   // sequencer 1: S01-S99 初始化 / S01-S99 Initial
   INITIAL_STEP F12_Initial:   // S1, max time T#10S, warning time T#7S
              S    #ioPM_Inface.InitialRun
              R    #ioPM_Inface.InitialOK
              R    #ioPM_Inface.WaitRunning
              R    #ioPM_Inface.Running
              R    #ioPM_Inface.ProcessComplete
              R    #ioPM_Inface.UnPause
              R    "Station_Sys".Cmd.Calibration
              R    "Station_Sys".Cmd.ChangeOver
                   //"ST350_Sys".Cmd.DryRun
              R    "Station_Sys".Cmd.Reserve
              R    "Station_Sys".Cmd.OneCycle
          S1  N    "AutoProcessControl".A_Table_2Loading.ServoRunCount:=0
              R    #ioPM_Inface.ProcessStart
   END_STEP
   TRANSITION Trans1 FROM F12_Initial TO S2   // T1
      := #iSysInface.Ready;
   END_TRANSITION
   STEP S2:   // S2, max time T#10S, warning time T#7S
   END_STEP
   TRANSITION Trans2 FROM S2 TO S3   // T2
      := TRUE;
   END_TRANSITION
   STEP S4:   // S4, max time T#10S, warning time T#7S
   END_STEP
   TRANSITION Trans3 FROM S4 TO S5_MESInitial   // T3
      := TRUE;
   END_TRANSITION
   STEP S5_MESInitial:   // S5, max time T#10S, warning time T#7S
   END_STEP
   TRANSITION Trans325 FROM S5_MESInitial TO WaitRobotInitialFinish   // T4
      := TRUE;
   END_TRANSITION
   STEP S10_InitialFinish:   // S10, max time T#10S, warning time T#7S
              S    #ioPM_Inface.InitialOK
   END_STEP
   TRANSITION Trans102 FROM S10_InitialFinish TO ProcessStart   // T10, jump
      := #ioPM_Inface.Running;
   END_TRANSITION
   STEP S3:   // S3, max time T#10S, warning time T#7S
   END_STEP
   TRANSITION Trans613 FROM S3 TO "ServoReady?"   // T607
      := TRUE;
   END_TRANSITION
   STEP WaitRobotInitialFinish:   // S8, max time T#10S, warning time T#7S
   END_STEP
   TRANSITION Trans10 FROM WaitRobotInitialFinish TO "CheckA-Loading-02HorizontalCylinderPos"   // T8
      := "KukaRobot3_CtrlDB".sROBtoPLC.User.Home.DO163_HomeSeqOK OR "KukaRobot3_CtrlDB".sROBtoPLC.Sys.SO.IN_HOME;
   END_TRANSITION
   STEP "A-Loading-02UpDownTakeCylinderToHP_2":   // S120, max time T#10S, warning time T#7S
              S    "ST10Cylinder".Cy[4].Inout.AutoGoHome
              R    "ST10Cylinder".Cy[4].Inout.AutoGoWork
   END_STEP
   TRANSITION Trans768 FROM "A-Loading-02UpDownTakeCylinderToHP_2" TO "A-Loading-02HorizontalCylinderToHP"   // T121
      := NOT "ST10Cylinder".Cy[4].In.WorkPositionSensor AND "ST10Cylinder".Cy[4].In.HomePositionSensor;
   END_TRANSITION
   STEP "CheckA-Loading-02HorizontalCylinderPos":   // S117, max time T#10S, warning time T#7S
   END_STEP
   TRANSITION Trans117 FROM "CheckA-Loading-02HorizontalCylinderPos" TO "A-Loading-02HorizontalCylinderToHP"   // T117
      := NOT "ST10Cylinder".Cy[3].In.WorkPositionSensor AND "ST10Cylinder".Cy[3].In.HomePositionSensor;
   END_TRANSITION
   TRANSITION Trans119 FROM "CheckA-Loading-02HorizontalCylinderPos" TO "A-Loading-02UpDownTakeCylinderToHP_2"   // T119
      := ("ST10Cylinder".Cy[3].In.WorkPositionSensor AND NOT "ST10Cylinder".Cy[3].In.HomePositionSensor) OR (NOT "ST10Cylinder".Cy[3].In.WorkPositionSensor AND NOT "ST10Cylinder".Cy[3].In.HomePositionSensor);
   END_TRANSITION
   STEP "A-Loading-02HorizontalCylinderToHP":   // S119, max time T#10S, warning time T#7S
              S    "ST10Cylinder".Cy[3].Inout.AutoGoHome
              R    "ST10Cylinder".Cy[3].Inout.AutoGoWork
   END_STEP
   TRANSITION Trans767 FROM "A-Loading-02HorizontalCylinderToHP" TO "A-Loading-02UpDownTakeCylinderToWP"   // T120
      := NOT "ST10Cylinder".Cy[3].In.WorkPositionSensor AND "ST10Cylinder".Cy[3].In.HomePositionSensor;
   END_TRANSITION
   STEP "A-Loading-02UpDownTakeCylinderToWP":   // S116, max time T#10S, warning time T#7S
              R    "ST10Cylinder".Cy[4].Inout.AutoGoHome
              S    "ST10Cylinder".Cy[4].Inout.AutoGoWork
   END_STEP
   TRANSITION Trans765 FROM "A-Loading-02UpDownTakeCylinderToWP" TO S10_InitialFinish   // T116
      := "ST10Cylinder".Cy[4].In.WorkPositionSensor AND NOT "ST10Cylinder".Cy[4].In.HomePositionSensor;
   END_TRANSITION
   STEP "ServoReady?":   // S6, max time T#10S, warning time T#7S
   END_STEP
   TRANSITION Trans4 FROM "ServoReady?" TO S4   // T5
      := "ServoV90_A4".Out.oReady;
   END_TRANSITION

   // sequencer 2: S100-S199 等待到位 / S100-S199 CheckSysStatus
   STEP "A-Loading-02HorizontalCylinderToWP_1":   // S121, max time T#10S, warning time T#7S
              R    "ST10Cylinder".Cy[3].Inout.AutoGoHome
              S    "ST10Cylinder".Cy[3].Inout.AutoGoWork
   END_STEP
   TRANSITION Trans769 FROM "A-Loading-02HorizontalCylinderToWP_1" TO TimDelay   // T122
      := "ST10Cylinder".Cy[3].In.WorkPositionSensor AND NOT "ST10Cylinder".Cy[3].In.HomePositionSensor;
   END_TRANSITION
   STEP "A-Loading-02UpDownTakeCylinderToHP3":   // S122, max time T#10S, warning time T#7S
              S    "ST10Cylinder".Cy[4].Inout.AutoGoHome
              R    "ST10Cylinder".Cy[4].Inout.AutoGoWork
   END_STEP
   TRANSITION Trans770 FROM "A-Loading-02UpDownTakeCylinderToHP3" TO "A-Loading-02HorizontalCylinderToWP_1"   // T123
      := NOT "ST10Cylinder".Cy[4].In.WorkPositionSensor AND "ST10Cylinder".Cy[4].In.HomePositionSensor;
   END_TRANSITION
   STEP TimDelay:   // S123, max time T#10S, warning time T#7S
   END_STEP
   TRANSITION Trans124 FROM TimDelay TO "A-Loading-02UpDownTakeCylinderToWP_1"   // T124
      := #TimDelay.T > t#100MS;
   END_TRANSITION
   STEP SensorNoPart:   // S113, max time T#10S, warning time T#7S
   END_STEP
   TRANSITION Trans113 FROM SensorNoPart TO WaitEmptyFinish   // T113
      := #TOF[5].Q;
   END_TRANSITION
   STEP ProcessStart:   // S100, max time T#10S, warning time T#7S
      // 自动等待开始运行
              R    #ioPM_Inface.InitialRun
              R    #ioPM_Inface.ProcessComplete
              R    #ioPM_Inface.ProcessStart
              S    #ioPM_Inface.InitialOK
              S    #ioPM_Inface.WaitRunning
          S1  N    #ioPM_Inface.ProcessResult:=0
              R    "ST10_GeneralData".FlowControl_Handshake[12].Start
              R    "ST10_GeneralData".FlowControl_Handshake[12].Done
   END_STEP
   TRANSITION Trans200 FROM ProcessStart TO WaitChangeOverFinish   // T100
      := NOT #ioPM_Inface.AlarmCycleStop AND #ioPM_Inface.Running AND NOT #iSysInface.Auto.RunningOver AND (NOT #iSysInface.Auto.OneCycleMode OR (#iSysInface.Auto.OneCycleMode AND #ioPM_Inface.TriggerOneCycle));
   END_TRANSITION
   STEP TimDelay_1:   // S124, max time T#10S, warning time T#7S
   END_STEP
   TRANSITION Trans125 FROM TimDelay_1 TO "A-Loading-02HorizontalCylinderToHP_1"   // T125
      := #TimDelay_1.T > t#1S;
   END_TRANSITION
   STEP "Process Finish":   // S237, max time T#10S, warning time T#7S
   END_STEP
   TRANSITION Trans250 FROM "Process Finish" TO ProcessStart   // T249, jump
      := TRUE;
   END_TRANSITION
   STEP "A-Loading-02HorizontalCylinderToHP_1":   // S125, max time T#10S, warning time T#7S
              S    "ST10Cylinder".Cy[3].Inout.AutoGoHome
              R    "ST10Cylinder".Cy[3].Inout.AutoGoWork
   END_STEP
   TRANSITION Trans771 FROM "A-Loading-02HorizontalCylinderToHP_1" TO "Detect UnloadingRing exist_1"   // T126
      := NOT "ST10Cylinder".Cy[3].In.WorkPositionSensor AND "ST10Cylinder".Cy[3].In.HomePositionSensor;
   END_TRANSITION
   STEP "No cartridge":   // S127, max time T#10S, warning time T#7S
   END_STEP
   TRANSITION Trans129 FROM "No cartridge" TO ServoNeedMove   // T129, jump
      := TRUE;
   END_TRANSITION
   STEP "A-Loading-02UpDownTakeCylinderToWP_1":   // S118, max time T#10S, warning time T#7S
              R    "ST10Cylinder".Cy[4].Inout.AutoGoHome
              S    "ST10Cylinder".Cy[4].Inout.AutoGoWork
   END_STEP
   TRANSITION Trans766 FROM "A-Loading-02UpDownTakeCylinderToWP_1" TO TimDelay_1   // T118
      := "ST10Cylinder".Cy[4].In.WorkPositionSensor AND NOT "ST10Cylinder".Cy[4].In.HomePositionSensor;
   END_TRANSITION
   STEP ServoNeedMove:   // S126, max time T#10S, warning time T#7S
   END_STEP
   TRANSITION Trans128 FROM ServoNeedMove TO WaitChangeOverOK   // T128
      := TRUE;
   END_TRANSITION
   STEP WaitChangeOverFinish:   // S101, max time T#10S, warning time T#7S
   END_STEP
   TRANSITION Trans101 FROM WaitChangeOverFinish TO "Clearing mode?"   // T101
      := TRUE;
   END_TRANSITION
   STEP WaitServoInPosition:   // S105, max time T#10S, warning time T#7S
              R    #ioPM_Inface.ProcessComplete
              S    #ioPM_Inface.ProcessStart
   END_STEP
   TRANSITION Trans103 FROM WaitServoInPosition TO WaitFixtureScanFinish   // T105
      := TRUE;
   END_TRANSITION
   TRANSITION Trans127 FROM WaitServoInPosition TO ServoNeedMove   // T127
      := "AlwaysTRUE" AND NOT "AlwaysTRUE";
   END_TRANSITION
   STEP "Detect cartridge exist":   // S106, max time T#10S, warning time T#7S
   END_STEP
   TRANSITION Trans106 FROM "Detect cartridge exist" TO CountClear   // T106
      := "ServoV90_A4".Out.oServoPosOK AND #TON[0].Q;
   END_TRANSITION
   TRANSITION Trans107 FROM "Detect cartridge exist" TO "No cartridge"   // T107
      := (NOT "iA-Loading-02PipeDetection" OR NOT "ServoV90_A4".Out.oServoPosOK) AND (#"Detect cartridge exist".T > t#1500MS);
   END_TRANSITION
   STEP "Detect UnloadingRing exist":   // S108, max time T#10S, warning time T#7S
   END_STEP
   TRANSITION Trans110 FROM "Detect UnloadingRing exist" TO "Request robot pick"   // T110
      := #TON[4].Q;
   END_TRANSITION
   TRANSITION Trans111 FROM "Detect UnloadingRing exist" TO "A-Loading-02UpDownTakeCylinderToHP3"   // T111
      := #TOF[5].Q AND NOT "ChangeOver_DB".Global.ScanFixtureFlag AND "ChangeOver_DB".Global.AllFixtureScanCompareOk AND "AutoProcessData".GlobalData.Table2CodeOKFlag;
   END_TRANSITION
   STEP "Detect Ring exist":   // S107, max time T#10S, warning time T#7S
   END_STEP
   TRANSITION Trans108 FROM "Detect Ring exist" TO Step111   // T108
      := #TON[2].Q;
   END_TRANSITION
   TRANSITION Trans109 FROM "Detect Ring exist" TO "No Ring"   // T109
      := NOT "iA-Loading-02Detection" AND (#"Detect Ring exist".T > t#1500MS);
   END_TRANSITION
   STEP "Wait  robot finish task":   // S130, max time T#10S, warning time T#7S
   END_STEP
   TRANSITION Trans146 FROM "Wait  robot finish task" TO SensorNoPart   // T146
      := "KukaRobot3_CtrlDB".sROBtoPLC.User.Cycle.DO258_PickTableFinish;
   END_TRANSITION
   STEP "Request robot pick":   // S112, max time T#10S, warning time T#7S
              N    "AutoProcessControl".A_Table_2Loading.Robot3PickPrimit
              S    #ioPM_Inface.ProcessComplete
              R    #ioPM_Inface.ProcessStart
   END_STEP
   TRANSITION Trans283 FROM "Request robot pick" TO "Wait  robot finish task"   // T112
      := "KukaRobot3_CtrlDB".sROBtoPLC.User.Cycle.DO257_PickTableInside AND NOT "KukaRobot3_CtrlDB".sROBtoPLC.User.Cycle.DO258_PickTableFinish;
   END_TRANSITION
   STEP "No Ring":   // S128, max time T#10S, warning time T#7S
   END_STEP
   TRANSITION Trans130 FROM "No Ring" TO ServoNeedMove   // T130, jump
      := TRUE;
   END_TRANSITION
   STEP "Detect UnloadingRing exist_1":   // S109, max time T#10S, warning time T#7S
   END_STEP
   TRANSITION Trans112 FROM "Detect UnloadingRing exist_1" TO ResetPartMissingAlarm   // T114
      := #TON[4].Q;
   END_TRANSITION
   TRANSITION Trans115 FROM "Detect UnloadingRing exist_1" TO PartMissingAlarm   // T115
      := NOT "iA-Loading-02GripperTakeDetection" AND (#"Detect UnloadingRing exist_1".T > t#3000MS);
   END_TRANSITION
   STEP PartMissingAlarm:   // S110, max time T#10S, warning time T#7S
          S1  S    "ST10_DeviceError".A.A2TableUnloading.RingCheckExist
   END_STEP
   TRANSITION Trans131 FROM PartMissingAlarm TO ProcessStart   // T131, jump
      := #iSysInface.Reset OR NOT "ST10_DeviceError"."A".A2TableUnloading.RingCheckExist;
   END_TRANSITION
   STEP Step111:   // S111, max time T#10S, warning time T#7S
          S1  N    "AutoProcessControl".A_Table_2Loading.ServoRunCount:=0
   END_STEP
   TRANSITION Trans132 FROM Step111 TO "Detect UnloadingRing exist"   // T132
      := TRUE;
   END_TRANSITION
   STEP CountClear:   // S114, max time T#10S, warning time T#7S
   END_STEP
   TRANSITION Trans133 FROM CountClear TO "Detect Ring exist"   // T133
      := TRUE;
   END_TRANSITION
   STEP "Servo returns to1st Pos":   // S16, max time T#10S, warning time T#7S
      interlock C := "ServoV90_A4".Out.oReady;
      (C)     N    "ServoV90_DeviceCtl".V90Servo[4].Point["ServoV90_DeviceCtl".V90Servo[4].nPositionListNo].Start
   END_STEP
   TRANSITION Trans17 FROM "Servo returns to1st Pos" TO CountCompare   // T16
      := "ServoV90_DeviceCtl".V90Servo[4].Point["ServoV90_DeviceCtl".V90Servo[4].nPositionListNo].Achieve;
   END_TRANSITION
   STEP ServoPosCount:   // S17, max time T#10S, warning time T#7S
          S1  N    "ServoV90_DeviceCtl".V90Servo[4].nPositionListNo:= "ServoV90_DeviceCtl".V90Servo[4].nPositionListNo+1
          S1  N    "AutoProcessControl".A_Table_2Loading.ServoRunCount:="AutoProcessControl".A_Table_2Loading.ServoRunCount+1
   END_STEP
   TRANSITION Trans18 FROM ServoPosCount TO ServoPosCountJudge   // T17
      := TRUE;
   END_TRANSITION
   STEP ServoPosCountJudge:   // S18, max time T#10S, warning time T#7S
   END_STEP
   TRANSITION Trans19 FROM ServoPosCountJudge TO "Servo returns to1st Pos"   // T18
      := ("ServoV90_DeviceCtl".V90Servo[4].nPositionListNo >= 1) AND ("ServoV90_DeviceCtl".V90Servo[4].nPositionListNo <= 8);
   END_TRANSITION
   TRANSITION Trans20 FROM ServoPosCountJudge TO ServoPosCountClear   // T19
      := ("ServoV90_A4".Auto.Index <= 0) OR ("ServoV90_A4".Auto.Index > 8);
   END_TRANSITION
   STEP ServoPosCountClear:   // S19, max time T#10S, warning time T#7S
              N    "ServoV90_DeviceCtl".V90Servo[4].nPositionListNo:=1
   END_STEP
   TRANSITION Trans21 FROM ServoPosCountClear TO "Servo returns to1st Pos"   // T20
      := "ServoV90_DeviceCtl".V90Servo[4].nPositionListNo = 1;
   END_TRANSITION
   STEP CountCompare:   // S20, max time T#10S, warning time T#7S
   END_STEP
   TRANSITION Trans22 FROM CountCompare TO ProcessStart   // T21, jump
      := "AutoProcessControl".A_Table_2Loading.ServoRunCount <= 8;
   END_TRANSITION
   TRANSITION Trans23 FROM CountCompare TO TableLackMaterial   // T22
      := "AutoProcessControl".A_Table_2Loading.ServoRunCount > 8;
   END_TRANSITION
   STEP TableLackMaterial:   // S21, max time T#10S, warning time T#7S
          S1  S    "ST10_DeviceError".A.A2TableUnloading.LackMaterial
   END_STEP
   TRANSITION Trans24 FROM TableLackMaterial TO CountClear_1   // T23
      := #iSysInface.Reset;
   END_TRANSITION
   STEP CountClear_1:   // S115, max time T#10S, warning time T#7S
          S1  N    "AutoProcessControl".A_Table_2Loading.ServoRunCount:=1
   END_STEP
   TRANSITION Trans134 FROM CountClear_1 TO CountCompare   // T134, jump
      := TRUE;
   END_TRANSITION
   STEP "Clearing mode?":   // S129, max time T#10S, warning time T#7S
   END_STEP
   TRANSITION Trans135 FROM "Clearing mode?" TO WaitServoInPosition   // T135
      := NOT "Station_Sys".Cmd.ClearFlags OR ("Station_Sys".Cmd.ClearFlags AND "AutoProcessControl".B_Press_2.Robot3PutRingPrimit AND ("AutoProcessData".F_Robot3Grip2.PartStatus = 0));
   END_TRANSITION
   STEP WaitChangeOverOK:   // S133, max time T#10S, warning time T#7S
   END_STEP
   TRANSITION Trans139 FROM WaitChangeOverOK TO ServoPosCount   // T139
      := "ChangeOver_DB".Global.AllFixtureScanCompareOk AND NOT "ChangeOver_DB".Global.ScanFixtureFlag;
   END_TRANSITION
   TRANSITION Trans31 FROM WaitChangeOverOK TO "Detect UnloadingRing exist"   // T31, jump
      := NOT "ChangeOver_DB".Global.AllFixtureScanCompareOk AND #TON[4].Q AND NOT "ST10_GeneralData".FunctionDeSelect.Global.DeSelectPB_ScanFixture;
   END_TRANSITION
   STEP WaitEmptyFinish:   // S134, max time T#10S, warning time T#7S
   END_STEP
   TRANSITION Trans140 FROM WaitEmptyFinish TO "Process Finish"   // T140
      := NOT "ChangeOver_DB".Global.ManualModeFlag;
   END_TRANSITION
   STEP WaitFixtureScanFinish:   // S30, max time T#10S, warning time T#7S
   END_STEP
   TRANSITION Trans30 FROM WaitFixtureScanFinish TO "Detect cartridge exist"   // T30
      := (NOT "ChangeOver_DB".Global.ScanFixtureFlag AND NOT "ChangeOver_DB".Global.ChangeOverRequest) OR #TON[4].Q;
   END_TRANSITION
   STEP ResetPartMissingAlarm:   // S31, max time T#10S, warning time T#7S
   END_STEP
   TRANSITION Trans32 FROM ResetPartMissingAlarm TO "Detect UnloadingRing exist"   // T32, jump
      := TRUE;
   END_TRANSITION

   // permanent post-instructions
   NETWORK 1
      #ioPM_Inface.StepNum := #RT_DATA.S_DISPLAY;
   NETWORK 2
      IF #iSysInface.Reset THEN #AlarmID := 0; END_IF;
   NETWORK 3
      #TON[10].TON(IN := #工件放行中, PT := T#0.5S);
      IF #TON[10].Q THEN #工件放行中 := FALSE; END_IF;
END_FUNCTION_BLOCK

FUNCTION_BLOCK "ST10_Flow14_B2Press"   // FB1084, GRAPH
// stored: AcknowledgeErrorsRequired false, AutoNumber false, GraphVersion 6.0, InitialValuesAcquisition false, SetENOAutomatically false
   // inherited from GRAPH_BASE
   VAR_INPUT
      iSysInface : "RCS_SysComInterface_V1";
   END_VAR
   VAR_IN_OUT
      ioPM_Inface : "RCS_PMInterface_V1";
      ioStatus : Int;
   END_VAR
   VAR
      sCtrlMode { S7_SetPoint := 'True'} : "SysFlowCtrlGraph";
      sUpdMES_Data : Bool;   // 更新MES数据
      工件放行中 : Bool;
      前站站号 { ExternalAccessible := 'False'; ExternalVisible := 'False'; ExternalWritable := 'False'} : UInt;
      本站站号 { ExternalAccessible := 'False'; ExternalVisible := 'False'; ExternalWritable := 'False'} : UInt;
      弹窗Temp : Array[1..10] of Int;
      AlarmID : Int;
      TON { S7_SetPoint := 'True'} : Array[0..10] of TON_TIME;
      TOF { S7_SetPoint := 'True'} : Array[0..10] of TOF_TIME;
      sUP { S7_SetPoint := 'True'} : Array[0..10] of Bool;
      更新RFID完成 : Bool;
   END_VAR
   VAR_TEMP
      Tempresult : USInt;
      本站站号乘10 : UInt;
   END_VAR
   // // TON[0] : 托盘流入1托盘到位传感器 / iA-Rotating product Check
   // // TON[1] : 托盘流入1托盘到位传感器
   // // TON[2] : 托盘流入1产品有无传感器
   // // TON[3] : 托盘流入1产品有无传感器
   // // TON[4] : 托盘流入1姿态检测光电2
   // // TON[5] : 托盘流入1姿态检测光电3
   // // TON[0].Q : 托盘流入1托盘到位 / iA-Rotating product Check
   // // TON[1].Q : 托盘流入1托盘无
   // // TON[2].Q : 托盘流入1有产品
   // // TON[3].Q : 托盘流入1无产品
   // // TON[4].Q : 托盘流入1姿态检测光电2
   // // TON[5].Q : 托盘流入1姿态检测光电3
   // // TOF[1] : iA-Rotating product Check
BEGIN
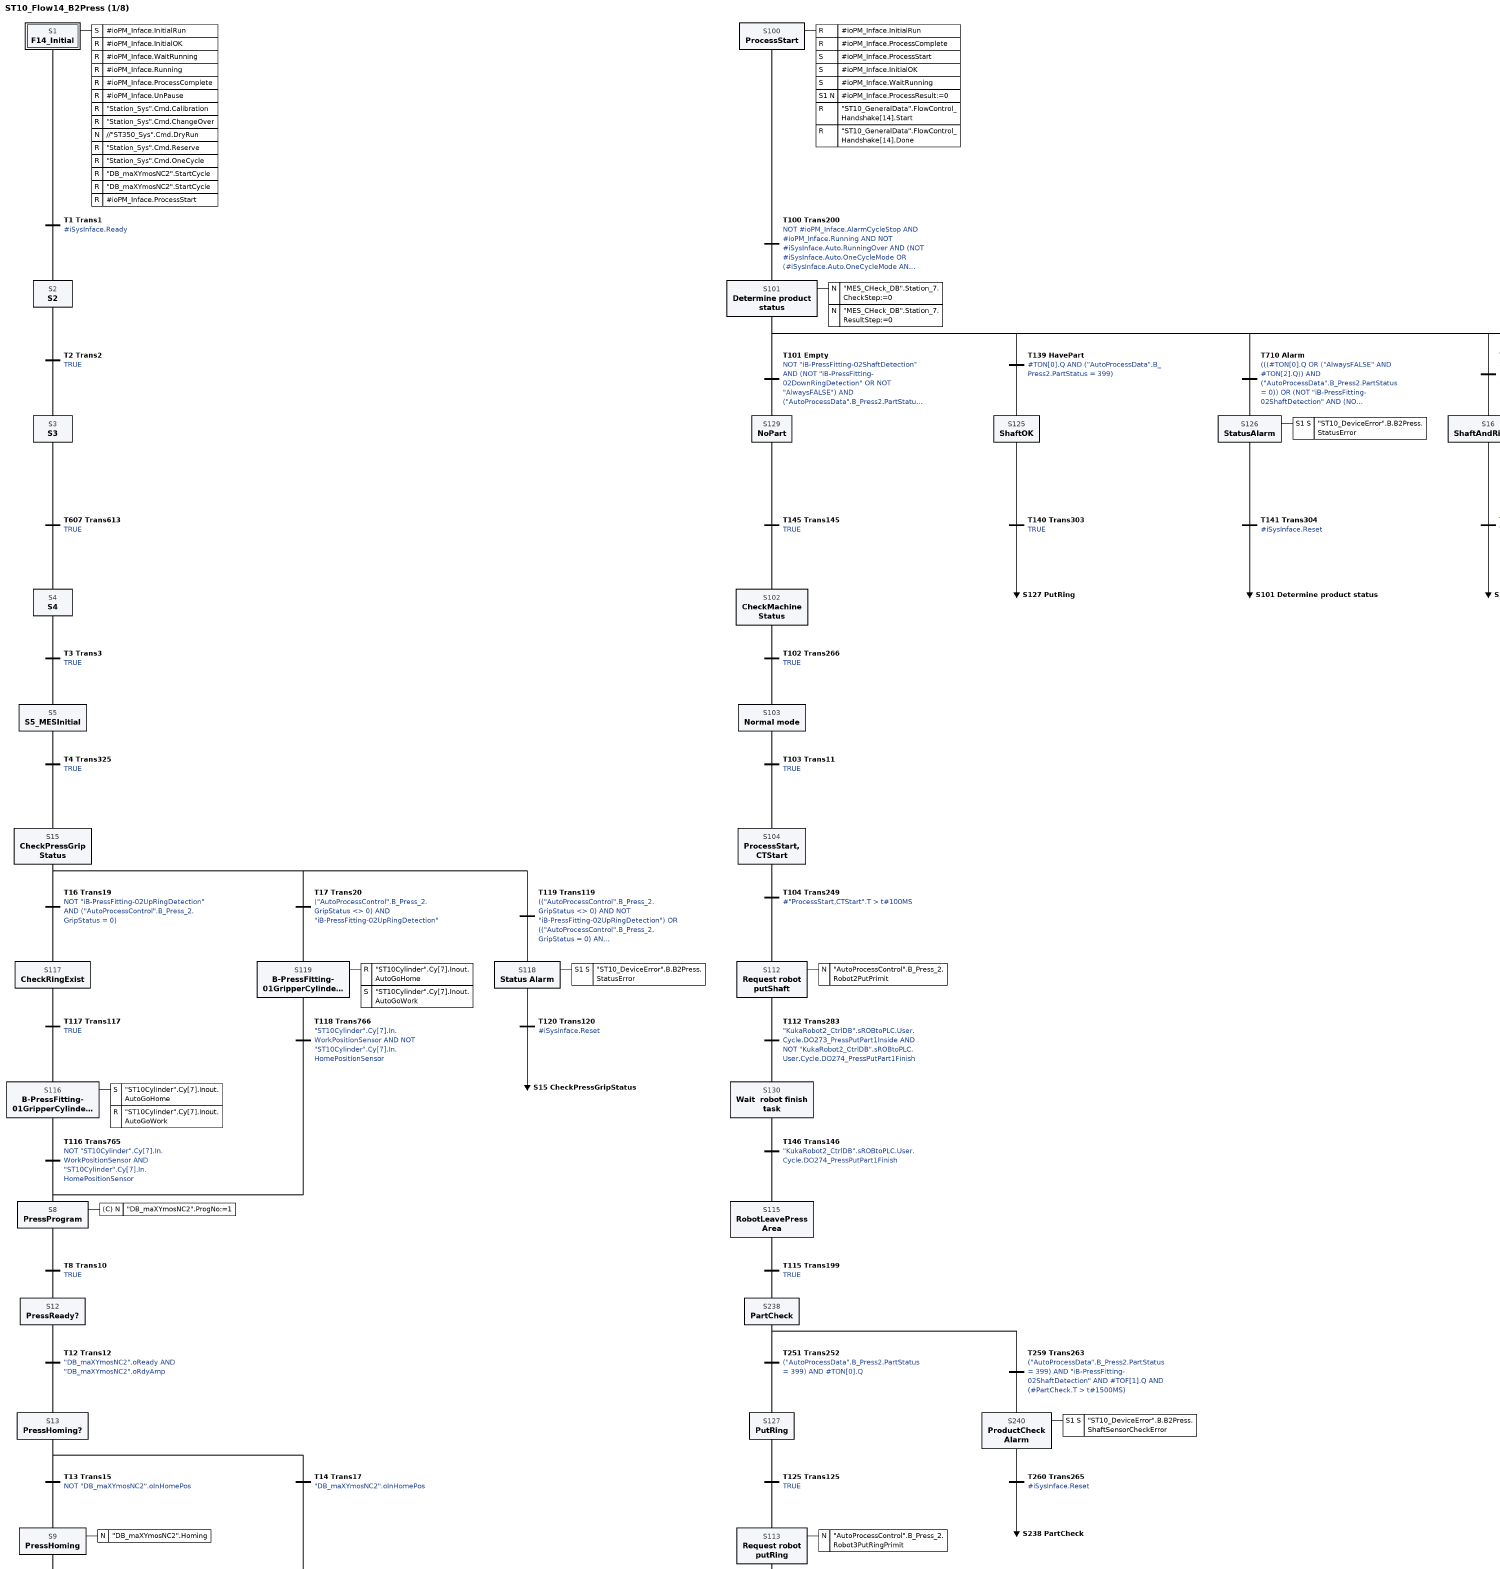
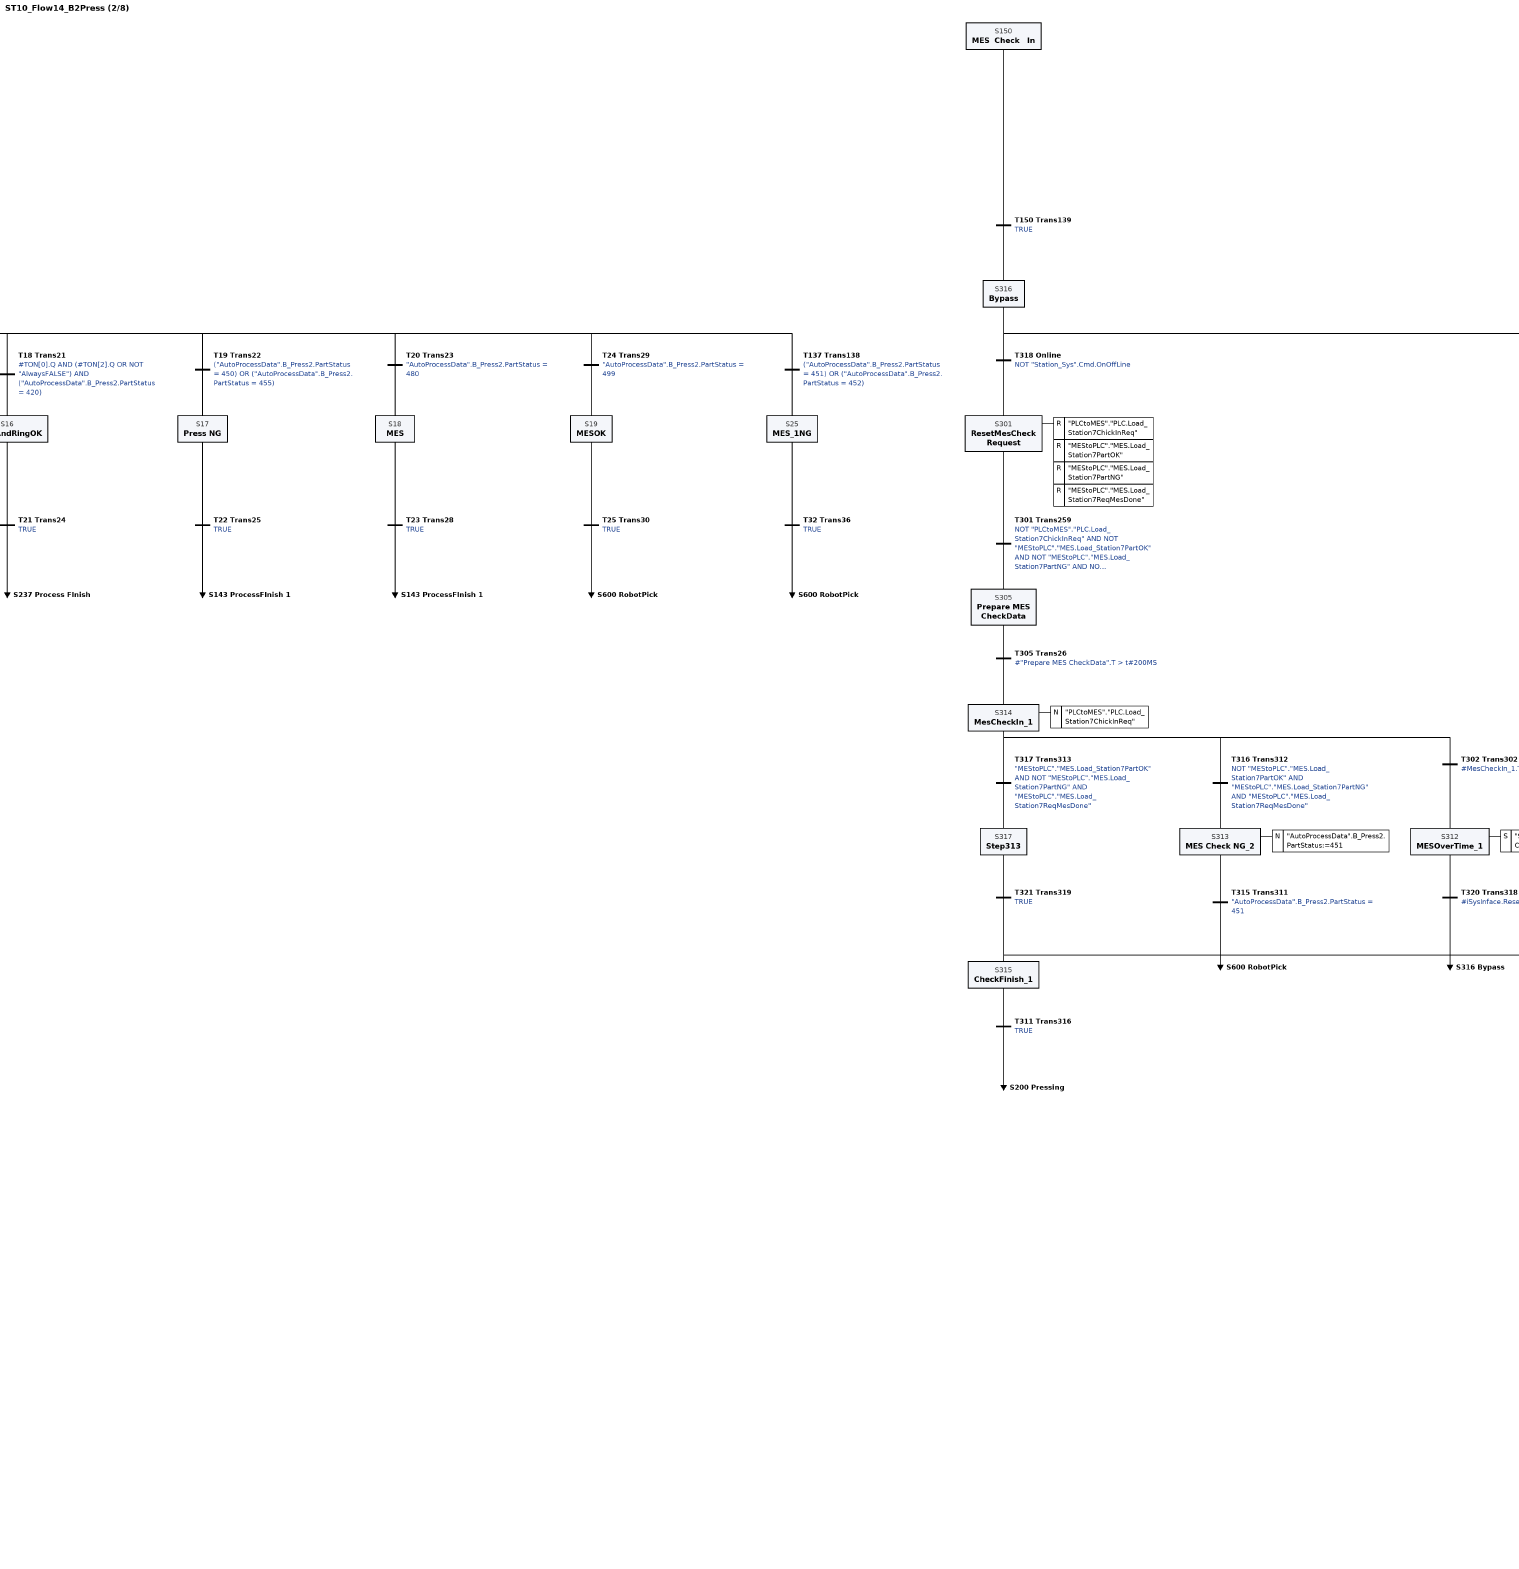
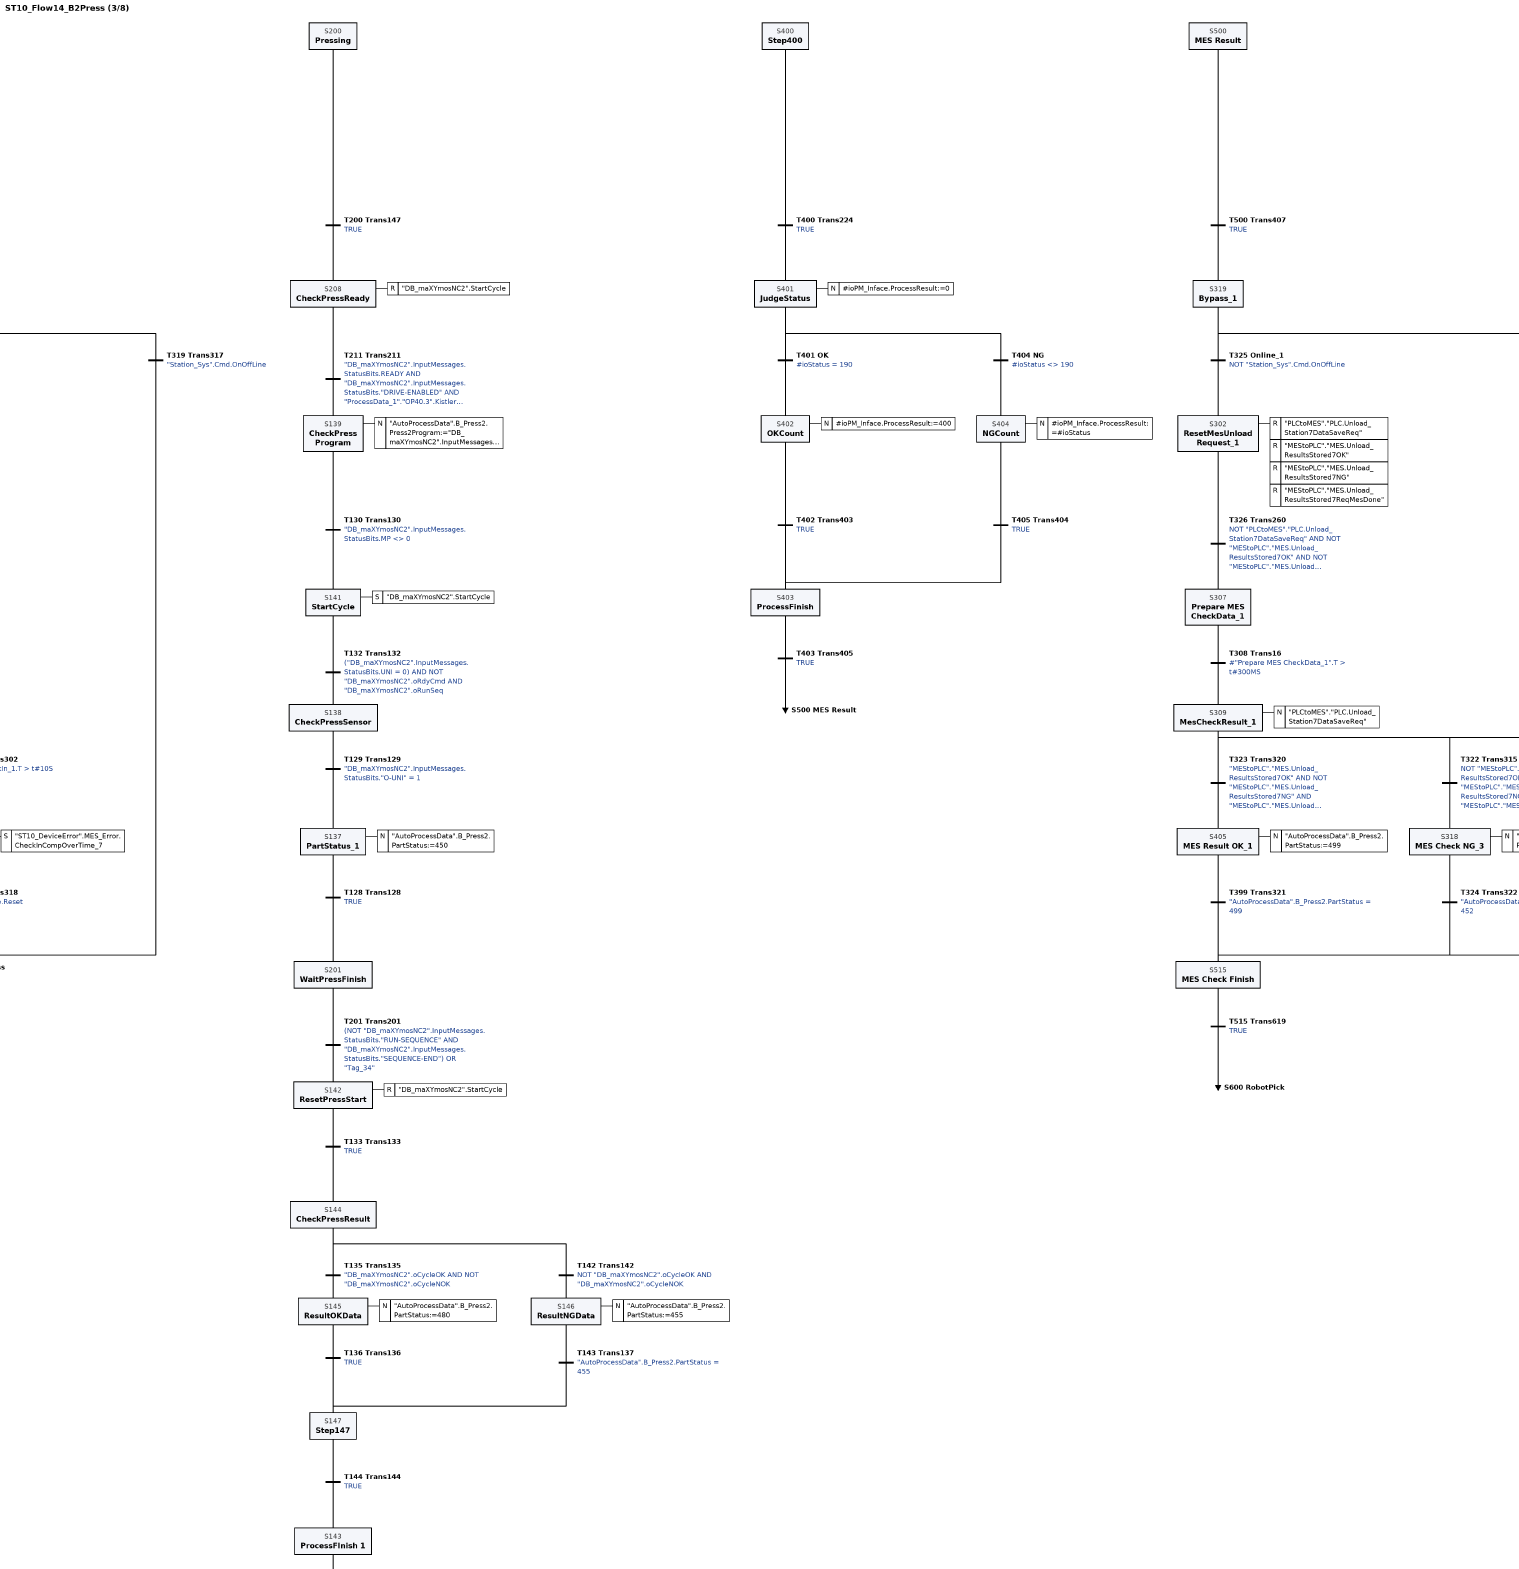
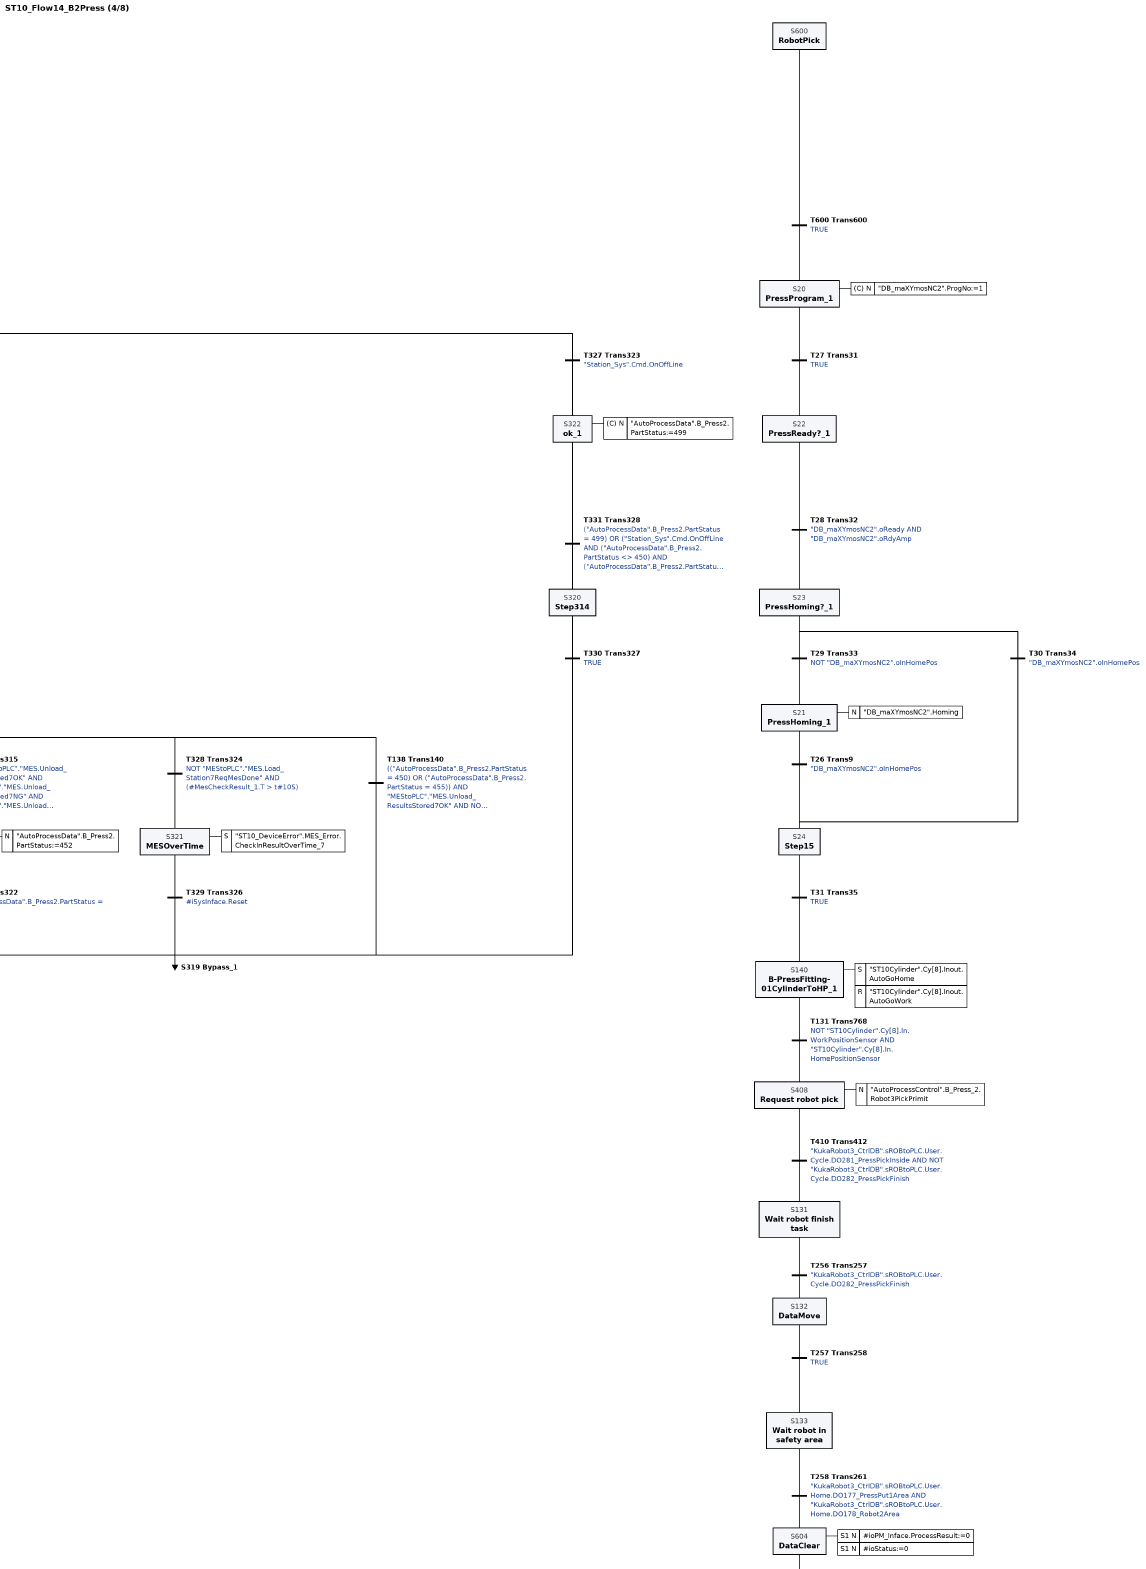
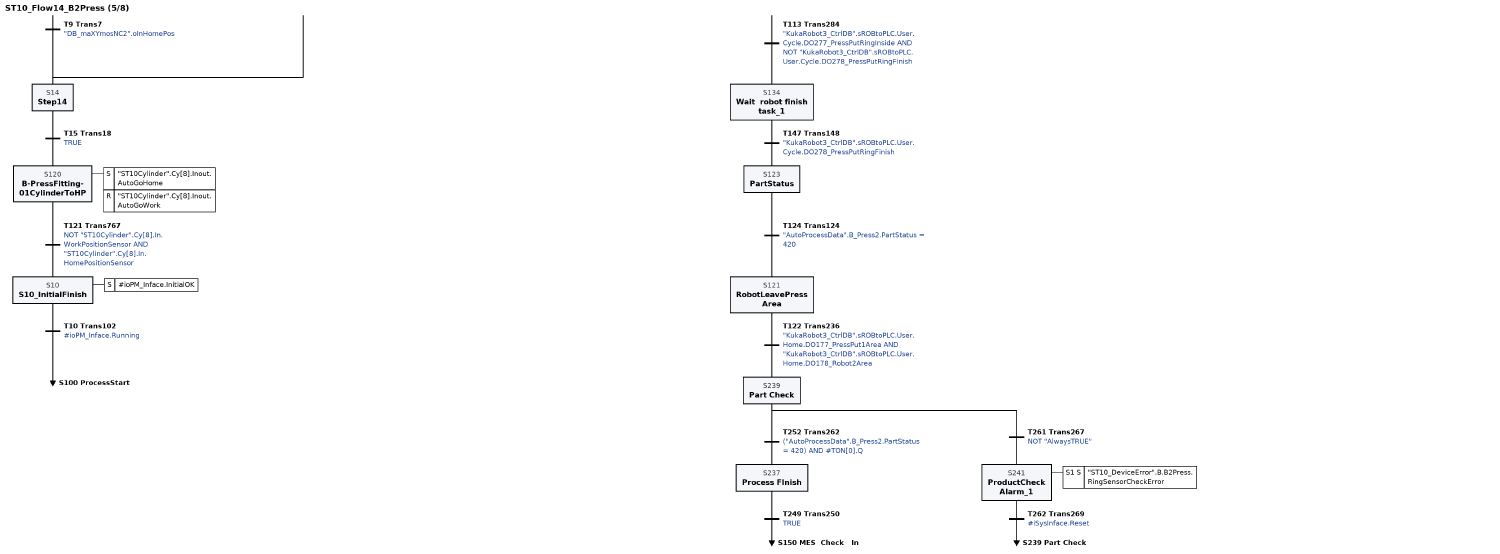
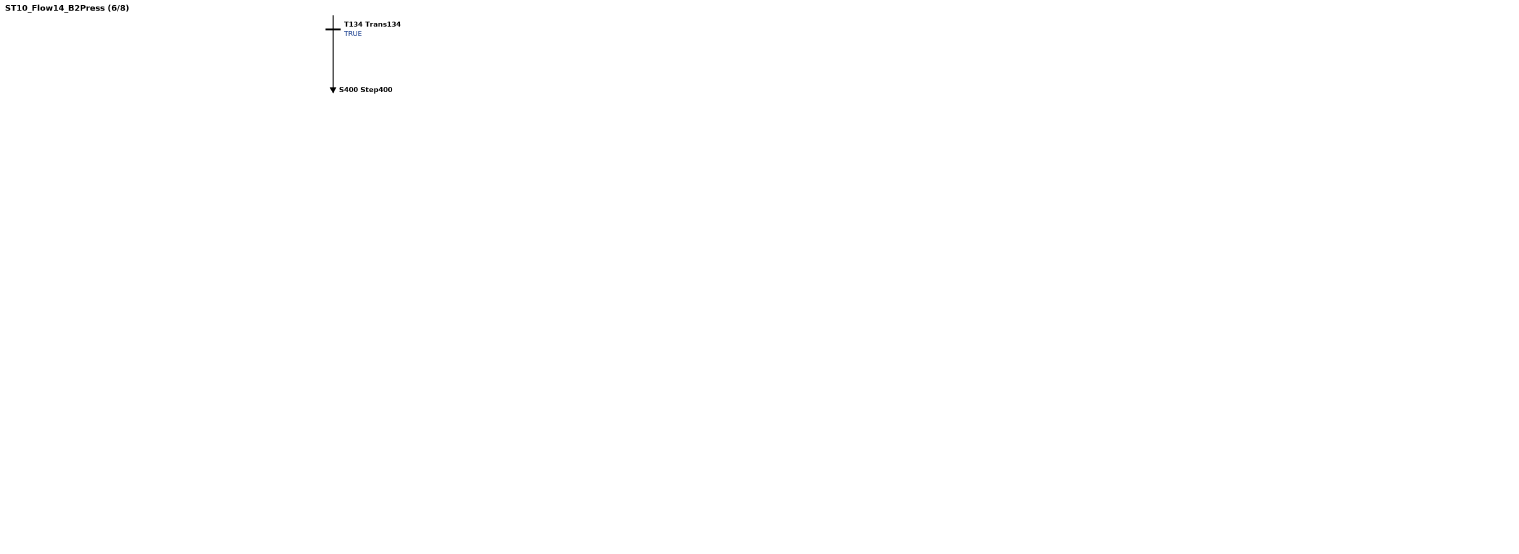
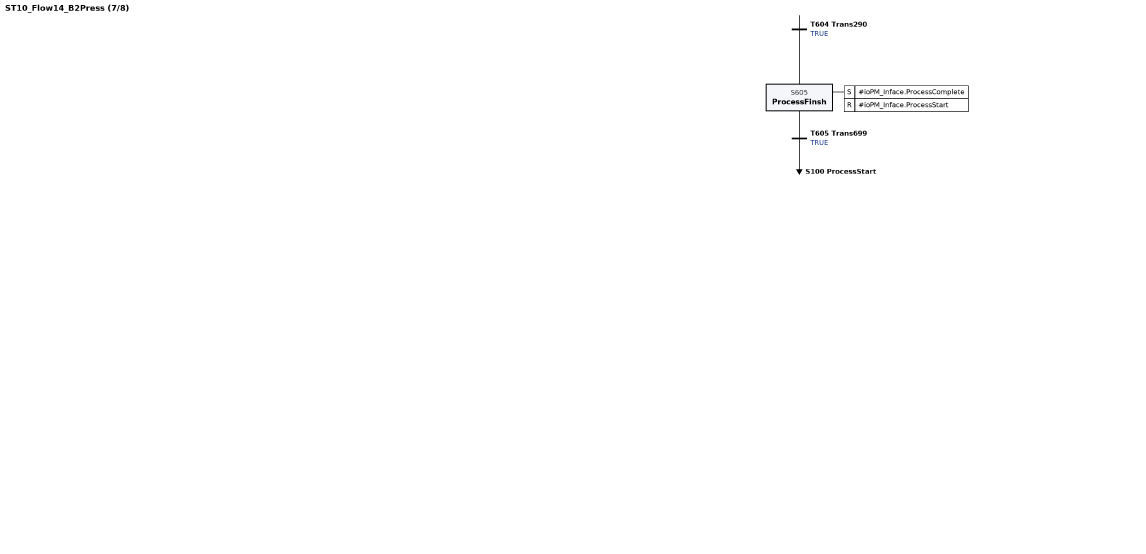
   // permanent pre-instructions
   NETWORK 1
      #TON[10].TON(IN := "AlwaysTRUE" AND "Station_Sys".Alarm.ImmediatelyStop, PT := T#300ms);
      #ioPM_Inface.AlarmImdilyStop := #TON[10].Q;
      #ioPM_Inface.AlarmCycleStop := "AlwaysTRUE" AND "Station_Sys".Alarm.CycleStop;
   NETWORK 2
      IF NOT False THEN
          #sCtrlMode(iSysInface := #iSysInface, ioPM_Inface := #ioPM_Inface, ioGraphCtrl := #RT_DATA.MOP);   // "SysFlowCtrlGraph"
      END_IF;
   NETWORK 3
      #TON[0].TON(IN := "AlwaysTRUE" AND "iB-PressFitting-02ShaftDetection", PT := t#500ms);   // 工位11有托盘
      #TOF[1].TOF(IN := "AlwaysTRUE" AND NOT "iB-PressFitting-02ShaftDetection", PT := T#300ms);   // 工位无托盘
      #TON[2].TON(IN := "AlwaysTRUE" AND "iB-PressFitting-02DownRingDetection", PT := T#300ms);
      #TOF[3].TOF(IN := "AlwaysTRUE" AND NOT "iB-PressFitting-02DownRingDetection", PT := T#300ms);
      #TON[4].TON(IN := "AlwaysTRUE" AND "iB-PressFitting-02UpRingDetection", PT := T#300ms);
      #TON[5].TON(IN := "AlwaysTRUE" AND NOT "iB-PressFitting-02UpRingDetection", PT := T#300ms);
   NETWORK 4
      #前站站号 := 345;
      #本站站号 := 350;

   // sequencer 1: S01-S99 初始化 / S01-S99 Initial
   INITIAL_STEP F14_Initial:   // S1, max time T#10S, warning time T#7S
              S    #ioPM_Inface.InitialRun
              R    #ioPM_Inface.InitialOK
              R    #ioPM_Inface.WaitRunning
              R    #ioPM_Inface.Running
              R    #ioPM_Inface.ProcessComplete
              R    #ioPM_Inface.UnPause
              R    "Station_Sys".Cmd.Calibration
              R    "Station_Sys".Cmd.ChangeOver
                   //"ST350_Sys".Cmd.DryRun
              R    "Station_Sys".Cmd.Reserve
              R    "Station_Sys".Cmd.OneCycle
              R    "DB_maXYmosNC2".StartCycle
              R    "DB_maXYmosNC2".StartCycle
              R    #ioPM_Inface.ProcessStart
              R    "AutoProcessControl".B_Press_2.Robot3PickPrimit
              R    "AutoProcessControl".B_Press_2.Robot3PutRingPrimit
              R    "AutoProcessControl".B_Press_2.Robot2PutPrimit
   END_STEP
   TRANSITION Trans1 FROM F14_Initial TO S2   // T1
      := #iSysInface.Ready;
   END_TRANSITION
   STEP S2:   // S2, max time T#10S, warning time T#7S
   END_STEP
   TRANSITION Trans2 FROM S2 TO S3   // T2
      := TRUE;
   END_TRANSITION
   STEP S4:   // S4, max time T#10S, warning time T#7S
   END_STEP
   TRANSITION Trans3 FROM S4 TO S5_MESInitial   // T3
      := TRUE;
   END_TRANSITION
   STEP S5_MESInitial:   // S5, max time T#10S, warning time T#7S
   END_STEP
   TRANSITION Trans325 FROM S5_MESInitial TO CheckPressGripStatus   // T4
      := TRUE;
   END_TRANSITION
   STEP S10_InitialFinish:   // S10, max time T#10S, warning time T#7S
              S    #ioPM_Inface.InitialOK
   END_STEP
   TRANSITION Trans102 FROM S10_InitialFinish TO ProcessStart   // T10, jump
      := #ioPM_Inface.Running;
   END_TRANSITION
   STEP S3:   // S3, max time T#10S, warning time T#7S
   END_STEP
   TRANSITION Trans613 FROM S3 TO S4   // T607
      := TRUE;
   END_TRANSITION
   STEP PressProgram:   // S8, max time T#10S, warning time T#7S
      interlock C := NOT "ST10_GeneralData".FunctionDeSelect."B".FunctionDeSelected_TestPress375A1;
      (C)     N    "DB_maXYmosNC2".ProgNo:=1
   END_STEP
   TRANSITION Trans10 FROM PressProgram TO "PressReady?"   // T8
      := TRUE;
   END_TRANSITION
   STEP PressHoming:   // S9, max time T#10S, warning time T#7S
              N    "DB_maXYmosNC2".Homing
   END_STEP
   TRANSITION Trans7 FROM PressHoming TO Step14   // T9
      := "DB_maXYmosNC2".oInHomePos;
   END_TRANSITION
   STEP "PressReady?":   // S12, max time T#10S, warning time T#7S
   END_STEP
   TRANSITION Trans12 FROM "PressReady?" TO "PressHoming?"   // T12
      := "DB_maXYmosNC2".oReady AND "DB_maXYmosNC2".oRdyAmp;
   END_TRANSITION
   STEP "PressHoming?":   // S13, max time T#10S, warning time T#7S
   END_STEP
   TRANSITION Trans15 FROM "PressHoming?" TO PressHoming   // T13
      := NOT "DB_maXYmosNC2".oInHomePos;
   END_TRANSITION
   TRANSITION Trans17 FROM "PressHoming?" TO Step14   // T14
      := "DB_maXYmosNC2".oInHomePos;
   END_TRANSITION
   STEP Step14:   // S14, max time T#10S, warning time T#7S
   END_STEP
   TRANSITION Trans18 FROM Step14 TO "B-PressFitting-01CylinderToHP"   // T15
      := TRUE;
   END_TRANSITION
   STEP CheckPressGripStatus:   // S15, max time T#10S, warning time T#7S
   END_STEP
   TRANSITION Trans19 FROM CheckPressGripStatus TO CheckRingExist   // T16
      := NOT "iB-PressFitting-02UpRingDetection" AND ("AutoProcessControl".B_Press_2.GripStatus = 0);
   END_TRANSITION
   TRANSITION Trans20 FROM CheckPressGripStatus TO "B-PressFitting-01GripperCylinderToWP"   // T17
      := ("AutoProcessControl".B_Press_2.GripStatus <> 0) AND "iB-PressFitting-02UpRingDetection";
   END_TRANSITION
   TRANSITION Trans119 FROM CheckPressGripStatus TO "Status Alarm"   // T119
      := (("AutoProcessControl".B_Press_2.GripStatus <> 0) AND NOT "iB-PressFitting-02UpRingDetection") OR (("AutoProcessControl".B_Press_2.GripStatus = 0) AND "iB-PressFitting-02UpRingDetection");
   END_TRANSITION
   STEP "B-PressFitting-01GripperCylinderToHP":   // S116, max time T#10S, warning time T#7S
              S    "ST10Cylinder".Cy[7].Inout.AutoGoHome
              R    "ST10Cylinder".Cy[7].Inout.AutoGoWork
   END_STEP
   TRANSITION Trans765 FROM "B-PressFitting-01GripperCylinderToHP" TO PressProgram   // T116
      := NOT "ST10Cylinder".Cy[7].In.WorkPositionSensor AND "ST10Cylinder".Cy[7].In.HomePositionSensor;
   END_TRANSITION
   STEP CheckRingExist:   // S117, max time T#10S, warning time T#7S
   END_STEP
   TRANSITION Trans117 FROM CheckRingExist TO "B-PressFitting-01GripperCylinderToHP"   // T117
      := TRUE;
   END_TRANSITION
   STEP "Status Alarm":   // S118, max time T#10S, warning time T#7S
          S1  S    "ST10_DeviceError".B.B2Press.StatusError
   END_STEP
   TRANSITION Trans120 FROM "Status Alarm" TO CheckPressGripStatus   // T120, jump
      := #iSysInface.Reset;
   END_TRANSITION
   STEP "B-PressFitting-01GripperCylinderToWP":   // S119, max time T#10S, warning time T#7S
              R    "ST10Cylinder".Cy[7].Inout.AutoGoHome
              S    "ST10Cylinder".Cy[7].Inout.AutoGoWork
   END_STEP
   TRANSITION Trans766 FROM "B-PressFitting-01GripperCylinderToWP" TO PressProgram   // T118
      := "ST10Cylinder".Cy[7].In.WorkPositionSensor AND NOT "ST10Cylinder".Cy[7].In.HomePositionSensor;
   END_TRANSITION
   STEP "B-PressFitting-01CylinderToHP":   // S120, max time T#10S, warning time T#7S
              S    "ST10Cylinder".Cy[8].Inout.AutoGoHome
              R    "ST10Cylinder".Cy[8].Inout.AutoGoWork
   END_STEP
   TRANSITION Trans767 FROM "B-PressFitting-01CylinderToHP" TO S10_InitialFinish   // T121
      := NOT "ST10Cylinder".Cy[8].In.WorkPositionSensor AND "ST10Cylinder".Cy[8].In.HomePositionSensor;
   END_TRANSITION

   // sequencer 2: S100-S199 等待到位 / S100-S149 CheckPartStatus
   STEP "Wait  robot finish task":   // S130, max time T#10S, warning time T#7S
   END_STEP
   TRANSITION Trans146 FROM "Wait  robot finish task" TO "RobotLeavePress Area"   // T146
      := "KukaRobot2_CtrlDB".sROBtoPLC.User.Cycle.DO274_PressPutPart1Finish;
   END_TRANSITION
   STEP CheckMachineStatus:   // S102, max time T#10S, warning time T#7S
   END_STEP
   TRANSITION Trans266 FROM CheckMachineStatus TO "Normal mode"   // T102
      := TRUE;
   END_TRANSITION
   STEP "Normal mode":   // S103, max time T#10S, warning time T#7S
   END_STEP
   TRANSITION Trans11 FROM "Normal mode" TO "ProcessStart,CTStart"   // T103
      := TRUE;
   END_TRANSITION
   STEP ProcessStart:   // S100, max time T#10S, warning time T#7S
      // 自动等待开始运行
              R    #ioPM_Inface.InitialRun
              R    #ioPM_Inface.ProcessComplete
              S    #ioPM_Inface.ProcessStart
              S    #ioPM_Inface.InitialOK
              S    #ioPM_Inface.WaitRunning
          S1  N    #ioPM_Inface.ProcessResult:=0
              R    "ST10_GeneralData".FlowControl_Handshake[14].Start
              R    "ST10_GeneralData".FlowControl_Handshake[14].Done
   END_STEP
   TRANSITION Trans200 FROM ProcessStart TO "Determine product status"   // T100
      := NOT #ioPM_Inface.AlarmCycleStop AND #ioPM_Inface.Running AND NOT #iSysInface.Auto.RunningOver AND (NOT #iSysInface.Auto.OneCycleMode OR (#iSysInface.Auto.OneCycleMode AND #ioPM_Inface.TriggerOneCycle));
   END_TRANSITION
   STEP "ProcessStart,CTStart":   // S104, max time T#10S, warning time T#7S
   END_STEP
   TRANSITION Trans249 FROM "ProcessStart,CTStart" TO "Request robot putShaft"   // T104
      := #"ProcessStart,CTStart".T > t#100MS;
   END_TRANSITION
   STEP "Process FInish":   // S237, max time T#10S, warning time T#7S
   END_STEP
   TRANSITION Trans250 FROM "Process FInish" TO "MES  Check   In"   // T249, jump
      := TRUE;
   END_TRANSITION
   STEP "Request robot putShaft":   // S112, max time T#10S, warning time T#7S
              N    "AutoProcessControl".B_Press_2.Robot2PutPrimit
   END_STEP
   TRANSITION Trans283 FROM "Request robot putShaft" TO "Wait  robot finish task"   // T112
      := "KukaRobot2_CtrlDB".sROBtoPLC.User.Cycle.DO273_PressPutPart1Inside AND NOT "KukaRobot2_CtrlDB".sROBtoPLC.User.Cycle.DO274_PressPutPart1Finish;
   END_TRANSITION
   STEP PutRing:   // S127, max time T#10S, warning time T#7S
   END_STEP
   TRANSITION Trans125 FROM PutRing TO "Request robot putRing"   // T125
      := TRUE;
   END_TRANSITION
   STEP PartCheck:   // S238, max time T#10S, warning time T#7S
   END_STEP
   TRANSITION Trans252 FROM PartCheck TO PutRing   // T251
      := ("AutoProcessData".B_Press2.PartStatus = 399) AND #TON[0].Q;
   END_TRANSITION
   TRANSITION Trans263 FROM PartCheck TO ProductCheckAlarm   // T259
      := ("AutoProcessData".B_Press2.PartStatus = 399) AND "iB-PressFitting-02ShaftDetection" AND #TOF[1].Q AND (#PartCheck.T > t#1500MS);
   END_TRANSITION
   STEP "Determine product status":   // S101, max time T#10S, warning time T#7S
              N    "MES_CHeck_DB".Station_7.CheckStep:=0
              N    "MES_CHeck_DB".Station_7.ResultStep:=0
   END_STEP
   TRANSITION Empty FROM "Determine product status" TO NoPart   // T101
      := NOT "iB-PressFitting-02ShaftDetection" AND (NOT "iB-PressFitting-02DownRingDetection" OR NOT "AlwaysFALSE") AND ("AutoProcessData".B_Press2.PartStatus = 0) AND (#"Determine product status".T > t#1000MS);
   END_TRANSITION
   TRANSITION HavePart FROM "Determine product status" TO ShaftOK   // T139
      := #TON[0].Q AND ("AutoProcessData".B_Press2.PartStatus = 399);
   END_TRANSITION
   TRANSITION Alarm FROM "Determine product status" TO StatusAlarm   // T710
      := (((#TON[0].Q OR ("AlwaysFALSE" AND #TON[2].Q)) AND ("AutoProcessData".B_Press2.PartStatus = 0)) OR (NOT "iB-PressFitting-02ShaftDetection" AND (NOT "iB-PressFitting-02DownRingDetection" OR NOT "AlwaysFALSE") AND ("AutoProcessData".B_Press2.PartStatus <> 0))) AND (#"Determine product status".T > t#1500MS);
   END_TRANSITION
   TRANSITION Trans21 FROM "Determine product status" TO ShaftAndRingOK   // T18
      := #TON[0].Q AND (#TON[2].Q OR NOT "AlwaysFALSE") AND ("AutoProcessData".B_Press2.PartStatus = 420);
   END_TRANSITION
   TRANSITION Trans22 FROM "Determine product status" TO "Press NG"   // T19
      := ("AutoProcessData".B_Press2.PartStatus = 450) OR ("AutoProcessData".B_Press2.PartStatus = 455);
   END_TRANSITION
   TRANSITION Trans23 FROM "Determine product status" TO MES   // T20
      := "AutoProcessData".B_Press2.PartStatus = 480;
   END_TRANSITION
   TRANSITION Trans29 FROM "Determine product status" TO MESOK   // T24
      := "AutoProcessData".B_Press2.PartStatus = 499;
   END_TRANSITION
   TRANSITION Trans138 FROM "Determine product status" TO MES_1NG   // T137
      := ("AutoProcessData".B_Press2.PartStatus = 451) OR ("AutoProcessData".B_Press2.PartStatus = 452);
   END_TRANSITION
   STEP ShaftOK:   // S125, max time T#10S, warning time T#7S
   END_STEP
   TRANSITION Trans303 FROM ShaftOK TO PutRing   // T140, jump
      := TRUE;
   END_TRANSITION
   STEP StatusAlarm:   // S126, max time T#10S, warning time T#7S
          S1  S    "ST10_DeviceError".B.B2Press.StatusError
   END_STEP
   TRANSITION Trans304 FROM StatusAlarm TO "Determine product status"   // T141, jump
      := #iSysInface.Reset;
   END_TRANSITION
   STEP NoPart:   // S129, max time T#10S, warning time T#7S
   END_STEP
   TRANSITION Trans145 FROM NoPart TO CheckMachineStatus   // T145
      := TRUE;
   END_TRANSITION
   STEP ShaftAndRingOK:   // S16, max time T#10S, warning time T#7S
   END_STEP
   TRANSITION Trans24 FROM ShaftAndRingOK TO "Process FInish"   // T21, jump
      := TRUE;
   END_TRANSITION
   STEP "Press NG":   // S17, max time T#10S, warning time T#7S
   END_STEP
   TRANSITION Trans25 FROM "Press NG" TO "ProcessFInish 1"   // T22, jump
      := TRUE;
   END_TRANSITION
   STEP MES:   // S18, max time T#10S, warning time T#7S
   END_STEP
   TRANSITION Trans28 FROM MES TO "ProcessFInish 1"   // T23, jump
      := TRUE;
   END_TRANSITION
   STEP MESOK:   // S19, max time T#10S, warning time T#7S
   END_STEP
   TRANSITION Trans30 FROM MESOK TO RobotPick   // T25, jump
      := TRUE;
   END_TRANSITION
   STEP "Wait  robot finish task_1":   // S134, max time T#10S, warning time T#7S
   END_STEP
   TRANSITION Trans148 FROM "Wait  robot finish task_1" TO PartStatus   // T147
      := "KukaRobot3_CtrlDB".sROBtoPLC.User.Cycle.DO278_PressPutRingFinish;
   END_TRANSITION
   STEP "Request robot putRing":   // S113, max time T#10S, warning time T#7S
              N    "AutoProcessControl".B_Press_2.Robot3PutRingPrimit
   END_STEP
   TRANSITION Trans284 FROM "Request robot putRing" TO "Wait  robot finish task_1"   // T113
      := "KukaRobot3_CtrlDB".sROBtoPLC.User.Cycle.DO277_PressPutRingInside AND NOT "KukaRobot3_CtrlDB".sROBtoPLC.User.Cycle.DO278_PressPutRingFinish;
   END_TRANSITION
   STEP "Part Check":   // S239, max time T#10S, warning time T#7S
   END_STEP
   TRANSITION Trans262 FROM "Part Check" TO "Process FInish"   // T252
      := ("AutoProcessData".B_Press2.PartStatus = 420) AND #TON[0].Q;
   END_TRANSITION
   TRANSITION Trans267 FROM "Part Check" TO ProductCheckAlarm_1   // T261
      := NOT "AlwaysTRUE";
   END_TRANSITION
   STEP ProductCheckAlarm:   // S240, max time T#10S, warning time T#7S
          S1  S    "ST10_DeviceError".B.B2Press.ShaftSensorCheckError
   END_STEP
   TRANSITION Trans265 FROM ProductCheckAlarm TO PartCheck   // T260, jump
      := #iSysInface.Reset;
   END_TRANSITION
   STEP ProductCheckAlarm_1:   // S241, max time T#10S, warning time T#7S
          S1  S    "ST10_DeviceError".B.B2Press.RingSensorCheckError
   END_STEP
   TRANSITION Trans269 FROM ProductCheckAlarm_1 TO "Part Check"   // T262, jump
      := #iSysInface.Reset;
   END_TRANSITION
   STEP RobotLeavePressArea:   // S121, max time T#10S, warning time T#7S
   END_STEP
   TRANSITION Trans236 FROM RobotLeavePressArea TO "Part Check"   // T122
      := "KukaRobot3_CtrlDB".sROBtoPLC.User.Home.DO177_PressPut1Area AND "KukaRobot3_CtrlDB".sROBtoPLC.User.Home.DO178_Robot2Area;
   END_TRANSITION
   STEP "RobotLeavePress Area":   // S115, max time T#10S, warning time T#7S
   END_STEP
   TRANSITION Trans199 FROM "RobotLeavePress Area" TO PartCheck   // T115
      := TRUE;
   END_TRANSITION
   STEP PartStatus:   // S123, max time T#10S, warning time T#7S
   END_STEP
   TRANSITION Trans124 FROM PartStatus TO RobotLeavePressArea   // T124
      := "AutoProcessData".B_Press2.PartStatus = 420;
   END_TRANSITION
   STEP MES_1NG:   // S25, max time T#10S, warning time T#7S
   END_STEP
   TRANSITION Trans36 FROM MES_1NG TO RobotPick   // T32, jump
      := TRUE;
   END_TRANSITION

   // sequencer 3: S150-S199 MES Check In
   STEP "MES  Check   In":   // S150, max time T#10S, warning time T#7S
   END_STEP
   TRANSITION Trans139 FROM "MES  Check   In" TO Bypass   // T150
      := TRUE;
   END_TRANSITION
   STEP MESOverTime_1:   // S312, max time T#10S, warning time T#7S
              S    "ST10_DeviceError".MES_Error.CheckInCompOverTime_7
   END_STEP
   TRANSITION Trans318 FROM MESOverTime_1 TO Bypass   // T320, jump
      := #iSysInface.Reset;
   END_TRANSITION
   STEP "MES Check NG_2":   // S313, max time T#10S, warning time T#7S
              N    "AutoProcessData".B_Press2.PartStatus:=451
   END_STEP
   TRANSITION Trans311 FROM "MES Check NG_2" TO RobotPick   // T315, jump
      := "AutoProcessData".B_Press2.PartStatus = 451;
   END_TRANSITION
   STEP ResetMesCheckRequest:   // S301, max time T#10S, warning time T#7S
              R    "PLCtoMES"."PLC.Load_Station7ChickInReq"
              R    "MEStoPLC"."MES.Load_Station7PartOK"
              R    "MEStoPLC"."MES.Load_Station7PartNG"
              R    "MEStoPLC"."MES.Load_Station7ReqMesDone"
   END_STEP
   TRANSITION Trans259 FROM ResetMesCheckRequest TO "Prepare MES CheckData"   // T301
      := NOT "PLCtoMES"."PLC.Load_Station7ChickInReq" AND NOT "MEStoPLC"."MES.Load_Station7PartOK" AND NOT "MEStoPLC"."MES.Load_Station7PartNG" AND NOT "MEStoPLC"."MES.Load_Station7ReqMesDone";
   END_TRANSITION
   STEP "Prepare MES CheckData":   // S305, max time T#10S, warning time T#7S
   END_STEP
   TRANSITION Trans26 FROM "Prepare MES CheckData" TO MesCheckIn_1   // T305
      := #"Prepare MES CheckData".T > t#200MS;
   END_TRANSITION
   STEP MesCheckIn_1:   // S314, max time T#10S, warning time T#7S
              N    "PLCtoMES"."PLC.Load_Station7ChickInReq"
   END_STEP
   TRANSITION Trans313 FROM MesCheckIn_1 TO Step313   // T317
      := "MEStoPLC"."MES.Load_Station7PartOK" AND NOT "MEStoPLC"."MES.Load_Station7PartNG" AND "MEStoPLC"."MES.Load_Station7ReqMesDone";
   END_TRANSITION
   TRANSITION Trans312 FROM MesCheckIn_1 TO "MES Check NG_2"   // T316
      := NOT "MEStoPLC"."MES.Load_Station7PartOK" AND "MEStoPLC"."MES.Load_Station7PartNG" AND "MEStoPLC"."MES.Load_Station7ReqMesDone";
   END_TRANSITION
   TRANSITION Trans302 FROM MesCheckIn_1 TO MESOverTime_1   // T302
      := #MesCheckIn_1.T > t#10S;
   END_TRANSITION
   STEP CheckFinish_1:   // S315, max time T#10S, warning time T#7S
   END_STEP
   TRANSITION Trans316 FROM CheckFinish_1 TO Pressing   // T311, jump
      := TRUE;
   END_TRANSITION
   STEP Bypass:   // S316, max time T#10S, warning time T#7S
   END_STEP
   TRANSITION Online FROM Bypass TO ResetMesCheckRequest   // T318
      := NOT "Station_Sys".Cmd.OnOffLine;
   END_TRANSITION
   TRANSITION Trans317 FROM Bypass TO CheckFinish_1   // T319
      := "Station_Sys".Cmd.OnOffLine;
   END_TRANSITION
   STEP Step313:   // S317, max time T#10S, warning time T#7S
   END_STEP
   TRANSITION Trans319 FROM Step313 TO CheckFinish_1   // T321
      := TRUE;
   END_TRANSITION

   // sequencer 4: S200-S299Pressing
   STEP Pressing:   // S200, max time T#10S, warning time T#7S
   END_STEP
   TRANSITION Trans147 FROM Pressing TO CheckPressReady   // T200
      := TRUE;
   END_TRANSITION
   STEP WaitPressFinish:   // S201, max time T#10S, warning time T#7S
   END_STEP
   TRANSITION Trans201 FROM WaitPressFinish TO ResetPressStart   // T201
      := (NOT "DB_maXYmosNC2".InputMessages.StatusBits."RUN-SEQUENCE" AND "DB_maXYmosNC2".InputMessages.StatusBits."SEQUENCE-END") OR "Tag_34";
   END_TRANSITION
   STEP ResultNGData:   // S146, max time T#10S, warning time T#7S
              N    "AutoProcessData".B_Press2.PartStatus:=455
   END_STEP
   TRANSITION Trans137 FROM ResultNGData TO Step147   // T143
      := "AutoProcessData".B_Press2.PartStatus = 455;
   END_TRANSITION
   STEP PartStatus_1:   // S137, max time T#10S, warning time T#7S
              N    "AutoProcessData".B_Press2.PartStatus:=450
   END_STEP
   TRANSITION Trans128 FROM PartStatus_1 TO WaitPressFinish   // T128
      := TRUE;
   END_TRANSITION
   STEP CheckPressSensor:   // S138, max time T#10S, warning time T#7S
   END_STEP
   TRANSITION Trans129 FROM CheckPressSensor TO PartStatus_1   // T129
      := "DB_maXYmosNC2".InputMessages.StatusBits."O-UNI" = 1;
   END_TRANSITION
   STEP ResetPressStart:   // S142, max time T#10S, warning time T#7S
              R    "DB_maXYmosNC2".StartCycle
   END_STEP
   TRANSITION Trans133 FROM ResetPressStart TO CheckPressResult   // T133
      := TRUE;
   END_TRANSITION
   STEP CheckPressProgram:   // S139, max time T#10S, warning time T#7S
              N    "AutoProcessData".B_Press2.Press2Program:="DB_maXYmosNC2".InputMessages.StatusBits.MP
   END_STEP
   TRANSITION Trans130 FROM CheckPressProgram TO StartCycle   // T130
      := "DB_maXYmosNC2".InputMessages.StatusBits.MP <> 0;
   END_TRANSITION
   STEP StartCycle:   // S141, max time T#10S, warning time T#7S
              S    "DB_maXYmosNC2".StartCycle
   END_STEP
   TRANSITION Trans132 FROM StartCycle TO CheckPressSensor   // T132
      := ("DB_maXYmosNC2".InputMessages.StatusBits.UNI = 0) AND NOT "DB_maXYmosNC2".oRdyCmd AND "DB_maXYmosNC2".oRunSeq;
   END_TRANSITION
   STEP CheckPressReady:   // S208, max time T#10S, warning time T#7S
              R    "DB_maXYmosNC2".StartCycle
   END_STEP
   TRANSITION Trans211 FROM CheckPressReady TO CheckPressProgram   // T211
      := "DB_maXYmosNC2".InputMessages.StatusBits.READY AND "DB_maXYmosNC2".InputMessages.StatusBits."DRIVE-ENABLED" AND "ProcessData_1"."OP40.3".Kistler_Interlock;
   END_TRANSITION
   STEP "ProcessFInish 1":   // S143, max time T#10S, warning time T#7S
   END_STEP
   TRANSITION Trans134 FROM "ProcessFInish 1" TO Step400   // T134, jump
      := TRUE;
   END_TRANSITION
   STEP ResultOKData:   // S145, max time T#10S, warning time T#7S
              N    "AutoProcessData".B_Press2.PartStatus:=480
   END_STEP
   TRANSITION Trans136 FROM ResultOKData TO Step147   // T136
      := TRUE;
   END_TRANSITION
   STEP CheckPressResult:   // S144, max time T#10S, warning time T#7S
   END_STEP
   TRANSITION Trans135 FROM CheckPressResult TO ResultOKData   // T135
      := "DB_maXYmosNC2".oCycleOK AND NOT "DB_maXYmosNC2".oCycleNOK;
   END_TRANSITION
   TRANSITION Trans142 FROM CheckPressResult TO ResultNGData   // T142
      := NOT "DB_maXYmosNC2".oCycleOK AND "DB_maXYmosNC2".oCycleNOK;
   END_TRANSITION
   STEP Step147:   // S147, max time T#10S, warning time T#7S
   END_STEP
   TRANSITION Trans144 FROM Step147 TO "ProcessFInish 1"   // T144
      := TRUE;
   END_TRANSITION

   // sequencer 5: S400-S499OK&NG数据处理 / S400-S499OK&NG Status Count
   STEP Step400:   // S400, max time T#10S, warning time T#7S
   END_STEP
   TRANSITION Trans224 FROM Step400 TO JudgeStatus   // T400
      := TRUE;
   END_TRANSITION
   STEP JudgeStatus:   // S401, max time T#10S, warning time T#7S
              N    #ioPM_Inface.ProcessResult:=0
   END_STEP
   TRANSITION OK FROM JudgeStatus TO OKCount   // T401
      := #ioStatus = 190;
   END_TRANSITION
   TRANSITION NG FROM JudgeStatus TO NGCount   // T404
      := #ioStatus <> 190;
   END_TRANSITION
   STEP OKCount:   // S402, max time T#10S, warning time T#7S
              N    #ioPM_Inface.ProcessResult:=400
   END_STEP
   TRANSITION Trans403 FROM OKCount TO ProcessFinish   // T402
      := TRUE;
   END_TRANSITION
   STEP NGCount:   // S404, max time T#10S, warning time T#7S
              N    #ioPM_Inface.ProcessResult:=#ioStatus
   END_STEP
   TRANSITION Trans404 FROM NGCount TO ProcessFinish   // T405
      := TRUE;
   END_TRANSITION
   STEP ProcessFinish:   // S403, max time T#10S, warning time T#7S
   END_STEP
   TRANSITION Trans405 FROM ProcessFinish TO "MES Result"   // T403, jump
      := TRUE;
   END_TRANSITION

   // sequencer 6: S500-S599 MES上传RFID写入 / S500-S599 MES Result
   STEP "MES Result":   // S500, max time T#10S, warning time T#7S
   END_STEP
   TRANSITION Trans407 FROM "MES Result" TO Bypass_1   // T500
      := TRUE;
   END_TRANSITION
   STEP "MES Check Finish":   // S515, max time T#10S, warning time T#7S
   END_STEP
   TRANSITION Trans619 FROM "MES Check Finish" TO RobotPick   // T515, jump
      := TRUE;
   END_TRANSITION
   STEP "MES Result OK_1":   // S405, max time T#10S, warning time T#7S
              N    "AutoProcessData".B_Press2.PartStatus:=499
   END_STEP
   TRANSITION Trans321 FROM "MES Result OK_1" TO "MES Check Finish"   // T399
      := "AutoProcessData".B_Press2.PartStatus = 499;
   END_TRANSITION
   STEP "MES Check NG_3":   // S318, max time T#10S, warning time T#7S
              N    "AutoProcessData".B_Press2.PartStatus:=452
   END_STEP
   TRANSITION Trans322 FROM "MES Check NG_3" TO "MES Check Finish"   // T324
      := "AutoProcessData".B_Press2.PartStatus = 452;
   END_TRANSITION
   STEP MesCheckResult_1:   // S309, max time T#10S, warning time T#7S
              N    "PLCtoMES"."PLC.Unload_Station7DataSaveReq"
   END_STEP
   TRANSITION Trans320 FROM MesCheckResult_1 TO "MES Result OK_1"   // T323
      := "MEStoPLC"."MES.Unload_ResultsStored7OK" AND NOT "MEStoPLC"."MES.Unload_ResultsStored7NG" AND "MEStoPLC"."MES.Unload_ResultsStored7ReqMesDone" AND ("AutoProcessData".B_Press2.PartStatus <> 450) AND ("AutoProcessData".B_Press2.PartStatus <> 455);
   END_TRANSITION
   TRANSITION Trans315 FROM MesCheckResult_1 TO "MES Check NG_3"   // T322
      := NOT "MEStoPLC"."MES.Unload_ResultsStored7OK" AND "MEStoPLC"."MES.Unload_ResultsStored7NG" AND "MEStoPLC"."MES.Unload_ResultsStored7ReqMesDone";
   END_TRANSITION
   TRANSITION Trans324 FROM MesCheckResult_1 TO MESOverTime   // T328
      := NOT "MEStoPLC"."MES.Load_Station7ReqMesDone" AND (#MesCheckResult_1.T > t#10S);
   END_TRANSITION
   TRANSITION Trans140 FROM MesCheckResult_1 TO "MES Check Finish"   // T138
      := (("AutoProcessData".B_Press2.PartStatus = 450) OR ("AutoProcessData".B_Press2.PartStatus = 455)) AND "MEStoPLC"."MES.Unload_ResultsStored7OK" AND NOT "MEStoPLC"."MES.Unload_ResultsStored7NG" AND "MEStoPLC"."MES.Unload_ResultsStored7ReqMesDone";
   END_TRANSITION
   STEP Bypass_1:   // S319, max time T#10S, warning time T#7S
   END_STEP
   TRANSITION Online_1 FROM Bypass_1 TO ResetMesUnloadRequest_1   // T325
      := NOT "Station_Sys".Cmd.OnOffLine;
   END_TRANSITION
   TRANSITION Trans323 FROM Bypass_1 TO ok_1   // T327
      := "Station_Sys".Cmd.OnOffLine;
   END_TRANSITION
   STEP ResetMesUnloadRequest_1:   // S302, max time T#10S, warning time T#7S
              R    "PLCtoMES"."PLC.Unload_Station7DataSaveReq"
              R    "MEStoPLC"."MES.Unload_ResultsStored7OK"
              R    "MEStoPLC"."MES.Unload_ResultsStored7NG"
              R    "MEStoPLC"."MES.Unload_ResultsStored7ReqMesDone"
   END_STEP
   TRANSITION Trans260 FROM ResetMesUnloadRequest_1 TO "Prepare MES CheckData_1"   // T326
      := NOT "PLCtoMES"."PLC.Unload_Station7DataSaveReq" AND NOT "MEStoPLC"."MES.Unload_ResultsStored7OK" AND NOT "MEStoPLC"."MES.Unload_ResultsStored7NG" AND NOT "MEStoPLC"."MES.Unload_ResultsStored7ReqMesDone";
   END_TRANSITION
   STEP Step314:   // S320, max time T#10S, warning time T#7S
   END_STEP
   TRANSITION Trans327 FROM Step314 TO "MES Check Finish"   // T330
      := TRUE;
   END_TRANSITION
   STEP MESOverTime:   // S321, max time T#10S, warning time T#7S
              S    "ST10_DeviceError".MES_Error.CheckInResultOverTime_7
   END_STEP
   TRANSITION Trans326 FROM MESOverTime TO Bypass_1   // T329, jump
      := #iSysInface.Reset;
   END_TRANSITION
   STEP ok_1:   // S322, max time T#10S, warning time T#7S
      interlock C := "AutoProcessData".B_Press2.PartStatus = 480;
      (C)     N    "AutoProcessData".B_Press2.PartStatus:=499
   END_STEP
   TRANSITION Trans328 FROM ok_1 TO Step314   // T331
      := ("AutoProcessData".B_Press2.PartStatus = 499) OR ("Station_Sys".Cmd.OnOffLine AND ("AutoProcessData".B_Press2.PartStatus <> 450) AND ("AutoProcessData".B_Press2.PartStatus <> 455));
   END_TRANSITION
   STEP "Prepare MES CheckData_1":   // S307, max time T#10S, warning time T#7S
   END_STEP
   TRANSITION Trans16 FROM "Prepare MES CheckData_1" TO MesCheckResult_1   // T308
      := #"Prepare MES CheckData_1".T > t#300MS;
   END_TRANSITION

   // sequencer 7: S600-S699工件放行 / S600-S699 RobotPick
   STEP RobotPick:   // S600, max time T#10S, warning time T#7S
   END_STEP
   TRANSITION Trans600 FROM RobotPick TO PressProgram_1   // T600
      := TRUE;
   END_TRANSITION
   STEP ProcessFinsh:   // S605, max time T#10S, warning time T#7S: 正式使用时，需要激活复位空循环
              S    #ioPM_Inface.ProcessComplete
              R    #ioPM_Inface.ProcessStart
   END_STEP
   TRANSITION Trans699 FROM ProcessFinsh TO ProcessStart   // T605, jump
      := TRUE;
   END_TRANSITION
   STEP DataClear:   // S604, max time T#10S, warning time T#7S
          S1  N    #ioPM_Inface.ProcessResult:=0
          S1  N    #ioStatus:=0
   END_STEP
   TRANSITION Trans290 FROM DataClear TO ProcessFinsh   // T604
      := TRUE;
   END_TRANSITION
   STEP "Request robot pick":   // S408, max time T#10S, warning time T#7S
              N    "AutoProcessControl".B_Press_2.Robot3PickPrimit
   END_STEP
   TRANSITION Trans412 FROM "Request robot pick" TO "Wait robot finish task"   // T410
      := "KukaRobot3_CtrlDB".sROBtoPLC.User.Cycle.DO281_PressPickInside AND NOT "KukaRobot3_CtrlDB".sROBtoPLC.User.Cycle.DO282_PressPickFinish;
   END_TRANSITION
   STEP "Wait robot finish task":   // S131, max time T#10S, warning time T#7S
   END_STEP
   TRANSITION Trans257 FROM "Wait robot finish task" TO DataMove   // T256
      := "KukaRobot3_CtrlDB".sROBtoPLC.User.Cycle.DO282_PressPickFinish;
   END_TRANSITION
   STEP DataMove:   // S132, max time T#10S, warning time T#7S
   END_STEP
   TRANSITION Trans258 FROM DataMove TO "Wait robot in safety area"   // T257
      := TRUE;
   END_TRANSITION
   STEP "Wait robot in safety area":   // S133, max time T#10S, warning time T#7S
   END_STEP
   TRANSITION Trans261 FROM "Wait robot in safety area" TO DataClear   // T258
      := "KukaRobot3_CtrlDB".sROBtoPLC.User.Home.DO177_PressPut1Area AND "KukaRobot3_CtrlDB".sROBtoPLC.User.Home.DO178_Robot2Area;
   END_TRANSITION
   STEP PressProgram_1:   // S20, max time T#10S, warning time T#7S
      interlock C := NOT "ST10_GeneralData".FunctionDeSelect."B".FunctionDeSelected_TestPress375A1;
      (C)     N    "DB_maXYmosNC2".ProgNo:=1
   END_STEP
   TRANSITION Trans31 FROM PressProgram_1 TO "PressReady?_1"   // T27
      := TRUE;
   END_TRANSITION
   STEP PressHoming_1:   // S21, max time T#10S, warning time T#7S
              N    "DB_maXYmosNC2".Homing
   END_STEP
   TRANSITION Trans9 FROM PressHoming_1 TO Step15   // T26
      := "DB_maXYmosNC2".oInHomePos;
   END_TRANSITION
   STEP "PressReady?_1":   // S22, max time T#10S, warning time T#7S
   END_STEP
   TRANSITION Trans32 FROM "PressReady?_1" TO "PressHoming?_1"   // T28
      := "DB_maXYmosNC2".oReady AND "DB_maXYmosNC2".oRdyAmp;
   END_TRANSITION
   STEP "PressHoming?_1":   // S23, max time T#10S, warning time T#7S
   END_STEP
   TRANSITION Trans33 FROM "PressHoming?_1" TO PressHoming_1   // T29
      := NOT "DB_maXYmosNC2".oInHomePos;
   END_TRANSITION
   TRANSITION Trans34 FROM "PressHoming?_1" TO Step15   // T30
      := "DB_maXYmosNC2".oInHomePos;
   END_TRANSITION
   STEP Step15:   // S24, max time T#10S, warning time T#7S
   END_STEP
   TRANSITION Trans35 FROM Step15 TO "B-PressFitting-01CylinderToHP_1"   // T31
      := TRUE;
   END_TRANSITION
   STEP "B-PressFitting-01CylinderToHP_1":   // S140, max time T#10S, warning time T#7S
              S    "ST10Cylinder".Cy[8].Inout.AutoGoHome
              R    "ST10Cylinder".Cy[8].Inout.AutoGoWork
   END_STEP
   TRANSITION Trans768 FROM "B-PressFitting-01CylinderToHP_1" TO "Request robot pick"   // T131
      := NOT "ST10Cylinder".Cy[8].In.WorkPositionSensor AND "ST10Cylinder".Cy[8].In.HomePositionSensor;
   END_TRANSITION

   // permanent post-instructions
   NETWORK 1
      #ioPM_Inface.StepNum := #RT_DATA.S_DISPLAY;
   NETWORK 2
      IF #iSysInface.Reset THEN #AlarmID := 0; END_IF;
   NETWORK 3
      #TON[10].TON(IN := #工件放行中, PT := T#0.5S);
      IF #TON[10].Q THEN #工件放行中 := FALSE; END_IF;
END_FUNCTION_BLOCK

FUNCTION_BLOCK "ST10_Flow15_FRobot_3"   // FB1085, GRAPH
// stored: AcknowledgeErrorsRequired false, AutoNumber false, GraphVersion 6.0, InitialValuesAcquisition false, SetENOAutomatically false
   // inherited from GRAPH_BASE
   VAR_INPUT
      iSysInface : "RCS_SysComInterface_V1";
   END_VAR
   VAR_IN_OUT
      ioPM_Inface : "RCS_PMInterface_V1";
      ioStatus : Int;
   END_VAR
   VAR
      sCtrlMode { S7_SetPoint := 'True'} : "SysFlowCtrlGraph";
      sUpdMES_Data : Bool;   // 更新MES数据
      工件放行中 : Bool;
      前站站号 { ExternalAccessible := 'False'; ExternalVisible := 'False'; ExternalWritable := 'False'} : UInt;
      本站站号 { ExternalAccessible := 'False'; ExternalVisible := 'False'; ExternalWritable := 'False'} : UInt;
      弹窗Temp : Array[1..10] of Int;
      AlarmID : Int;
      TON { S7_SetPoint := 'True'} : Array[0..10] of TON_TIME;
      TOF { S7_SetPoint := 'True'} : Array[0..10] of TOF_TIME;
      sUP { S7_SetPoint := 'True'} : Array[0..10] of Bool;
      更新RFID完成 : Bool;
   END_VAR
   VAR_TEMP
      Tempresult : USInt;
      本站站号乘10 : UInt;
   END_VAR
   // // TON[0] : 托盘流入1托盘到位传感器
   // // TON[1] : 托盘流入1托盘到位传感器
   // // TON[2] : 托盘流入1产品有无传感器
   // // TON[3] : 托盘流入1产品有无传感器
   // // TON[4] : 托盘流入1姿态检测光电2
   // // TON[5] : 托盘流入1姿态检测光电3
   // // TON[0].Q : 托盘流入1托盘到位
   // // TON[1].Q : 托盘流入1托盘无
   // // TON[2].Q : 托盘流入1有产品
   // // TON[3].Q : 托盘流入1无产品
   // // TON[4].Q : 托盘流入1姿态检测光电2
   // // TON[5].Q : 托盘流入1姿态检测光电3
BEGIN
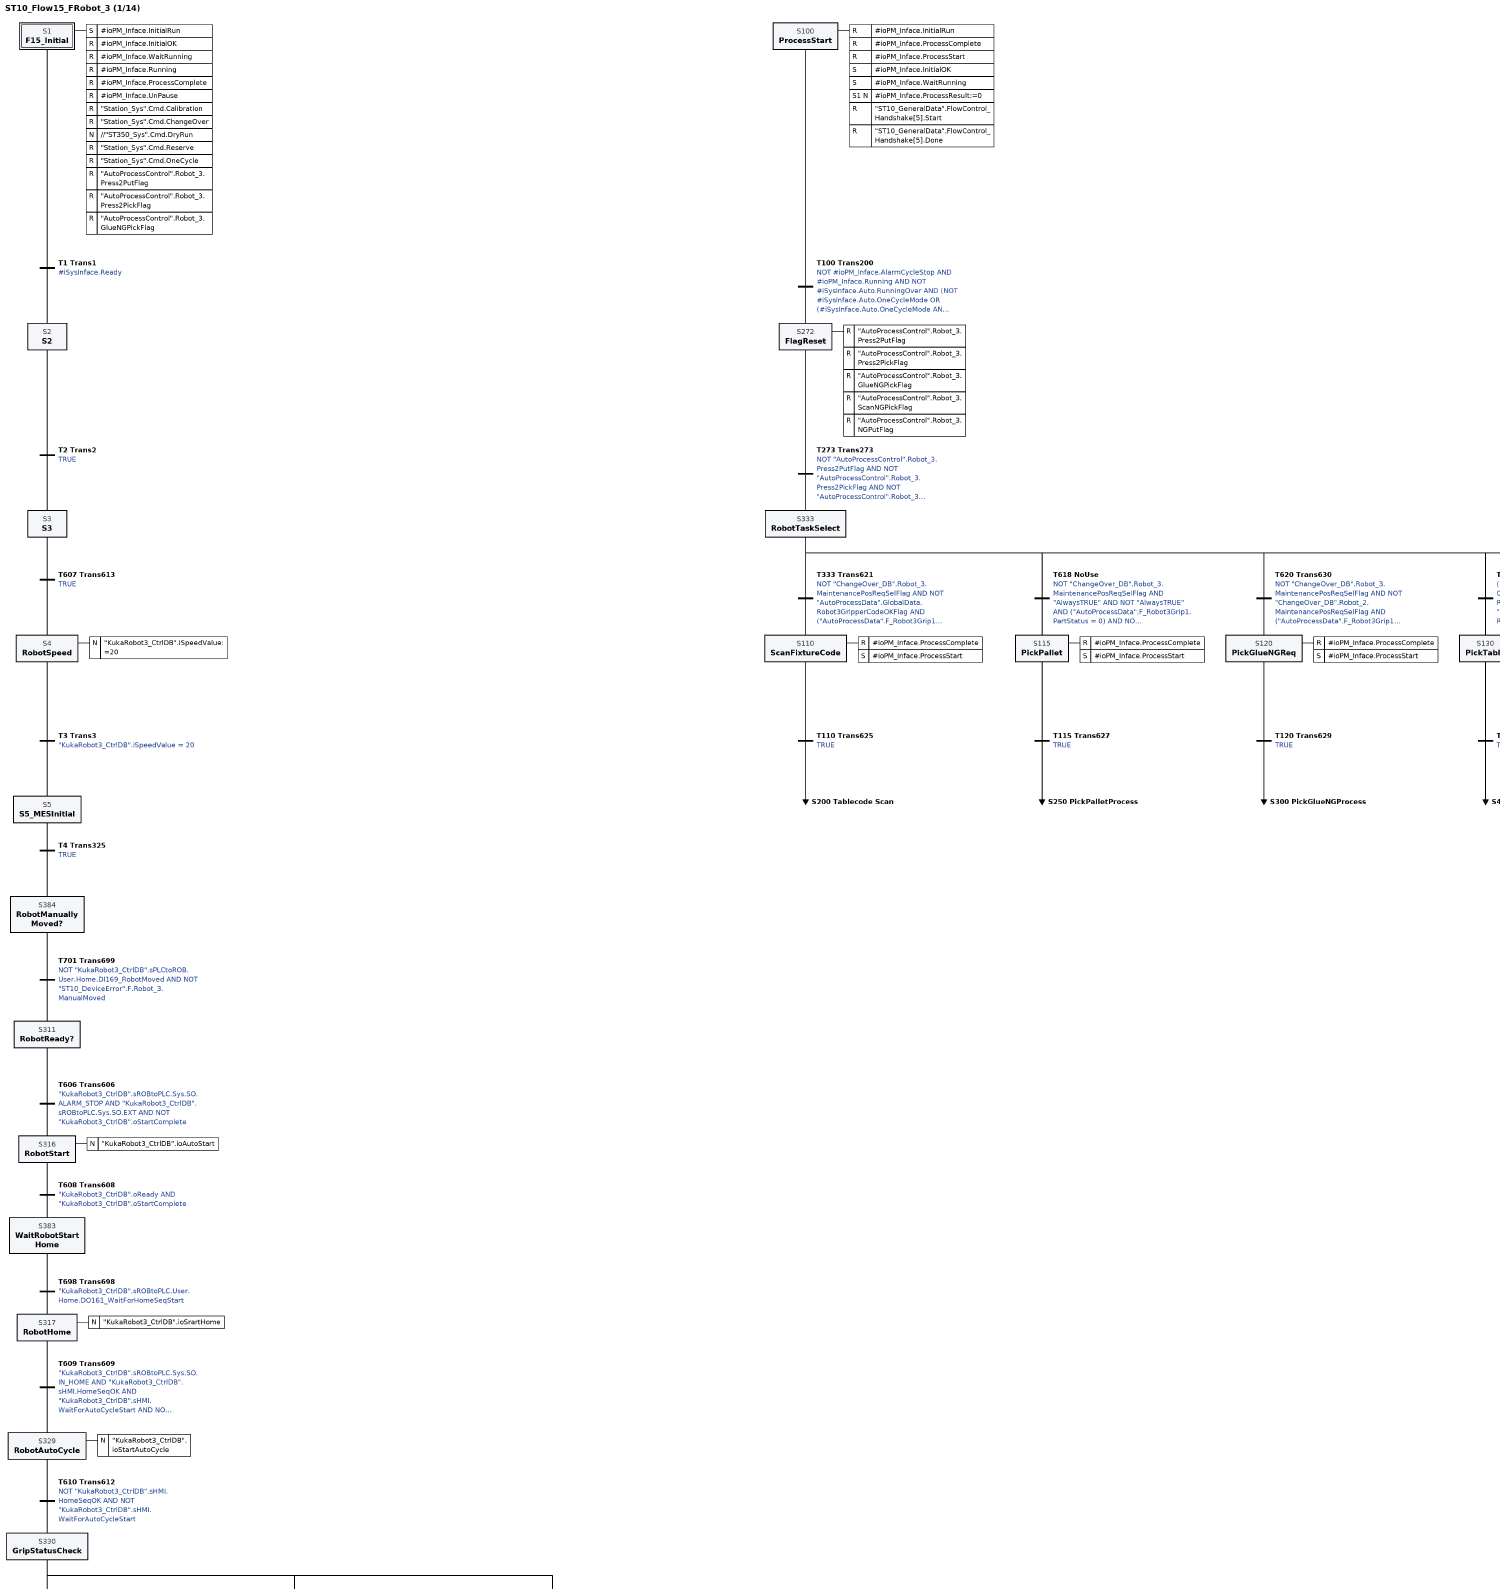
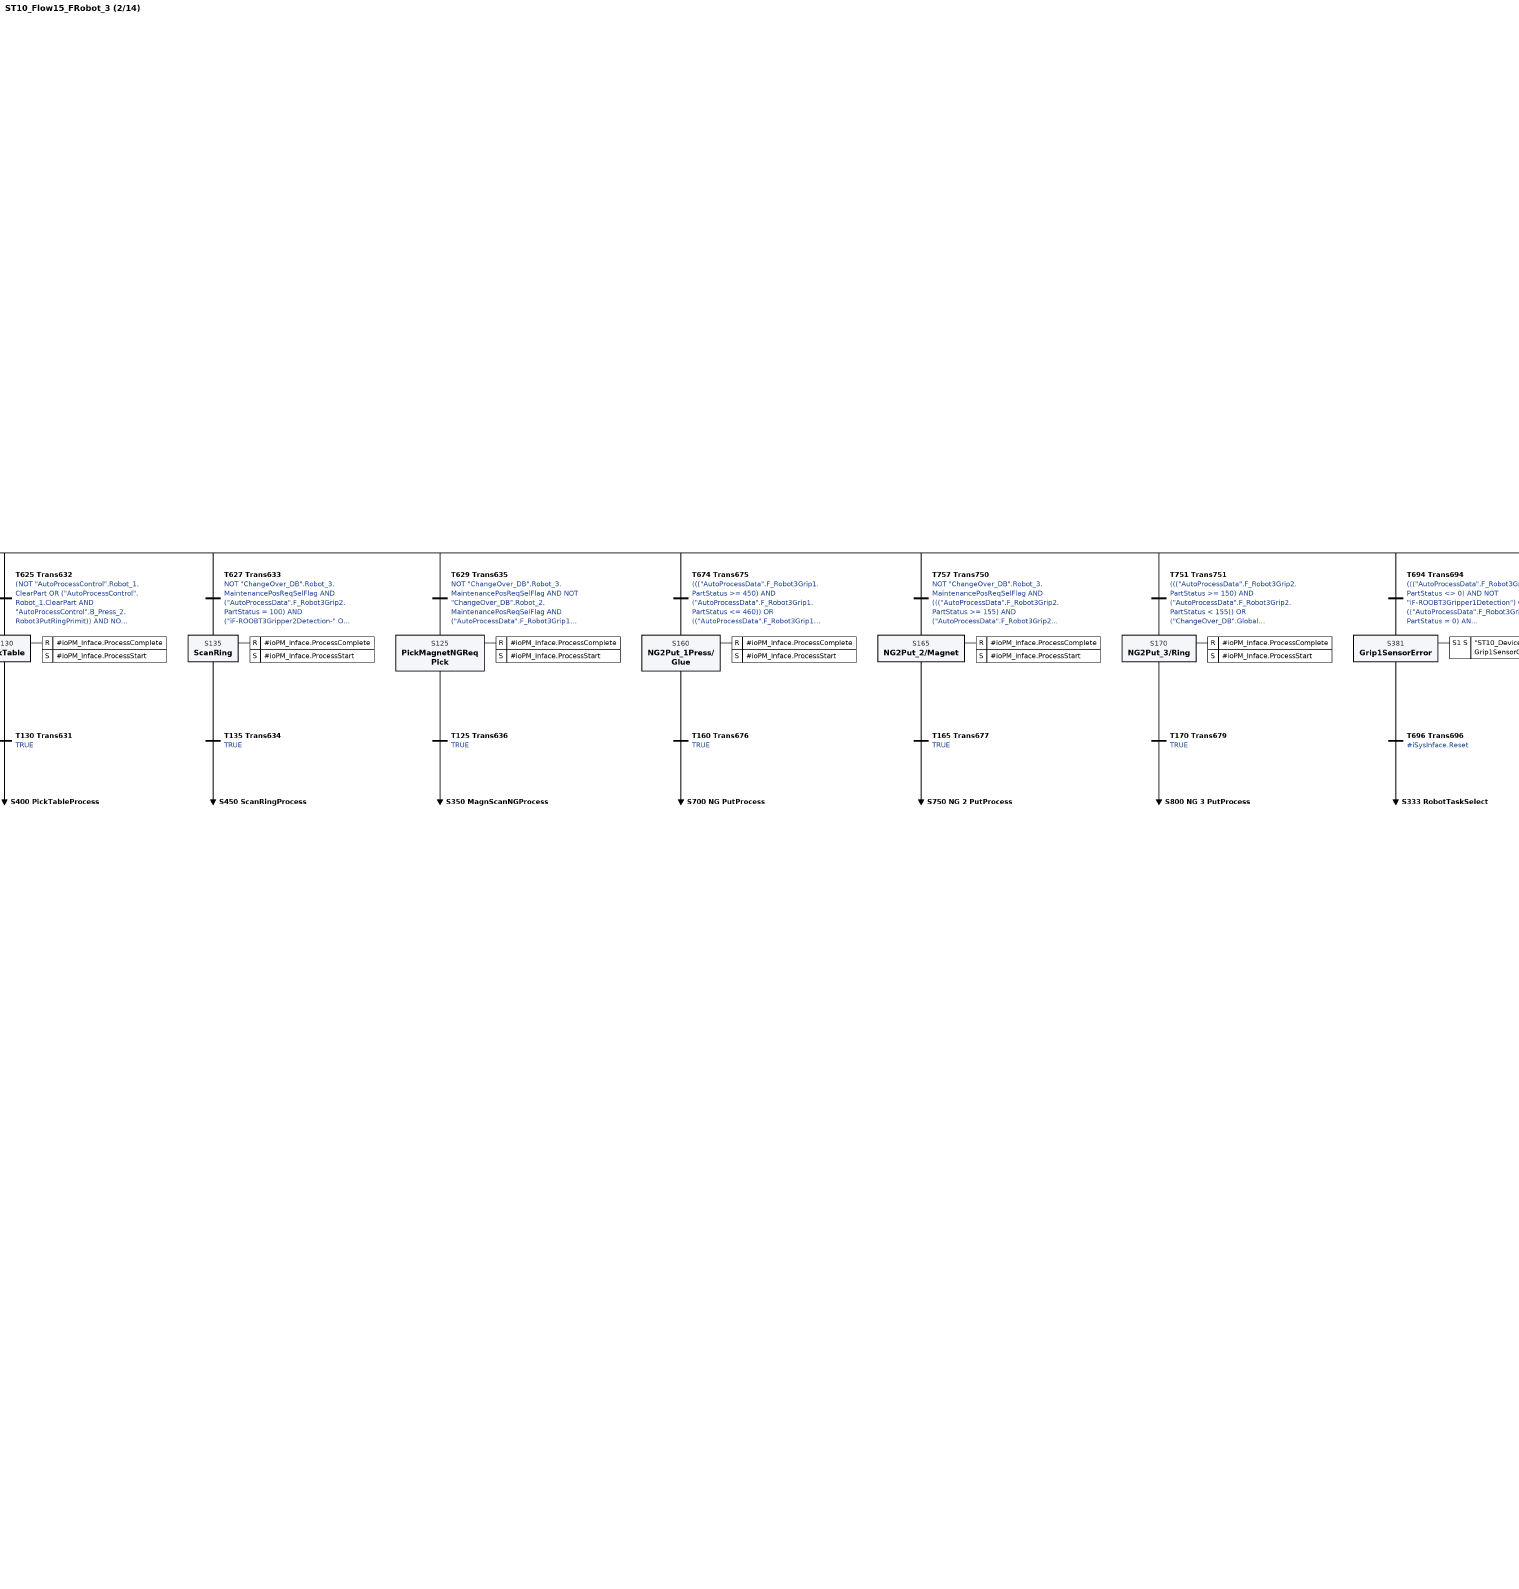
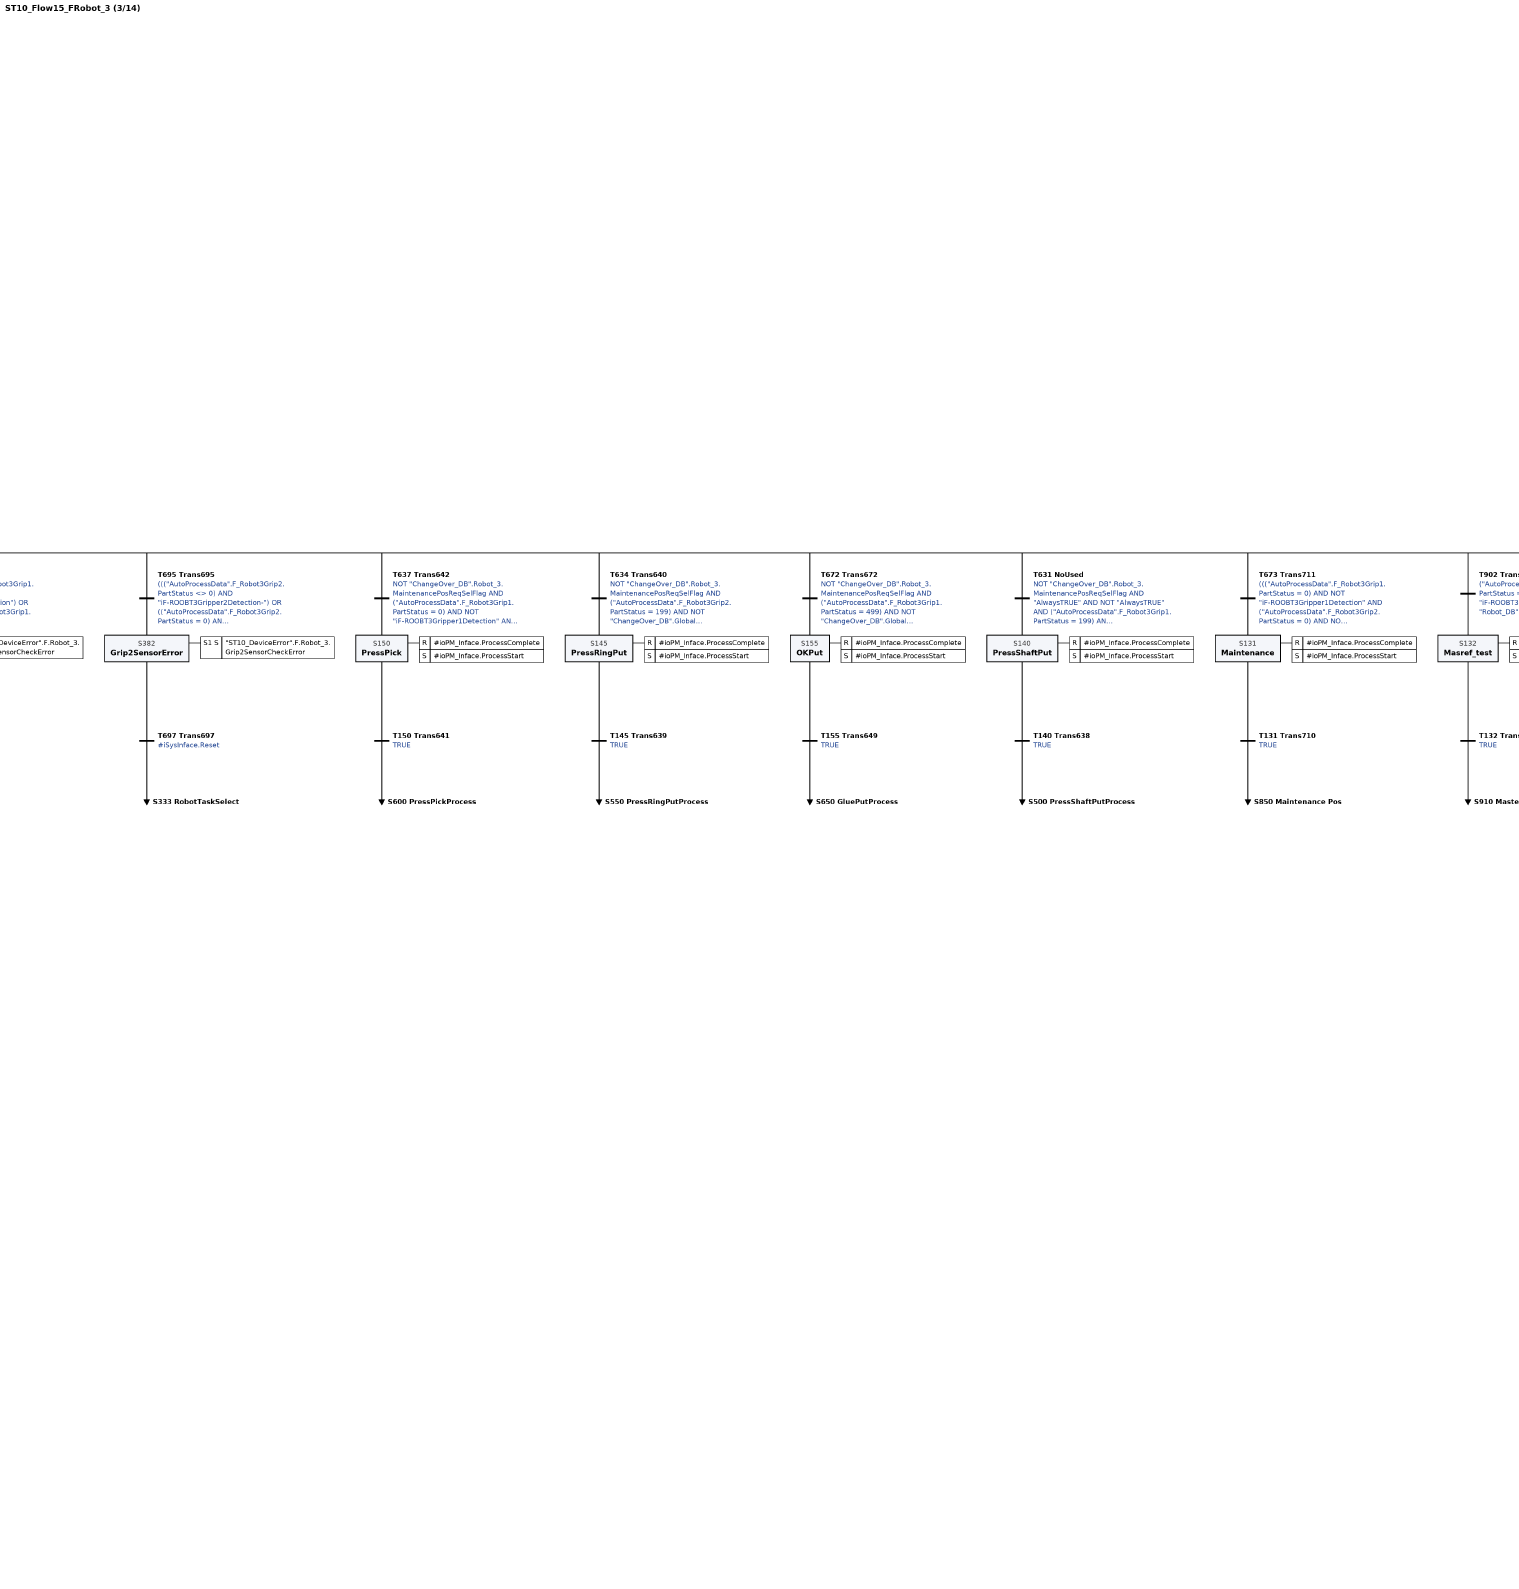
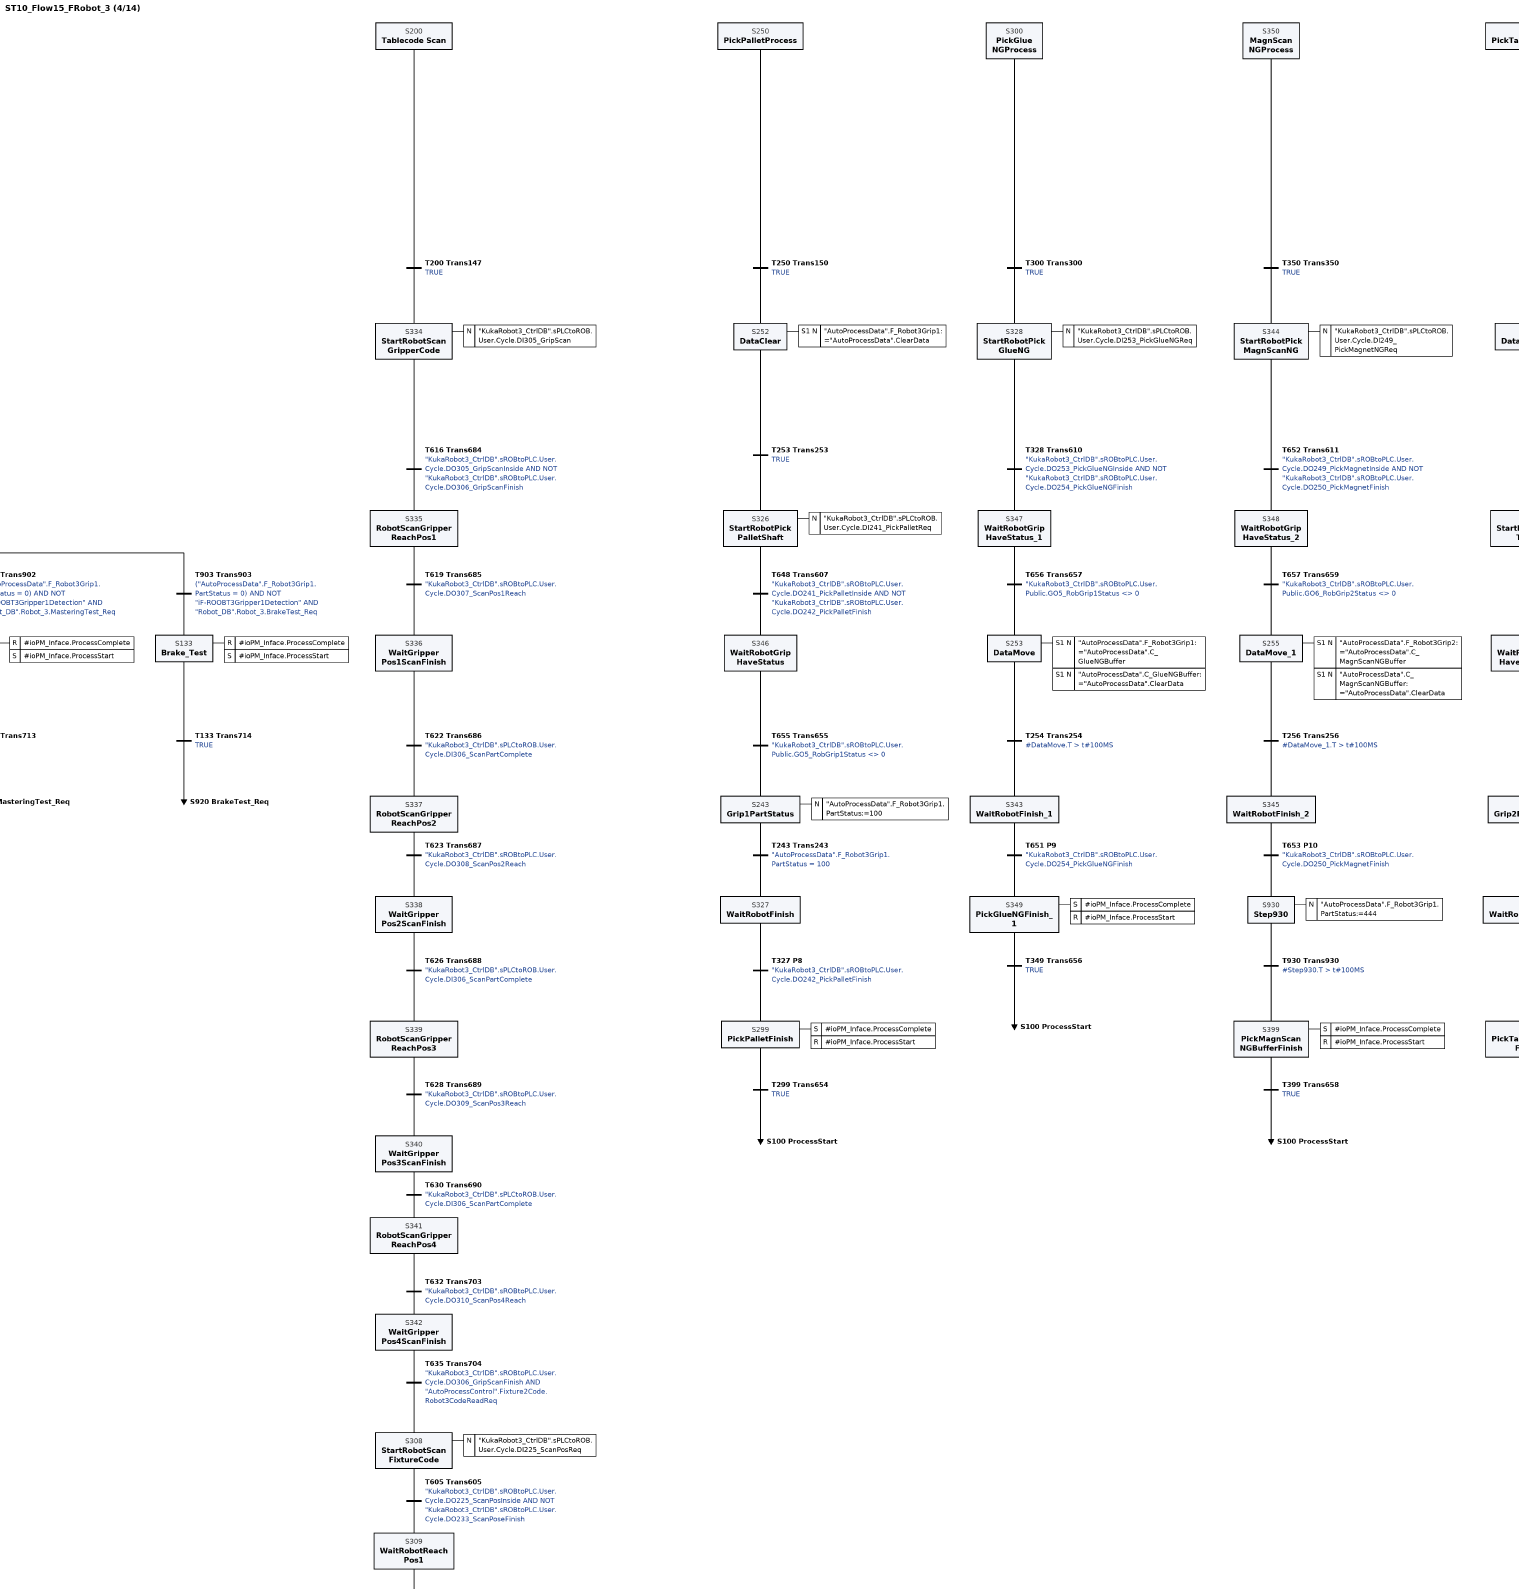
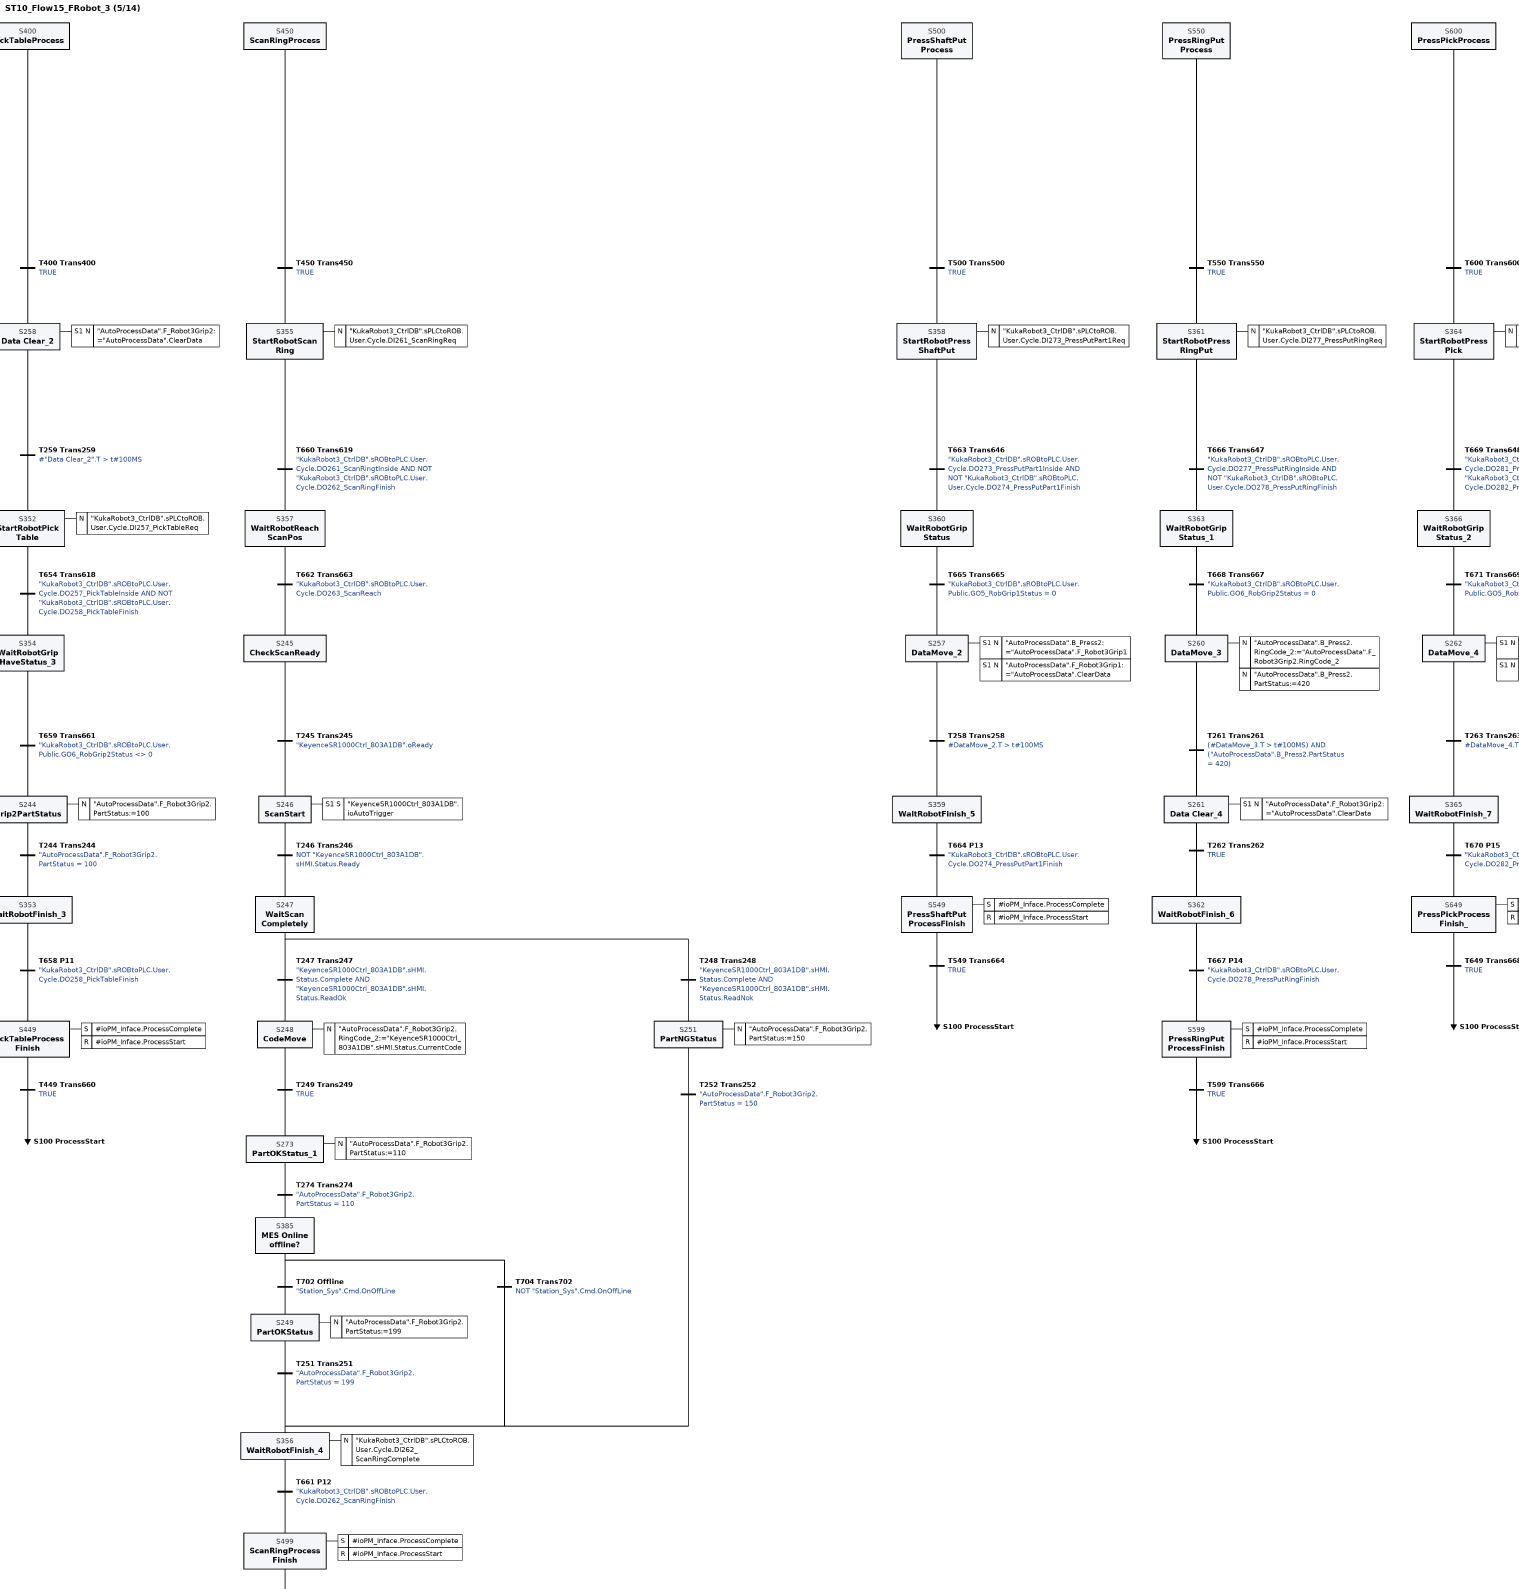
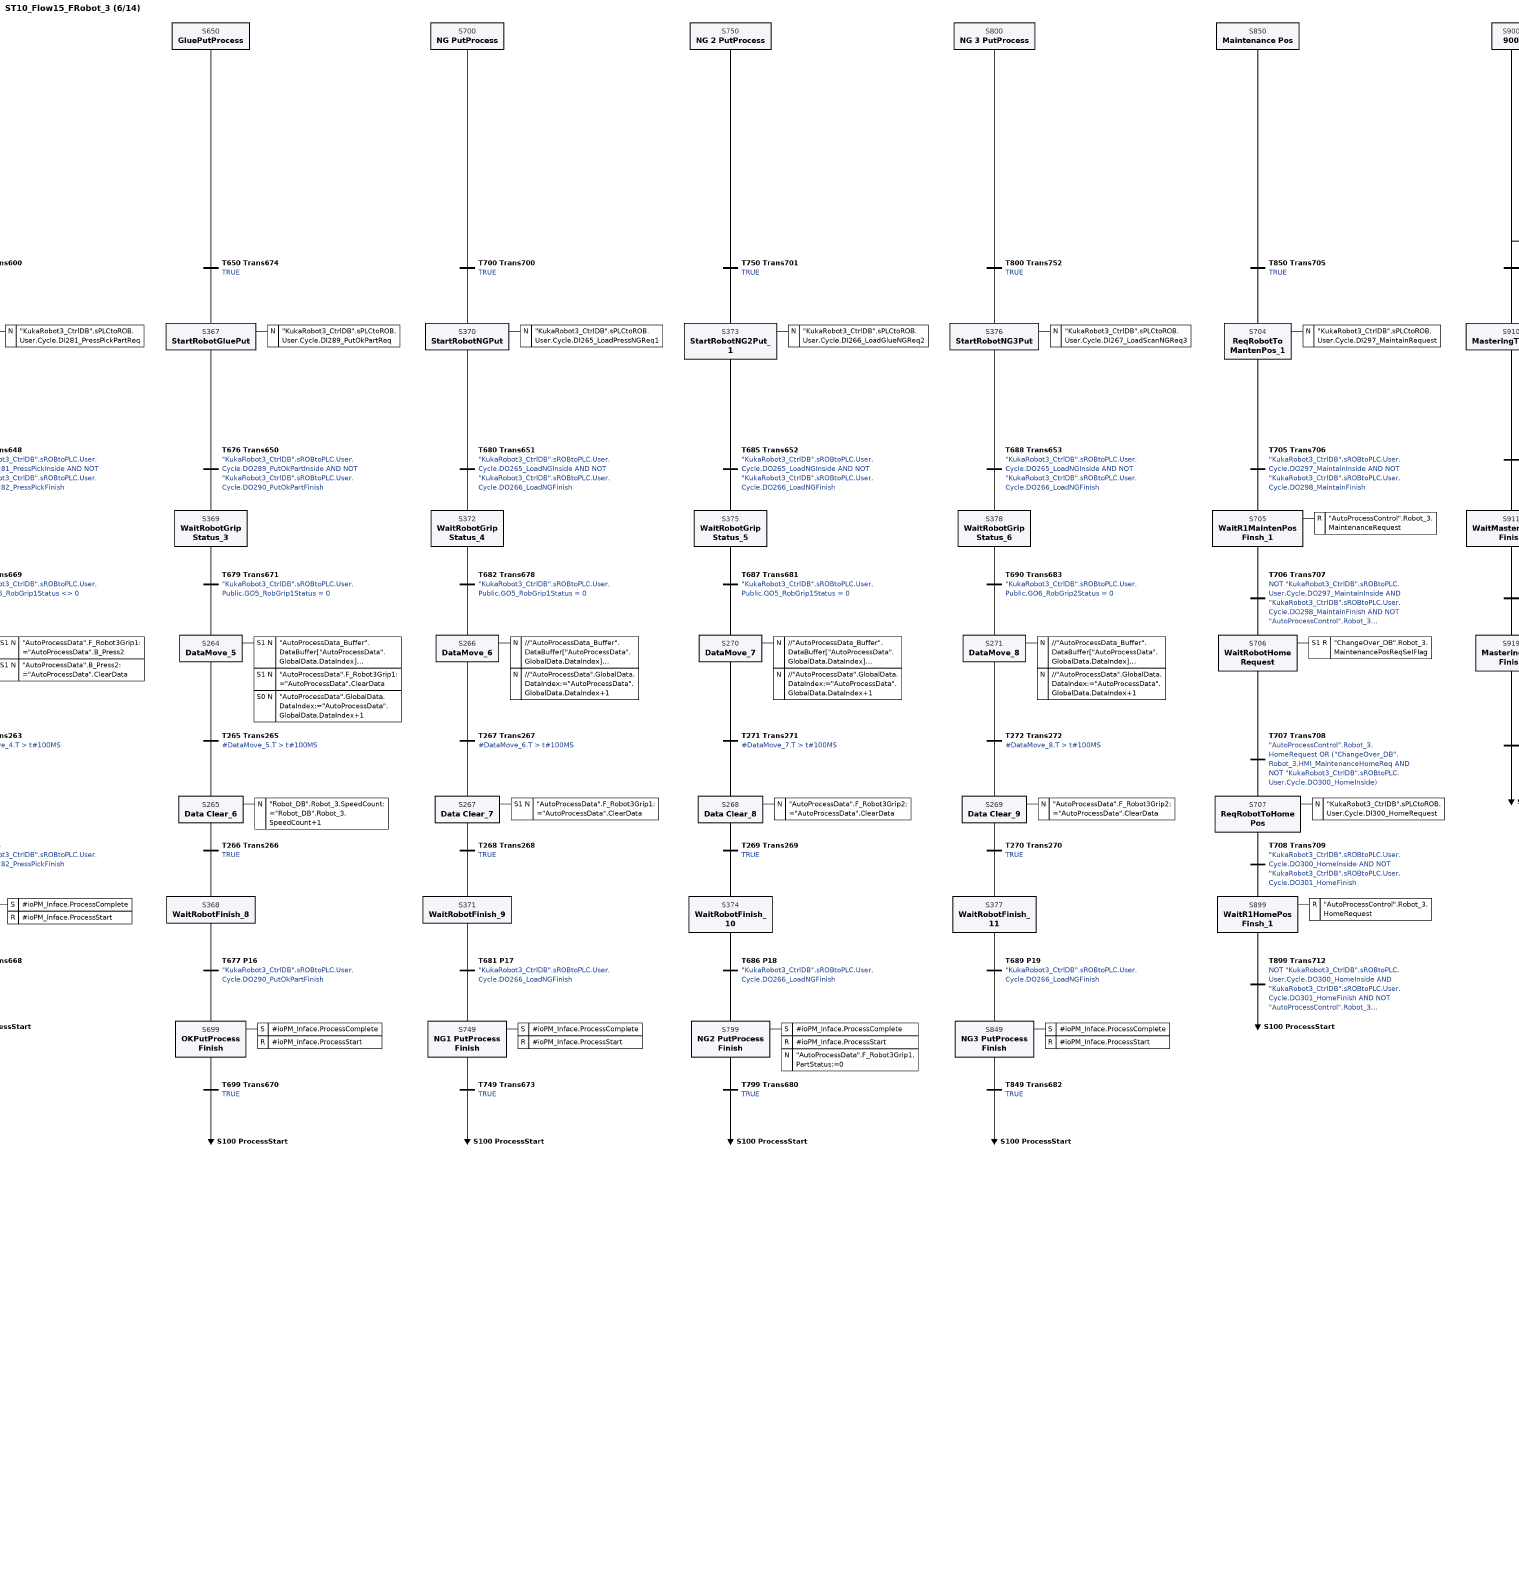
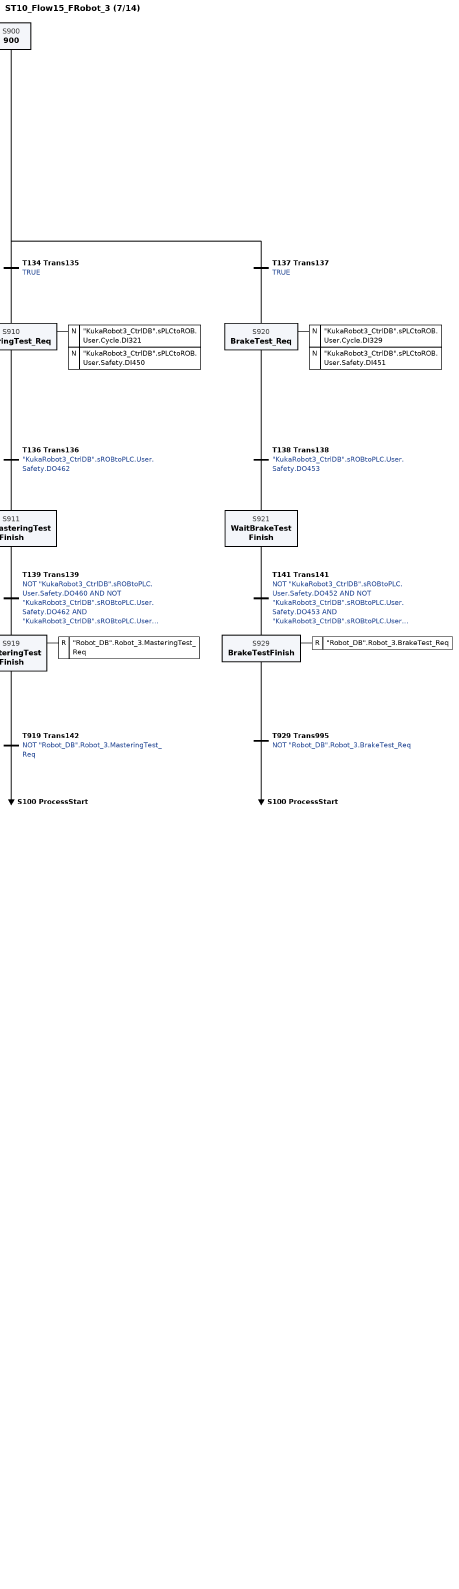
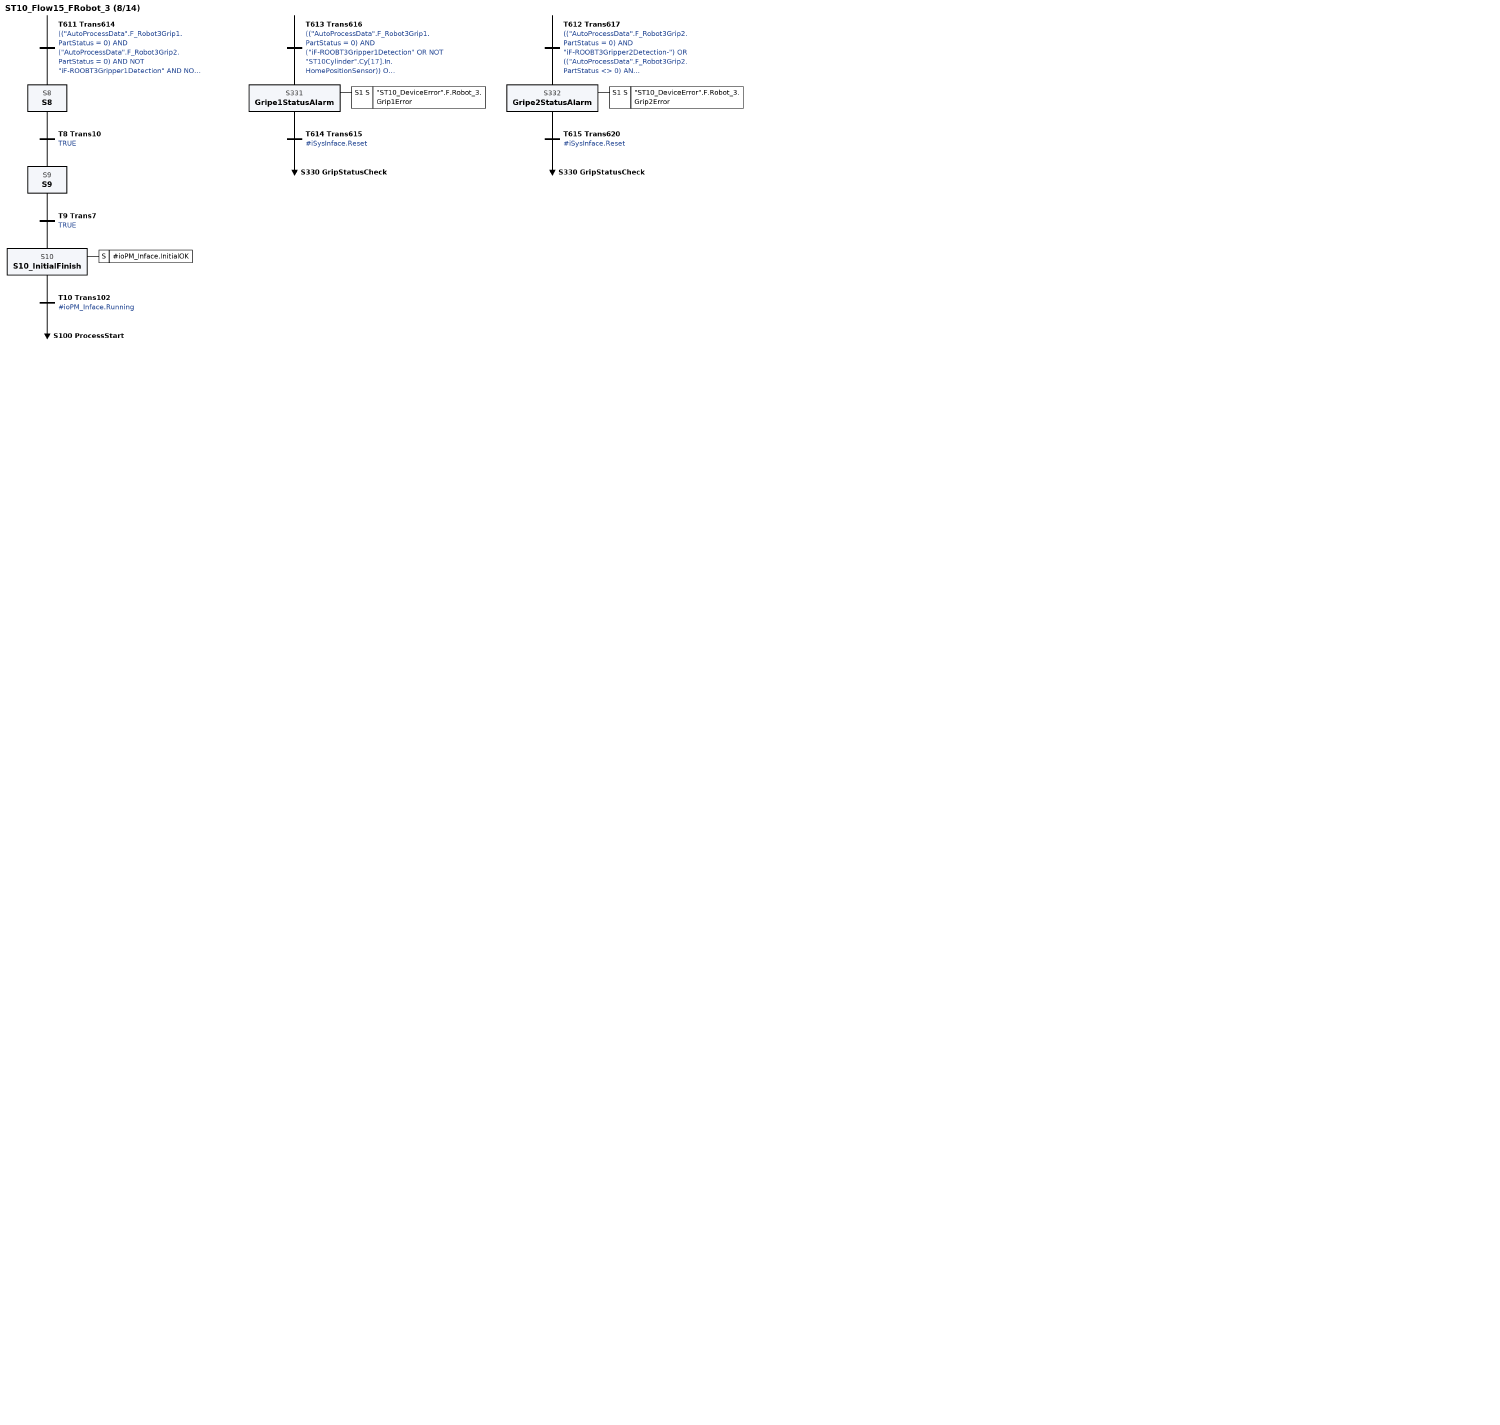
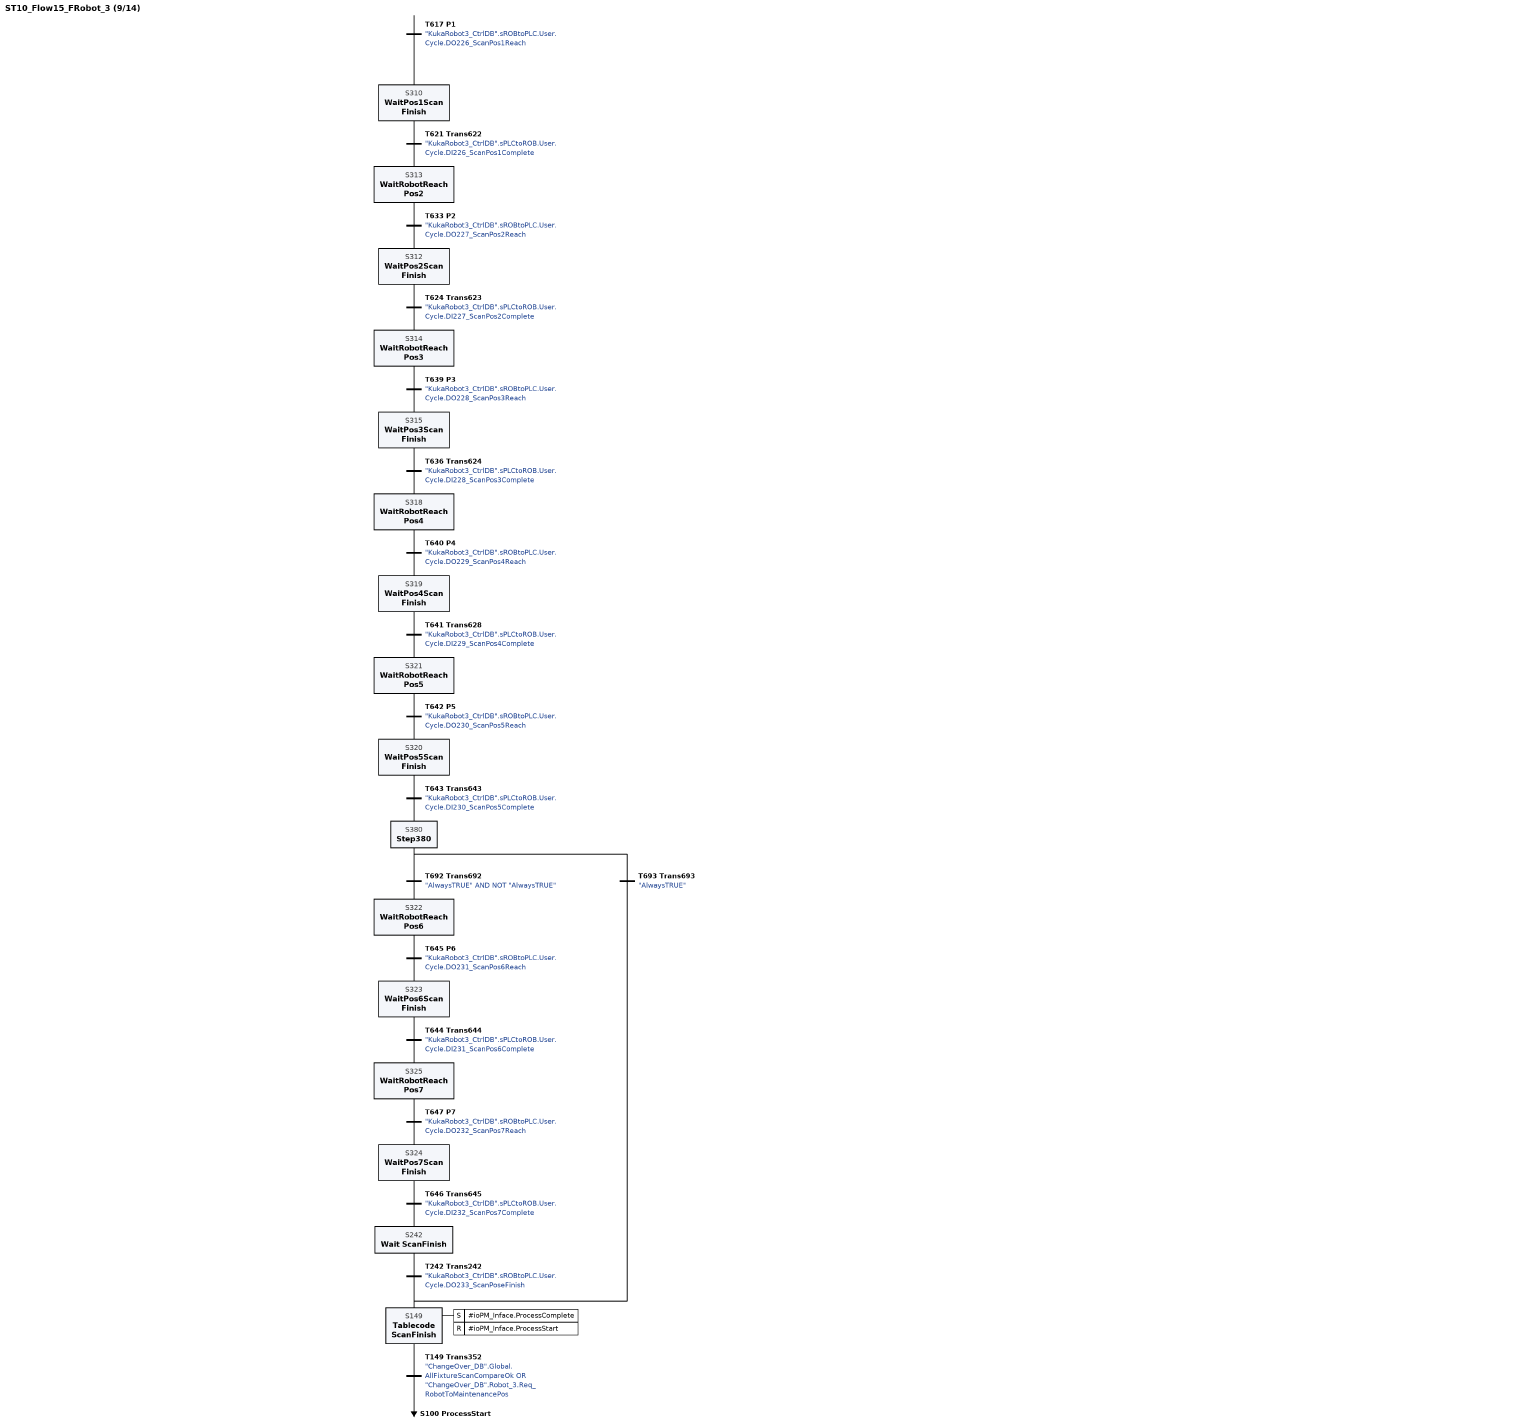
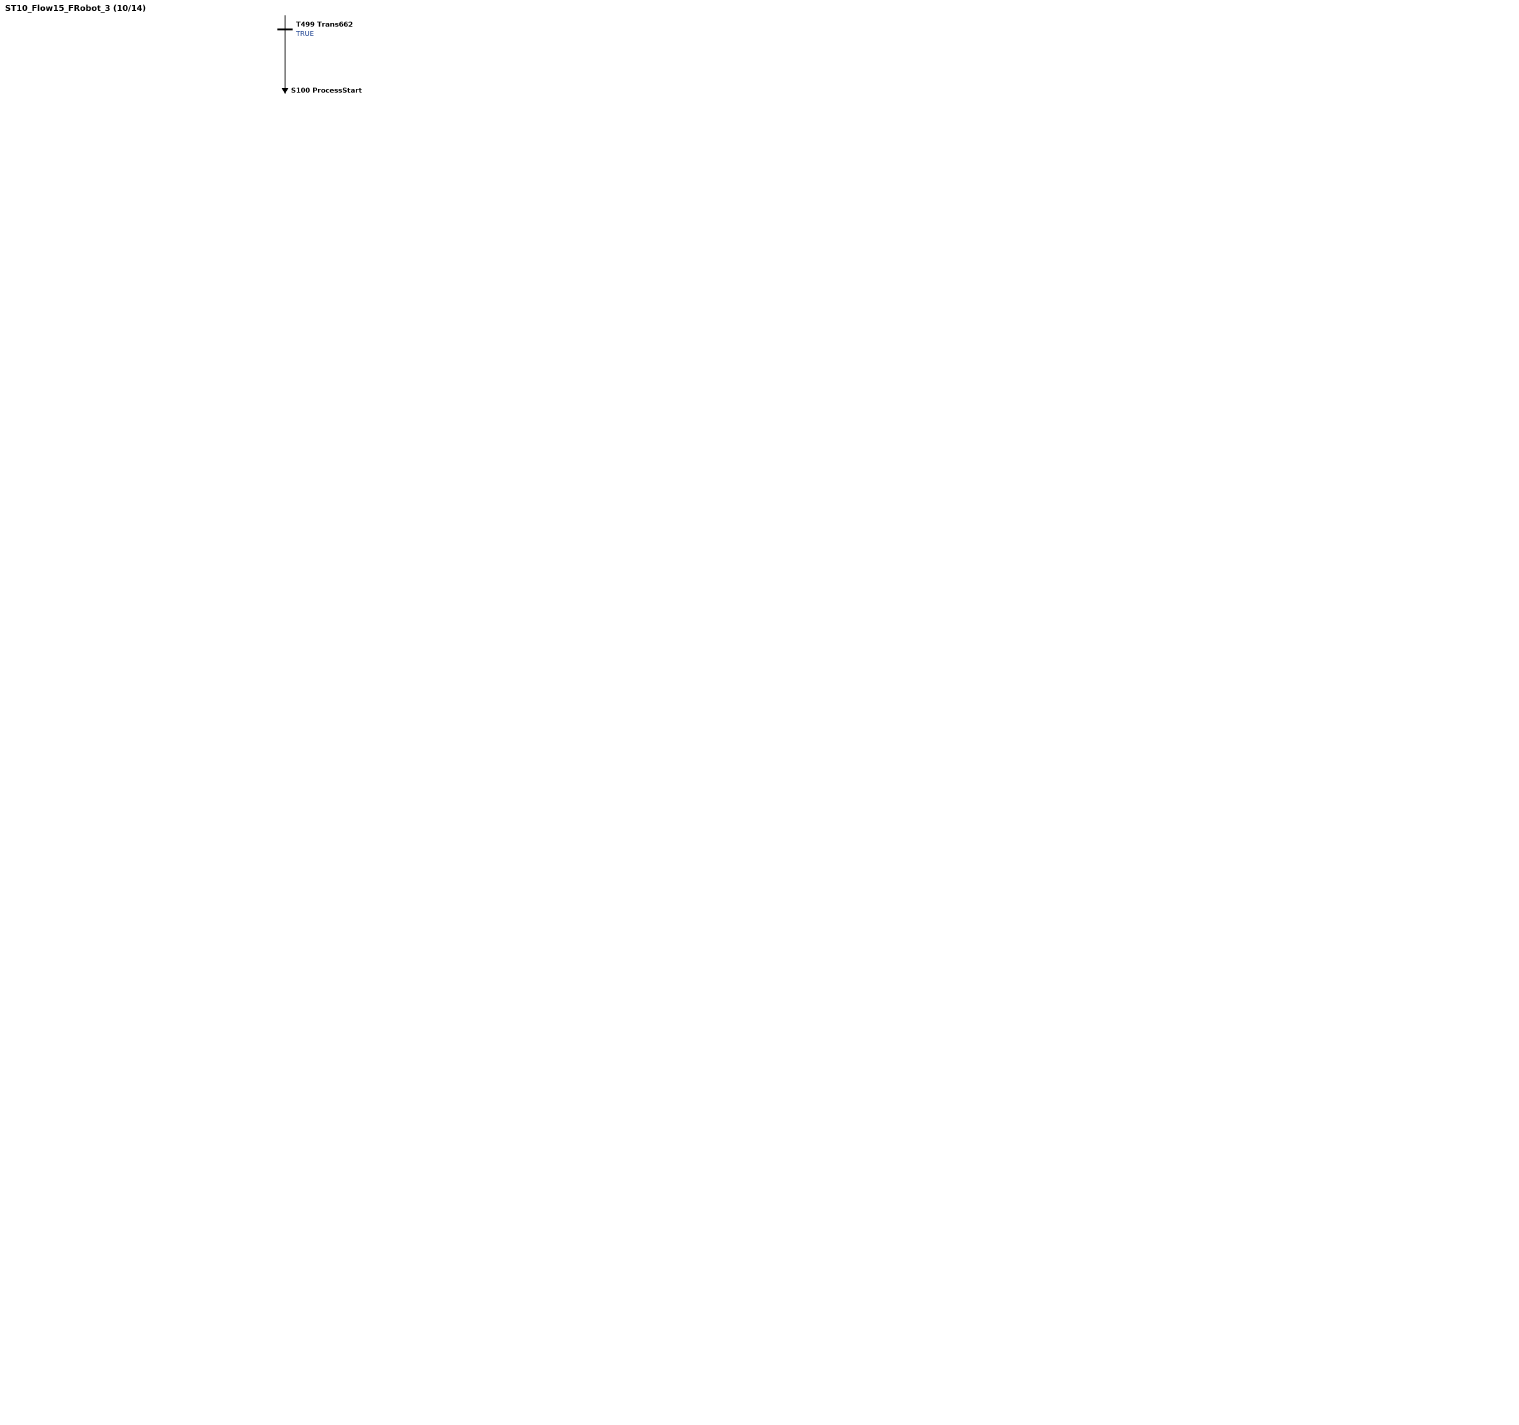
   // permanent pre-instructions
   NETWORK 1
      #TON[10].TON(IN := "AlwaysTRUE" AND "Station_Sys".Alarm.ImmediatelyStop, PT := T#300ms);
      #ioPM_Inface.AlarmImdilyStop := #TON[10].Q;
      #ioPM_Inface.AlarmCycleStop := "AlwaysTRUE" AND "Station_Sys".Alarm.CycleStop;
   NETWORK 2
      IF NOT False THEN
          #sCtrlMode(iSysInface := #iSysInface, ioPM_Inface := #ioPM_Inface, ioGraphCtrl := #RT_DATA.MOP);   // "SysFlowCtrlGraph"
      END_IF;
   NETWORK 3
      #TON[0].TON(IN := "AlwaysTRUE" AND "iA-Rotating product Check", PT := t#500ms);   // 工位11有托盘
      #TON[1].TOF(IN := "AlwaysTRUE" AND NOT "iA-Rotating product Check", PT := T#300ms);   // 工位无托盘
      #TON[2].TON(IN := "AlwaysTRUE", PT := T#300ms);
      #TON[3].TON(IN := "AlwaysTRUE", PT := T#300ms);
      #TON[4].TON(IN := "AlwaysTRUE", PT := T#300ms);
      #TON[5].TON(IN := "AlwaysTRUE", PT := T#300ms);
   NETWORK 4
      #前站站号 := 345;
      #本站站号 := 350;

   // sequencer 1: S01-S99 初始化 / S01-S99 Initial
   INITIAL_STEP F15_Initial:   // S1, max time T#10S, warning time T#7S
              S    #ioPM_Inface.InitialRun
              R    #ioPM_Inface.InitialOK
              R    #ioPM_Inface.WaitRunning
              R    #ioPM_Inface.Running
              R    #ioPM_Inface.ProcessComplete
              R    #ioPM_Inface.UnPause
              R    "Station_Sys".Cmd.Calibration
              R    "Station_Sys".Cmd.ChangeOver
                   //"ST350_Sys".Cmd.DryRun
              R    "Station_Sys".Cmd.Reserve
              R    "Station_Sys".Cmd.OneCycle
              R    "AutoProcessControl".Robot_3.Press2PutFlag
              R    "AutoProcessControl".Robot_3.Press2PickFlag
              R    "AutoProcessControl".Robot_3.GlueNGPickFlag
              R    "AutoProcessControl".Robot_3.ScanNGPickFlag
              R    "AutoProcessControl".Robot_3.NGPutFlag
              R    #ioPM_Inface.ProcessStart
          S1  R    "ChangeOver_DB".Robot_3.MaintenancePosReqSelFlag
                   //"Robot_DB".Robot_3.MasteringTest_Req
                   //"Robot_DB".Robot_3.BrakeTest_Req
   END_STEP
   TRANSITION Trans1 FROM F15_Initial TO S2   // T1
      := #iSysInface.Ready;
   END_TRANSITION
   STEP S2:   // S2, max time T#10S, warning time T#7S
   END_STEP
   TRANSITION Trans2 FROM S2 TO S3   // T2
      := TRUE;
   END_TRANSITION
   STEP RobotSpeed:   // S4, max time T#10S, warning time T#7S
              N    "KukaRobot3_CtrlDB".iSpeedValue:=20
   END_STEP
   TRANSITION Trans3 FROM RobotSpeed TO S5_MESInitial   // T3
      := "KukaRobot3_CtrlDB".iSpeedValue = 20;
   END_TRANSITION
   STEP S5_MESInitial:   // S5, max time T#10S, warning time T#7S
   END_STEP
   TRANSITION Trans325 FROM S5_MESInitial TO "RobotManuallyMoved?"   // T4
      := TRUE;
   END_TRANSITION
   STEP S10_InitialFinish:   // S10, max time T#10S, warning time T#7S
              S    #ioPM_Inface.InitialOK
   END_STEP
   TRANSITION Trans102 FROM S10_InitialFinish TO ProcessStart   // T10, jump
      := #ioPM_Inface.Running;
   END_TRANSITION
   STEP S3:   // S3, max time T#10S, warning time T#7S
   END_STEP
   TRANSITION Trans613 FROM S3 TO RobotSpeed   // T607
      := TRUE;
   END_TRANSITION
   STEP S8:   // S8, max time T#10S, warning time T#7S
   END_STEP
   TRANSITION Trans10 FROM S8 TO S9   // T8
      := TRUE;
   END_TRANSITION
   STEP S9:   // S9, max time T#10S, warning time T#7S
   END_STEP
   TRANSITION Trans7 FROM S9 TO S10_InitialFinish   // T9
      := TRUE;
   END_TRANSITION
   STEP "RobotReady?":   // S311, max time T#10S, warning time T#7S
   END_STEP
   TRANSITION Trans606 FROM "RobotReady?" TO RobotStart   // T606
      := "KukaRobot3_CtrlDB".sROBtoPLC.Sys.SO.ALARM_STOP AND "KukaRobot3_CtrlDB".sROBtoPLC.Sys.SO.EXT AND NOT "KukaRobot3_CtrlDB".oStartComplete;
   END_TRANSITION
   STEP RobotStart:   // S316, max time T#10S, warning time T#7S
              N    "KukaRobot3_CtrlDB".ioAutoStart
   END_STEP
   TRANSITION Trans608 FROM RobotStart TO WaitRobotStartHome   // T608
      := "KukaRobot3_CtrlDB".oReady AND "KukaRobot3_CtrlDB".oStartComplete;
   END_TRANSITION
   STEP RobotHome:   // S317, max time T#10S, warning time T#7S
              N    "KukaRobot3_CtrlDB".ioSrartHome
   END_STEP
   TRANSITION Trans609 FROM RobotHome TO RobotAutoCycle   // T609
      := "KukaRobot3_CtrlDB".sROBtoPLC.Sys.SO.IN_HOME AND "KukaRobot3_CtrlDB".sHMI.HomeSeqOK AND "KukaRobot3_CtrlDB".sHMI.WaitForAutoCycleStart AND NOT "KukaRobot3_CtrlDB".sHMI.GoHomeFail;
   END_TRANSITION
   STEP RobotAutoCycle:   // S329, max time T#10S, warning time T#7S
              N    "KukaRobot3_CtrlDB".ioStartAutoCycle
   END_STEP
   TRANSITION Trans612 FROM RobotAutoCycle TO GripStatusCheck   // T610
      := NOT "KukaRobot3_CtrlDB".sHMI.HomeSeqOK AND NOT "KukaRobot3_CtrlDB".sHMI.WaitForAutoCycleStart;
   END_TRANSITION
   STEP GripStatusCheck:   // S330, max time T#10S, warning time T#7S
   END_STEP
   TRANSITION Trans614 FROM GripStatusCheck TO S8   // T611
      := (("AutoProcessData".F_Robot3Grip1.PartStatus = 0) AND ("AutoProcessData".F_Robot3Grip2.PartStatus = 0) AND NOT "iF-ROOBT3Gripper1Detection" AND NOT "iF-ROOBT3Gripper2Detection-") OR (("AutoProcessData".F_Robot3Grip1.PartStatus <> 0) AND NOT "ST10Cylinder".Cy[17].In.WorkPositionSensor AND NOT "ST10Cylinder".Cy[17].In.HomePositionSensor) OR (("AutoProcessData".F_Robot3Grip2.PartStatus <> 0) AND NOT "iF-ROOBT3Gripper2Detection-" AND NOT "ST10Cylinder".Cy[18].In.HomePositionSensor);
   END_TRANSITION
   TRANSITION Trans616 FROM GripStatusCheck TO Gripe1StatusAlarm   // T613
      := (("AutoProcessData".F_Robot3Grip1.PartStatus = 0) AND ("iF-ROOBT3Gripper1Detection" OR NOT "ST10Cylinder".Cy[17].In.HomePositionSensor)) OR (("AutoProcessData".F_Robot3Grip1.PartStatus <> 0) AND (NOT "iF-ROOBT3Gripper1Detection" OR "ST10Cylinder".Cy[17].In.HomePositionSensor));
   END_TRANSITION
   TRANSITION Trans617 FROM GripStatusCheck TO Gripe2StatusAlarm   // T612
      := (("AutoProcessData".F_Robot3Grip2.PartStatus = 0) AND "iF-ROOBT3Gripper2Detection-") OR (("AutoProcessData".F_Robot3Grip2.PartStatus <> 0) AND "iF-ROOBT3Gripper2Detection-");
   END_TRANSITION
   STEP Gripe1StatusAlarm:   // S331, max time T#10S, warning time T#7S
          S1  S    "ST10_DeviceError".F.Robot_3.Grip1Error
   END_STEP
   TRANSITION Trans615 FROM Gripe1StatusAlarm TO GripStatusCheck   // T614, jump
      := #iSysInface.Reset;
   END_TRANSITION
   STEP Gripe2StatusAlarm:   // S332, max time T#10S, warning time T#7S
          S1  S    "ST10_DeviceError".F.Robot_3.Grip2Error
   END_STEP
   TRANSITION Trans620 FROM Gripe2StatusAlarm TO GripStatusCheck   // T615, jump
      := #iSysInface.Reset;
   END_TRANSITION
   STEP WaitRobotStartHome:   // S383, max time T#10S, warning time T#7S
   END_STEP
   TRANSITION Trans698 FROM WaitRobotStartHome TO RobotHome   // T698
      := "KukaRobot3_CtrlDB".sROBtoPLC.User.Home.DO161_WaitForHomeSeqStart;
   END_TRANSITION
   STEP "RobotManuallyMoved?":   // S384, max time T#10S, warning time T#7S
   END_STEP
   TRANSITION Trans699 FROM "RobotManuallyMoved?" TO "RobotReady?"   // T701
      := NOT "KukaRobot3_CtrlDB".sPLCtoROB.User.Home.DI169_RobotMoved AND NOT "ST10_DeviceError".F.Robot_3.ManualMoved;
   END_TRANSITION

   // sequencer 2: S100-S199 等待到位 / S100-S199 RobotTask
   STEP ProcessStart:   // S100, max time T#10S, warning time T#7S
      // 自动等待开始运行
              R    #ioPM_Inface.InitialRun
              R    #ioPM_Inface.ProcessComplete
              R    #ioPM_Inface.ProcessStart
              S    #ioPM_Inface.InitialOK
              S    #ioPM_Inface.WaitRunning
          S1  N    #ioPM_Inface.ProcessResult:=0
              R    "ST10_GeneralData".FlowControl_Handshake[5].Start
              R    "ST10_GeneralData".FlowControl_Handshake[5].Done
   END_STEP
   TRANSITION Trans200 FROM ProcessStart TO FlagReset   // T100
      := NOT #ioPM_Inface.AlarmCycleStop AND #ioPM_Inface.Running AND NOT #iSysInface.Auto.RunningOver AND (NOT #iSysInface.Auto.OneCycleMode OR (#iSysInface.Auto.OneCycleMode AND #ioPM_Inface.TriggerOneCycle));
   END_TRANSITION
   STEP PressShaftPut:   // S140, max time T#10S, warning time T#7S
              R    #ioPM_Inface.ProcessComplete
              S    #ioPM_Inface.ProcessStart
   END_STEP
   TRANSITION Trans638 FROM PressShaftPut TO PressShaftPutProcess   // T140, jump
      := TRUE;
   END_TRANSITION
   STEP ScanFixtureCode:   // S110, max time T#10S, warning time T#7S
              R    #ioPM_Inface.ProcessComplete
              S    #ioPM_Inface.ProcessStart
   END_STEP
   TRANSITION Trans625 FROM ScanFixtureCode TO "Tablecode Scan"   // T110, jump
      := TRUE;
   END_TRANSITION
   STEP RobotTaskSelect:   // S333, max time T#10S, warning time T#7S
   END_STEP
   TRANSITION Trans621 FROM RobotTaskSelect TO ScanFixtureCode   // T333
      := NOT "ChangeOver_DB".Robot_3.MaintenancePosReqSelFlag AND NOT "AutoProcessData".GlobalData.Robot3GripperCodeOKFlag AND ("AutoProcessData".F_Robot3Grip1.PartStatus = 0) AND NOT "iF-ROOBT3Gripper1Detection" AND NOT "KukaRobot2_CtrlDB".sROBtoPLC.User.Cycle.DO253_GlueNGPutInside AND NOT "KukaRobot2_CtrlDB".sROBtoPLC.User.Cycle.DO249_ScanNGPutInside AND NOT "KukaRobot2_CtrlDB".sROBtoPLC.User.Cycle.DO273_PressPutPart1Inside AND NOT "PalletNGData".UnLoadingNGPallet.OpenFlag AND "AutoProcessControl".Robot_3.GripScanRequest AND NOT "Robot_DB".Robot_3.MasteringTest_Req AND NOT "Robot_DB".Robot_3.BrakeTest_Req;
   END_TRANSITION
   TRANSITION NoUse FROM RobotTaskSelect TO PickPallet   // T618
      := NOT "ChangeOver_DB".Robot_3.MaintenancePosReqSelFlag AND "AlwaysTRUE" AND NOT "AlwaysTRUE" AND ("AutoProcessData".F_Robot3Grip1.PartStatus = 0) AND NOT "iF-ROOBT3Gripper1Detection" AND "ST10Cylinder".Cy[17].In.HomePositionSensor AND "AutoProcessControl".H_ShafeLine.Robot1PickPrimit AND NOT "PalletNGData".UnLoadingNGPallet.OpenFlag AND "AutoProcessControl".A_ScanRotary.Robot1PutPrimit AND NOT "Robot_DB".Robot_3.MasteringTest_Req AND NOT "Robot_DB".Robot_3.BrakeTest_Req;
   END_TRANSITION
   TRANSITION Trans630 FROM RobotTaskSelect TO PickGlueNGReq   // T620
      := NOT "ChangeOver_DB".Robot_3.MaintenancePosReqSelFlag AND NOT "ChangeOver_DB".Robot_2.MaintenancePosReqSelFlag AND ("AutoProcessData".F_Robot3Grip1.PartStatus = 0) AND NOT "iF-ROOBT3Gripper1Detection" AND "iE-NG-03ShaftDispenseNGDetection" AND "KukaRobot2_CtrlDB".sROBtoPLC.User.Home.DO181_Robot3Area AND NOT "KukaRobot2_CtrlDB".sROBtoPLC.User.Cycle.DO253_GlueNGPutInside AND NOT "KukaRobot2_CtrlDB".sROBtoPLC.User.Cycle.DO249_ScanNGPutInside AND NOT "KukaRobot2_CtrlDB".sROBtoPLC.User.Cycle.DO273_PressPutPart1Inside AND NOT "AutoProcessControl".Robot_2.GlueNGPutFlag AND NOT "AutoProcessControl".Robot_2.ScanNGPutFlag AND NOT "AutoProcessControl".Robot_2.Press2PutFlag AND NOT "PalletNGData".UnLoadingNGPallet.OpenFlag AND "AutoProcessControl".NGBuffer.PickGlueNGPrimit AND NOT "Robot_DB".Robot_3.MasteringTest_Req AND NOT "Robot_DB".Robot_3.BrakeTest_Req;
   END_TRANSITION
   TRANSITION Trans632 FROM RobotTaskSelect TO PickTable   // T625
      := (NOT "AutoProcessControl".Robot_1.ClearPart OR ("AutoProcessControl".Robot_1.ClearPart AND "AutoProcessControl".B_Press_2.Robot3PutRingPrimit)) AND NOT "ChangeOver_DB".Robot_3.MaintenancePosReqSelFlag AND ("AutoProcessData".F_Robot3Grip1.PartStatus = 0) AND NOT "iF-ROOBT3Gripper1Detection" AND ("AutoProcessData".F_Robot3Grip2.PartStatus = 0) AND NOT "iF-ROOBT3Gripper2Detection-" AND NOT "iE-NG-03MagnetDispenseNGDetection" AND NOT "iE-NG-03ShaftDispenseNGDetection" AND NOT "PalletNGData".UnLoadingNGPallet.OpenFlag AND "AutoProcessControl".A_Table_2Loading.Robot3PickPrimit AND NOT "Robot_DB".Robot_3.MasteringTest_Req AND NOT "Robot_DB".Robot_3.BrakeTest_Req;
   END_TRANSITION
   TRANSITION Trans633 FROM RobotTaskSelect TO ScanRing   // T627
      := NOT "ChangeOver_DB".Robot_3.MaintenancePosReqSelFlag AND ("AutoProcessData".F_Robot3Grip2.PartStatus = 100) AND ("iF-ROOBT3Gripper2Detection-" OR "AlwaysTRUE") AND NOT "ChangeOver_DB".Global.ManualModeFlag AND NOT "PalletNGData".UnLoadingNGPallet.OpenFlag AND NOT "ST10Cylinder".Cy[18].In.HomePositionSensor AND NOT "Robot_DB".Robot_3.MasteringTest_Req AND NOT "Robot_DB".Robot_3.BrakeTest_Req;
   END_TRANSITION
   TRANSITION Trans635 FROM RobotTaskSelect TO PickMagnetNGReqPick   // T629
      := NOT "ChangeOver_DB".Robot_3.MaintenancePosReqSelFlag AND NOT "ChangeOver_DB".Robot_2.MaintenancePosReqSelFlag AND ("AutoProcessData".F_Robot3Grip1.PartStatus = 0) AND NOT "iF-ROOBT3Gripper1Detection" AND ("AutoProcessData".F_Robot3Grip2.PartStatus = 0) AND NOT "iF-ROOBT3Gripper2Detection-" AND "iE-NG-03MagnetDispenseNGDetection" AND "KukaRobot2_CtrlDB".sROBtoPLC.User.Home.DO181_Robot3Area AND NOT "KukaRobot2_CtrlDB".sROBtoPLC.User.Cycle.DO253_GlueNGPutInside AND NOT "KukaRobot2_CtrlDB".sROBtoPLC.User.Cycle.DO249_ScanNGPutInside AND NOT "KukaRobot2_CtrlDB".sROBtoPLC.User.Cycle.DO273_PressPutPart1Inside AND NOT "AutoProcessControl".Robot_2.GlueNGPutFlag AND NOT "AutoProcessControl".Robot_2.ScanNGPutFlag AND NOT "AutoProcessControl".Robot_2.Press2PutFlag AND NOT "PalletNGData".UnLoadingNGPallet.OpenFlag AND "AutoProcessControl".NGBuffer.Robot3PPickMagnetNGPrimit AND NOT "Robot_DB".Robot_3.MasteringTest_Req AND NOT "Robot_DB".Robot_3.BrakeTest_Req;
   END_TRANSITION
   TRANSITION Trans675 FROM RobotTaskSelect TO "NG2Put_1Press/Glue"   // T674
      := ((("AutoProcessData".F_Robot3Grip1.PartStatus >= 450) AND ("AutoProcessData".F_Robot3Grip1.PartStatus <= 460)) OR (("AutoProcessData".F_Robot3Grip1.PartStatus >= 350) AND ("AutoProcessData".F_Robot3Grip1.PartStatus <= 360))) AND NOT "ChangeOver_DB".Robot_3.MaintenancePosReqSelFlag AND ("iF-ROOBT3Gripper1Detection" OR "AlwaysTRUE") AND NOT "ST10Cylinder".Cy[17].In.HomePositionSensor AND NOT "PalletNGData".UnLoadingNGPallet.OpenFlag AND "AutoProcessControl".NG_2.Robot3PutPrimit_1;
   END_TRANSITION
   TRANSITION Trans750 FROM RobotTaskSelect TO "NG2Put_2/Magnet"   // T757
      := NOT "ChangeOver_DB".Robot_3.MaintenancePosReqSelFlag AND ((("AutoProcessData".F_Robot3Grip2.PartStatus >= 155) AND ("AutoProcessData".F_Robot3Grip2.PartStatus <= 160)) OR ("AutoProcessData".F_Robot3Grip1.PartStatus = 444)) AND ("iF-ROOBT3Gripper2Detection-" OR "AlwaysTRUE") AND NOT "ST10Cylinder".Cy[18].In.HomePositionSensor AND NOT "PalletNGData".UnLoadingNGPallet.OpenFlag AND "AutoProcessControl".NG_2.Robot3PutPrimit_2;
   END_TRANSITION
   TRANSITION Trans751 FROM RobotTaskSelect TO "NG2Put_3/Ring"   // T751
      := ((("AutoProcessData".F_Robot3Grip2.PartStatus >= 150) AND ("AutoProcessData".F_Robot3Grip2.PartStatus < 155)) OR ("ChangeOver_DB".Global.ManualModeFlag AND ("AutoProcessData".F_Robot3Grip2.PartStatus = 100)) OR (("AutoProcessData".F_Robot3Grip2.PartStatus = 199) AND ("AutoProcessData".F_Robot2Grip2.PartStatus = 155) AND ("AutoProcessData".C_MagnScanNGBuffer.PartStatus = 155))) AND NOT "ChangeOver_DB".Robot_3.MaintenancePosReqSelFlag AND ("iF-ROOBT3Gripper2Detection-" OR "AlwaysTRUE") AND NOT "ST10Cylinder".Cy[18].In.HomePositionSensor AND NOT "PalletNGData".UnLoadingNGPallet.OpenFlag AND "AutoProcessControl".NG_2.Robot3PutPrimit_3;
   END_TRANSITION
   TRANSITION Trans694 FROM RobotTaskSelect TO Grip1SensorError   // T694
      := ((("AutoProcessData".F_Robot3Grip1.PartStatus <> 0) AND NOT "iF-ROOBT3Gripper1Detection") OR (("AutoProcessData".F_Robot3Grip1.PartStatus = 0) AND ("iF-ROOBT3Gripper1Detection" OR "AlwaysTRUE"))) AND (#RobotTaskSelect.T > t#5000MS) AND "TON".TON[69].Q;
   END_TRANSITION
   TRANSITION Trans695 FROM RobotTaskSelect TO Grip2SensorError   // T695
      := ((("AutoProcessData".F_Robot3Grip2.PartStatus <> 0) AND "iF-ROOBT3Gripper2Detection-") OR (("AutoProcessData".F_Robot3Grip2.PartStatus = 0) AND "iF-ROOBT3Gripper2Detection-")) AND (#RobotTaskSelect.T > t#5000MS) AND "TON".TON[70].Q;
   END_TRANSITION
   TRANSITION Trans642 FROM RobotTaskSelect TO PressPick   // T637
      := NOT "ChangeOver_DB".Robot_3.MaintenancePosReqSelFlag AND ("AutoProcessData".F_Robot3Grip1.PartStatus = 0) AND NOT "iF-ROOBT3Gripper1Detection" AND "KukaRobot2_CtrlDB".sROBtoPLC.User.Home.DO181_Robot3Area AND NOT "AutoProcessControl".Robot_2.GlueNGPutFlag AND NOT "AutoProcessControl".Robot_2.ScanNGPutFlag AND NOT "AutoProcessControl".Robot_2.Press2PutFlag AND NOT "PalletNGData".UnLoadingNGPallet.OpenFlag AND "AutoProcessControl".B_Press_2.Robot3PickPrimit AND NOT "Robot_DB".Robot_3.MasteringTest_Req AND NOT "Robot_DB".Robot_3.BrakeTest_Req;
   END_TRANSITION
   TRANSITION Trans640 FROM RobotTaskSelect TO PressRingPut   // T634
      := NOT "ChangeOver_DB".Robot_3.MaintenancePosReqSelFlag AND ("AutoProcessData".F_Robot3Grip2.PartStatus = 199) AND NOT "ChangeOver_DB".Global.ManualModeFlag AND ("iF-ROOBT3Gripper2Detection-" OR "AlwaysTRUE") AND NOT "ST10Cylinder".Cy[18].In.HomePositionSensor AND ("AutoProcessData".F_Robot3Grip1.PartStatus = 0) AND NOT "iF-ROOBT3Gripper1Detection" AND NOT "KukaRobot2_CtrlDB".sROBtoPLC.User.Cycle.DO253_GlueNGPutInside AND NOT "KukaRobot2_CtrlDB".sROBtoPLC.User.Cycle.DO249_ScanNGPutInside AND NOT "KukaRobot2_CtrlDB".sROBtoPLC.User.Cycle.DO273_PressPutPart1Inside AND "KukaRobot2_CtrlDB".sROBtoPLC.User.Home.DO181_Robot3Area AND "KukaRobot2_CtrlDB".sROBtoPLC.User.Home.DO180_PressPutArea AND NOT "AutoProcessControl".Robot_2.GlueNGPutFlag AND NOT "AutoProcessControl".Robot_2.ScanNGPutFlag AND NOT "AutoProcessControl".Robot_2.Press2PutFlag AND NOT "PalletNGData".UnLoadingNGPallet.OpenFlag AND "AutoProcessControl".B_Press_2.Robot3PutRingPrimit AND NOT "Robot_DB".Robot_3.MasteringTest_Req AND NOT "Robot_DB".Robot_3.BrakeTest_Req;
   END_TRANSITION
   TRANSITION Trans672 FROM RobotTaskSelect TO OKPut   // T672
      := NOT "ChangeOver_DB".Robot_3.MaintenancePosReqSelFlag AND ("AutoProcessData".F_Robot3Grip1.PartStatus = 499) AND NOT "ChangeOver_DB".Global.ManualModeFlag AND ("iF-ROOBT3Gripper1Detection" OR "AlwaysTRUE") AND NOT "ST10Cylinder".Cy[17].In.HomePositionSensor AND NOT "ST10Cylinder".Cy[17].In.WorkPositionSensor AND NOT "PalletNGData".UnLoadingNGPallet.OpenFlag AND "AutoProcessControl".L_ShafeLine.Robot3PutPrimit;
   END_TRANSITION
   TRANSITION NoUsed FROM RobotTaskSelect TO PressShaftPut   // T631
      := NOT "ChangeOver_DB".Robot_3.MaintenancePosReqSelFlag AND "AlwaysTRUE" AND NOT "AlwaysTRUE" AND ("AutoProcessData".F_Robot3Grip1.PartStatus = 199) AND ("iF-ROOBT3Gripper1Detection" OR "AlwaysTRUE") AND NOT "ST10Cylinder".Cy[17].In.HomePositionSensor AND ("AutoProcessData".F_Robot3Grip2.PartStatus = 199) AND ("iF-ROOBT3Gripper2Detection-" OR "AlwaysTRUE") AND NOT "ST10Cylinder".Cy[18].In.HomePositionSensor AND NOT "PalletNGData".UnLoadingNGPallet.OpenFlag AND "AutoProcessControl".B_Press_1.Robot1PutShaftPrimit;
   END_TRANSITION
   TRANSITION Trans711 FROM RobotTaskSelect TO Maintenance   // T673
      := ((("AutoProcessData".F_Robot3Grip1.PartStatus = 0) AND NOT "iF-ROOBT3Gripper1Detection" AND ("AutoProcessData".F_Robot3Grip2.PartStatus = 0) AND NOT "iF-ROOBT3Gripper2Detection-" AND "ChangeOver_DB".Robot_3.Req_RobotToMaintenancePos) OR ("ChangeOver_DB".Robot_3.HMI_MaintenancePosActive AND NOT "AutoProcessControl".Robot_3.MaintenanceRequest)) AND NOT "Robot_DB".Robot_3.MasteringTest_Req AND NOT "Robot_DB".Robot_3.BrakeTest_Req;
   END_TRANSITION
   TRANSITION Trans902 FROM RobotTaskSelect TO Masref_test   // T902
      := ("AutoProcessData".F_Robot3Grip1.PartStatus = 0) AND NOT "iF-ROOBT3Gripper1Detection" AND "Robot_DB".Robot_3.MasteringTest_Req;
   END_TRANSITION
   TRANSITION Trans903 FROM RobotTaskSelect TO Brake_Test   // T903
      := ("AutoProcessData".F_Robot3Grip1.PartStatus = 0) AND NOT "iF-ROOBT3Gripper1Detection" AND "Robot_DB".Robot_3.BrakeTest_Req;
   END_TRANSITION
   STEP PickPallet:   // S115, max time T#10S, warning time T#7S
              R    #ioPM_Inface.ProcessComplete
              S    #ioPM_Inface.ProcessStart
   END_STEP
   TRANSITION Trans627 FROM PickPallet TO PickPalletProcess   // T115, jump
      := TRUE;
   END_TRANSITION
   STEP PickGlueNGReq:   // S120, max time T#10S, warning time T#7S
              R    #ioPM_Inface.ProcessComplete
              S    #ioPM_Inface.ProcessStart
   END_STEP
   TRANSITION Trans629 FROM PickGlueNGReq TO PickGlueNGProcess   // T120, jump
      := TRUE;
   END_TRANSITION
   STEP PickTable:   // S130, max time T#10S, warning time T#7S
              R    #ioPM_Inface.ProcessComplete
              S    #ioPM_Inface.ProcessStart
   END_STEP
   TRANSITION Trans631 FROM PickTable TO PickTableProcess   // T130, jump
      := TRUE;
   END_TRANSITION
   STEP ScanRing:   // S135, max time T#10S, warning time T#7S
              R    #ioPM_Inface.ProcessComplete
              S    #ioPM_Inface.ProcessStart
   END_STEP
   TRANSITION Trans634 FROM ScanRing TO ScanRingProcess   // T135, jump
      := TRUE;
   END_TRANSITION
   STEP PickMagnetNGReqPick:   // S125, max time T#10S, warning time T#7S
              R    #ioPM_Inface.ProcessComplete
              S    #ioPM_Inface.ProcessStart
   END_STEP
   TRANSITION Trans636 FROM PickMagnetNGReqPick TO MagnScanNGProcess   // T125, jump
      := TRUE;
   END_TRANSITION
   STEP OKPut:   // S155, max time T#10S, warning time T#7S
              R    #ioPM_Inface.ProcessComplete
              S    #ioPM_Inface.ProcessStart
   END_STEP
   TRANSITION Trans649 FROM OKPut TO GluePutProcess   // T155, jump
      := TRUE;
   END_TRANSITION
   STEP PressRingPut:   // S145, max time T#10S, warning time T#7S
              R    #ioPM_Inface.ProcessComplete
              S    #ioPM_Inface.ProcessStart
   END_STEP
   TRANSITION Trans639 FROM PressRingPut TO PressRingPutProcess   // T145, jump
      := TRUE;
   END_TRANSITION
   STEP "NG2Put_1Press/Glue":   // S160, max time T#10S, warning time T#7S
              R    #ioPM_Inface.ProcessComplete
              S    #ioPM_Inface.ProcessStart
   END_STEP
   TRANSITION Trans676 FROM "NG2Put_1Press/Glue" TO "NG PutProcess"   // T160, jump
      := TRUE;
   END_TRANSITION
   STEP "NG2Put_2/Magnet":   // S165, max time T#10S, warning time T#7S
              R    #ioPM_Inface.ProcessComplete
              S    #ioPM_Inface.ProcessStart
   END_STEP
   TRANSITION Trans677 FROM "NG2Put_2/Magnet" TO "NG 2 PutProcess"   // T165, jump
      := TRUE;
   END_TRANSITION
   STEP "NG2Put_3/Ring":   // S170, max time T#10S, warning time T#7S
              R    #ioPM_Inface.ProcessComplete
              S    #ioPM_Inface.ProcessStart
   END_STEP
   TRANSITION Trans679 FROM "NG2Put_3/Ring" TO "NG 3 PutProcess"   // T170, jump
      := TRUE;
   END_TRANSITION
   STEP Grip1SensorError:   // S381, max time T#10S, warning time T#7S
          S1  S    "ST10_DeviceError".F.Robot_3.Grip1SensorCheckError
   END_STEP
   TRANSITION Trans696 FROM Grip1SensorError TO RobotTaskSelect   // T696, jump
      := #iSysInface.Reset;
   END_TRANSITION
   STEP Grip2SensorError:   // S382, max time T#10S, warning time T#7S
          S1  S    "ST10_DeviceError".F.Robot_3.Grip2SensorCheckError
   END_STEP
   TRANSITION Trans697 FROM Grip2SensorError TO RobotTaskSelect   // T697, jump
      := #iSysInface.Reset;
   END_TRANSITION
   STEP PressPick:   // S150, max time T#10S, warning time T#7S
              R    #ioPM_Inface.ProcessComplete
              S    #ioPM_Inface.ProcessStart
   END_STEP
   TRANSITION Trans641 FROM PressPick TO PressPickProcess   // T150, jump
      := TRUE;
   END_TRANSITION
   STEP FlagReset:   // S272, max time T#10S, warning time T#7S
              R    "AutoProcessControl".Robot_3.Press2PutFlag
              R    "AutoProcessControl".Robot_3.Press2PickFlag
              R    "AutoProcessControl".Robot_3.GlueNGPickFlag
              R    "AutoProcessControl".Robot_3.ScanNGPickFlag
              R    "AutoProcessControl".Robot_3.NGPutFlag
   END_STEP
   TRANSITION Trans273 FROM FlagReset TO RobotTaskSelect   // T273
      := NOT "AutoProcessControl".Robot_3.Press2PutFlag AND NOT "AutoProcessControl".Robot_3.Press2PickFlag AND NOT "AutoProcessControl".Robot_3.GlueNGPickFlag AND NOT "AutoProcessControl".Robot_3.ScanNGPickFlag AND NOT "AutoProcessControl".Robot_3.NGPutFlag;
   END_TRANSITION
   STEP Maintenance:   // S131, max time T#10S, warning time T#7S
              R    #ioPM_Inface.ProcessComplete
              S    #ioPM_Inface.ProcessStart
   END_STEP
   TRANSITION Trans710 FROM Maintenance TO "Maintenance Pos"   // T131, jump
      := TRUE;
   END_TRANSITION
   STEP Masref_test:   // S132, max time T#10S, warning time T#7S
              R    #ioPM_Inface.ProcessComplete
              S    #ioPM_Inface.ProcessStart
   END_STEP
   TRANSITION Trans713 FROM Masref_test TO MasteringTest_Req   // T132, jump
      := TRUE;
   END_TRANSITION
   STEP Brake_Test:   // S133, max time T#10S, warning time T#7S
              R    #ioPM_Inface.ProcessComplete
              S    #ioPM_Inface.ProcessStart
   END_STEP
   TRANSITION Trans714 FROM Brake_Test TO BrakeTest_Req   // T133, jump
      := TRUE;
   END_TRANSITION

   // sequencer 3: S200-S249 Fixturecode reading
   STEP "Tablecode Scan":   // S200, max time T#10S, warning time T#7S
   END_STEP
   TRANSITION Trans147 FROM "Tablecode Scan" TO StartRobotScanGripperCode   // T200
      := TRUE;
   END_TRANSITION
   STEP WaitPos4ScanFinish:   // S319, max time T#10S, warning time T#7S
   END_STEP
   TRANSITION Trans628 FROM WaitPos4ScanFinish TO WaitRobotReachPos5   // T641
      := "KukaRobot3_CtrlDB".sPLCtoROB.User.Cycle.DI229_ScanPos4Complete;
   END_TRANSITION
   STEP WaitRobotReachPos3:   // S314, max time T#10S, warning time T#7S
   END_STEP
   TRANSITION P3 FROM WaitRobotReachPos3 TO WaitPos3ScanFinish   // T639
      := "KukaRobot3_CtrlDB".sROBtoPLC.User.Cycle.DO228_ScanPos3Reach;
   END_TRANSITION
   STEP WaitPos6ScanFinish:   // S323, max time T#10S, warning time T#7S
   END_STEP
   TRANSITION Trans644 FROM WaitPos6ScanFinish TO WaitRobotReachPos7   // T644
      := "KukaRobot3_CtrlDB".sPLCtoROB.User.Cycle.DI231_ScanPos6Complete;
   END_TRANSITION
   STEP WaitRobotReachPos5:   // S321, max time T#10S, warning time T#7S
   END_STEP
   TRANSITION P5 FROM WaitRobotReachPos5 TO WaitPos5ScanFinish   // T642
      := "KukaRobot3_CtrlDB".sROBtoPLC.User.Cycle.DO230_ScanPos5Reach;
   END_TRANSITION
   STEP WaitPos5ScanFinish:   // S320, max time T#10S, warning time T#7S
   END_STEP
   TRANSITION Trans643 FROM WaitPos5ScanFinish TO Step380   // T643
      := "KukaRobot3_CtrlDB".sPLCtoROB.User.Cycle.DI230_ScanPos5Complete;
   END_TRANSITION
   STEP WaitPos3ScanFinish:   // S315, max time T#10S, warning time T#7S
   END_STEP
   TRANSITION Trans624 FROM WaitPos3ScanFinish TO WaitRobotReachPos4   // T636
      := "KukaRobot3_CtrlDB".sPLCtoROB.User.Cycle.DI228_ScanPos3Complete;
   END_TRANSITION
   STEP WaitRobotReachPos2:   // S313, max time T#10S, warning time T#7S
   END_STEP
   TRANSITION P2 FROM WaitRobotReachPos2 TO WaitPos2ScanFinish   // T633
      := "KukaRobot3_CtrlDB".sROBtoPLC.User.Cycle.DO227_ScanPos2Reach;
   END_TRANSITION
   STEP StartRobotScanFixtureCode:   // S308, max time T#10S, warning time T#7S
              N    "KukaRobot3_CtrlDB".sPLCtoROB.User.Cycle.DI225_ScanPosReq
   END_STEP
   TRANSITION Trans605 FROM StartRobotScanFixtureCode TO WaitRobotReachPos1   // T605
      := "KukaRobot3_CtrlDB".sROBtoPLC.User.Cycle.DO225_ScanPosInside AND NOT "KukaRobot3_CtrlDB".sROBtoPLC.User.Cycle.DO233_ScanPoseFinish;
   END_TRANSITION
   STEP WaitRobotReachPos4:   // S318, max time T#10S, warning time T#7S
   END_STEP
   TRANSITION P4 FROM WaitRobotReachPos4 TO WaitPos4ScanFinish   // T640
      := "KukaRobot3_CtrlDB".sROBtoPLC.User.Cycle.DO229_ScanPos4Reach;
   END_TRANSITION
   STEP WaitPos1ScanFinish:   // S310, max time T#10S, warning time T#7S
   END_STEP
   TRANSITION Trans622 FROM WaitPos1ScanFinish TO WaitRobotReachPos2   // T621
      := "KukaRobot3_CtrlDB".sPLCtoROB.User.Cycle.DI226_ScanPos1Complete;
   END_TRANSITION
   STEP WaitRobotReachPos1:   // S309, max time T#10S, warning time T#7S
   END_STEP
   TRANSITION P1 FROM WaitRobotReachPos1 TO WaitPos1ScanFinish   // T617
      := "KukaRobot3_CtrlDB".sROBtoPLC.User.Cycle.DO226_ScanPos1Reach;
   END_TRANSITION
   STEP WaitPos2ScanFinish:   // S312, max time T#10S, warning time T#7S
   END_STEP
   TRANSITION Trans623 FROM WaitPos2ScanFinish TO WaitRobotReachPos3   // T624
      := "KukaRobot3_CtrlDB".sPLCtoROB.User.Cycle.DI227_ScanPos2Complete;
   END_TRANSITION
   STEP WaitRobotReachPos6:   // S322, max time T#10S, warning time T#7S
   END_STEP
   TRANSITION P6 FROM WaitRobotReachPos6 TO WaitPos6ScanFinish   // T645
      := "KukaRobot3_CtrlDB".sROBtoPLC.User.Cycle.DO231_ScanPos6Reach;
   END_TRANSITION
   STEP WaitPos7ScanFinish:   // S324, max time T#10S, warning time T#7S
   END_STEP
   TRANSITION Trans645 FROM WaitPos7ScanFinish TO "Wait ScanFinish"   // T646
      := "KukaRobot3_CtrlDB".sPLCtoROB.User.Cycle.DI232_ScanPos7Complete;
   END_TRANSITION
   STEP "Wait ScanFinish":   // S242, max time T#10S, warning time T#7S
   END_STEP
   TRANSITION Trans242 FROM "Wait ScanFinish" TO "Tablecode ScanFinish"   // T242
      := "KukaRobot3_CtrlDB".sROBtoPLC.User.Cycle.DO233_ScanPoseFinish;
   END_TRANSITION
   STEP WaitRobotReachPos7:   // S325, max time T#10S, warning time T#7S
   END_STEP
   TRANSITION P7 FROM WaitRobotReachPos7 TO WaitPos7ScanFinish   // T647
      := "KukaRobot3_CtrlDB".sROBtoPLC.User.Cycle.DO232_ScanPos7Reach;
   END_TRANSITION
   STEP "Tablecode ScanFinish":   // S149, max time T#10S, warning time T#7S
              S    #ioPM_Inface.ProcessComplete
              R    #ioPM_Inface.ProcessStart
   END_STEP
   TRANSITION Trans352 FROM "Tablecode ScanFinish" TO ProcessStart   // T149, jump
      := "ChangeOver_DB".Global.AllFixtureScanCompareOk OR "ChangeOver_DB".Robot_3.Req_RobotToMaintenancePos;
   END_TRANSITION
   STEP Step380:   // S380, max time T#10S, warning time T#7S
   END_STEP
   TRANSITION Trans692 FROM Step380 TO WaitRobotReachPos6   // T692
      := "AlwaysTRUE" AND NOT "AlwaysTRUE";
   END_TRANSITION
   TRANSITION Trans693 FROM Step380 TO "Tablecode ScanFinish"   // T693
      := "AlwaysTRUE";
   END_TRANSITION
   STEP StartRobotScanGripperCode:   // S334, max time T#10S, warning time T#7S
              N    "KukaRobot3_CtrlDB".sPLCtoROB.User.Cycle.DI305_GripScan
   END_STEP
   TRANSITION Trans684 FROM StartRobotScanGripperCode TO RobotScanGripperReachPos1   // T616
      := "KukaRobot3_CtrlDB".sROBtoPLC.User.Cycle.DO305_GripScanInside AND NOT "KukaRobot3_CtrlDB".sROBtoPLC.User.Cycle.DO306_GripScanFinish;
   END_TRANSITION
   STEP RobotScanGripperReachPos1:   // S335, max time T#10S, warning time T#7S
   END_STEP
   TRANSITION Trans685 FROM RobotScanGripperReachPos1 TO WaitGripperPos1ScanFinish   // T619
      := "KukaRobot3_CtrlDB".sROBtoPLC.User.Cycle.DO307_ScanPos1Reach;
   END_TRANSITION
   STEP WaitGripperPos1ScanFinish:   // S336, max time T#10S, warning time T#7S
   END_STEP
   TRANSITION Trans686 FROM WaitGripperPos1ScanFinish TO RobotScanGripperReachPos2   // T622
      := "KukaRobot3_CtrlDB".sPLCtoROB.User.Cycle.DI306_ScanPartComplete;
   END_TRANSITION
   STEP RobotScanGripperReachPos2:   // S337, max time T#10S, warning time T#7S
   END_STEP
   TRANSITION Trans687 FROM RobotScanGripperReachPos2 TO WaitGripperPos2ScanFinish   // T623
      := "KukaRobot3_CtrlDB".sROBtoPLC.User.Cycle.DO308_ScanPos2Reach;
   END_TRANSITION
   STEP WaitGripperPos2ScanFinish:   // S338, max time T#10S, warning time T#7S
   END_STEP
   TRANSITION Trans688 FROM WaitGripperPos2ScanFinish TO RobotScanGripperReachPos3   // T626
      := "KukaRobot3_CtrlDB".sPLCtoROB.User.Cycle.DI306_ScanPartComplete;
   END_TRANSITION
   STEP RobotScanGripperReachPos3:   // S339, max time T#10S, warning time T#7S
   END_STEP
   TRANSITION Trans689 FROM RobotScanGripperReachPos3 TO WaitGripperPos3ScanFinish   // T628
      := "KukaRobot3_CtrlDB".sROBtoPLC.User.Cycle.DO309_ScanPos3Reach;
   END_TRANSITION
   STEP WaitGripperPos3ScanFinish:   // S340, max time T#10S, warning time T#7S
   END_STEP
   TRANSITION Trans690 FROM WaitGripperPos3ScanFinish TO RobotScanGripperReachPos4   // T630
      := "KukaRobot3_CtrlDB".sPLCtoROB.User.Cycle.DI306_ScanPartComplete;
   END_TRANSITION
   STEP RobotScanGripperReachPos4:   // S341, max time T#10S, warning time T#7S
   END_STEP
   TRANSITION Trans703 FROM RobotScanGripperReachPos4 TO WaitGripperPos4ScanFinish   // T632
      := "KukaRobot3_CtrlDB".sROBtoPLC.User.Cycle.DO310_ScanPos4Reach;
   END_TRANSITION
   STEP WaitGripperPos4ScanFinish:   // S342, max time T#10S, warning time T#7S
   END_STEP
   TRANSITION Trans704 FROM WaitGripperPos4ScanFinish TO StartRobotScanFixtureCode   // T635
      := "KukaRobot3_CtrlDB".sROBtoPLC.User.Cycle.DO306_GripScanFinish AND "AutoProcessControl".Fixture2Code.Robot3CodeReadReq;
   END_TRANSITION

   // sequencer 4: S250-S299 PickPallet
   STEP PickPalletProcess:   // S250, max time T#10S, warning time T#7S
   END_STEP
   TRANSITION Trans150 FROM PickPalletProcess TO DataClear   // T250
      := TRUE;
   END_TRANSITION
   STEP StartRobotPickPalletShaft:   // S326, max time T#10S, warning time T#7S
              N    "KukaRobot3_CtrlDB".sPLCtoROB.User.Cycle.DI241_PickPalletReq
   END_STEP
   TRANSITION Trans607 FROM StartRobotPickPalletShaft TO WaitRobotGripHaveStatus   // T648
      := "KukaRobot3_CtrlDB".sROBtoPLC.User.Cycle.DO241_PickPalletInside AND NOT "KukaRobot3_CtrlDB".sROBtoPLC.User.Cycle.DO242_PickPalletFinish;
   END_TRANSITION
   STEP WaitRobotFinish:   // S327, max time T#10S, warning time T#7S
   END_STEP
   TRANSITION P8 FROM WaitRobotFinish TO PickPalletFinish   // T327
      := "KukaRobot3_CtrlDB".sROBtoPLC.User.Cycle.DO242_PickPalletFinish;
   END_TRANSITION
   STEP PickPalletFinish:   // S299, max time T#10S, warning time T#7S
              S    #ioPM_Inface.ProcessComplete
              R    #ioPM_Inface.ProcessStart
   END_STEP
   TRANSITION Trans654 FROM PickPalletFinish TO ProcessStart   // T299, jump
      := TRUE;
   END_TRANSITION
   STEP WaitRobotGripHaveStatus:   // S346, max time T#10S, warning time T#7S
   END_STEP
   TRANSITION Trans655 FROM WaitRobotGripHaveStatus TO Grip1PartStatus   // T655
      := "KukaRobot3_CtrlDB".sROBtoPLC.User.Public.GO5_RobGrip1Status <> 0;
   END_TRANSITION
   STEP Grip1PartStatus:   // S243, max time T#10S, warning time T#7S
              N    "AutoProcessData".F_Robot3Grip1.PartStatus:=100
   END_STEP
   TRANSITION Trans243 FROM Grip1PartStatus TO WaitRobotFinish   // T243
      := "AutoProcessData".F_Robot3Grip1.PartStatus = 100;
   END_TRANSITION
   STEP DataClear:   // S252, max time T#10S, warning time T#7S
          S1  N    "AutoProcessData".F_Robot3Grip1:="AutoProcessData".ClearData
   END_STEP
   TRANSITION Trans253 FROM DataClear TO StartRobotPickPalletShaft   // T253
      := TRUE;
   END_TRANSITION

   // sequencer 5: S300-S349 PickGlueNGR
   STEP PickGlueNGProcess:   // S300, max time T#10S, warning time T#7S
   END_STEP
   TRANSITION Trans300 FROM PickGlueNGProcess TO StartRobotPickGlueNG   // T300
      := TRUE;
   END_TRANSITION
   STEP DataMove:   // S253, max time T#10S, warning time T#7S
          S1  N    "AutoProcessData".F_Robot3Grip1:="AutoProcessData".C_GlueNGBuffer
          S1  N    "AutoProcessData".C_GlueNGBuffer:="AutoProcessData".ClearData
   END_STEP
   TRANSITION Trans254 FROM DataMove TO WaitRobotFinish_1   // T254
      := #DataMove.T > t#100MS;
   END_TRANSITION
   STEP StartRobotPickGlueNG:   // S328, max time T#10S, warning time T#7S
              N    "KukaRobot3_CtrlDB".sPLCtoROB.User.Cycle.DI253_PickGlueNGReq
   END_STEP
   TRANSITION Trans610 FROM StartRobotPickGlueNG TO WaitRobotGripHaveStatus_1   // T328
      := "KukaRobot3_CtrlDB".sROBtoPLC.User.Cycle.DO253_PickGlueNGInside AND NOT "KukaRobot3_CtrlDB".sROBtoPLC.User.Cycle.DO254_PickGlueNGFinish;
   END_TRANSITION
   STEP WaitRobotFinish_1:   // S343, max time T#10S, warning time T#7S
   END_STEP
   TRANSITION P9 FROM WaitRobotFinish_1 TO PickGlueNGFinish_1   // T651
      := "KukaRobot3_CtrlDB".sROBtoPLC.User.Cycle.DO254_PickGlueNGFinish;
   END_TRANSITION
   STEP PickGlueNGFinish_1:   // S349, max time T#10S, warning time T#7S
              S    #ioPM_Inface.ProcessComplete
              R    #ioPM_Inface.ProcessStart
   END_STEP
   TRANSITION Trans656 FROM PickGlueNGFinish_1 TO ProcessStart   // T349, jump
      := TRUE;
   END_TRANSITION
   STEP WaitRobotGripHaveStatus_1:   // S347, max time T#10S, warning time T#7S
   END_STEP
   TRANSITION Trans657 FROM WaitRobotGripHaveStatus_1 TO DataMove   // T656
      := "KukaRobot3_CtrlDB".sROBtoPLC.User.Public.GO5_RobGrip1Status <> 0;
   END_TRANSITION

   // sequencer 6: S350-S399 MagnScanNG
   STEP MagnScanNGProcess:   // S350, max time T#10S, warning time T#7S
   END_STEP
   TRANSITION Trans350 FROM MagnScanNGProcess TO StartRobotPickMagnScanNG   // T350
      := TRUE;
   END_TRANSITION
   STEP DataMove_1:   // S255, max time T#10S, warning time T#7S
          S1  N    "AutoProcessData".F_Robot3Grip2:="AutoProcessData".C_MagnScanNGBuffer
          S1  N    "AutoProcessData".C_MagnScanNGBuffer:="AutoProcessData".ClearData
   END_STEP
   TRANSITION Trans256 FROM DataMove_1 TO WaitRobotFinish_2   // T256
      := #DataMove_1.T > t#100MS;
   END_TRANSITION
   STEP StartRobotPickMagnScanNG:   // S344, max time T#10S, warning time T#7S
              N    "KukaRobot3_CtrlDB".sPLCtoROB.User.Cycle.DI249_PickMagnetNGReq
   END_STEP
   TRANSITION Trans611 FROM StartRobotPickMagnScanNG TO WaitRobotGripHaveStatus_2   // T652
      := "KukaRobot3_CtrlDB".sROBtoPLC.User.Cycle.DO249_PickMagnetInside AND NOT "KukaRobot3_CtrlDB".sROBtoPLC.User.Cycle.DO250_PickMagnetFinish;
   END_TRANSITION
   STEP WaitRobotFinish_2:   // S345, max time T#10S, warning time T#7S
   END_STEP
   TRANSITION P10 FROM WaitRobotFinish_2 TO Step930   // T653
      := "KukaRobot3_CtrlDB".sROBtoPLC.User.Cycle.DO250_PickMagnetFinish;
   END_TRANSITION
   STEP PickMagnScanNGBufferFinish:   // S399, max time T#10S, warning time T#7S
              S    #ioPM_Inface.ProcessComplete
              R    #ioPM_Inface.ProcessStart
   END_STEP
   TRANSITION Trans658 FROM PickMagnScanNGBufferFinish TO ProcessStart   // T399, jump
      := TRUE;
   END_TRANSITION
   STEP WaitRobotGripHaveStatus_2:   // S348, max time T#10S, warning time T#7S
   END_STEP
   TRANSITION Trans659 FROM WaitRobotGripHaveStatus_2 TO DataMove_1   // T657
      := "KukaRobot3_CtrlDB".sROBtoPLC.User.Public.GO6_RobGrip2Status <> 0;
   END_TRANSITION
   STEP Step930:   // S930, max time T#10S, warning time T#7S
              N    "AutoProcessData".F_Robot3Grip1.PartStatus:=444
   END_STEP
   TRANSITION Trans930 FROM Step930 TO PickMagnScanNGBufferFinish   // T930
      := #Step930.T > t#100MS;
   END_TRANSITION

   // sequencer 7: S400-S449 PickTable
   STEP PickTableProcess:   // S400, max time T#10S, warning time T#7S
   END_STEP
   TRANSITION Trans400 FROM PickTableProcess TO "Data Clear_2"   // T400
      := TRUE;
   END_TRANSITION
   STEP Grip2PartStatus:   // S244, max time T#10S, warning time T#7S
              N    "AutoProcessData".F_Robot3Grip2.PartStatus:=100
   END_STEP
   TRANSITION Trans244 FROM Grip2PartStatus TO WaitRobotFinish_3   // T244
      := "AutoProcessData".F_Robot3Grip2.PartStatus = 100;
   END_TRANSITION
   STEP StartRobotPickTable:   // S352, max time T#10S, warning time T#7S
              N    "KukaRobot3_CtrlDB".sPLCtoROB.User.Cycle.DI257_PickTableReq
   END_STEP
   TRANSITION Trans618 FROM StartRobotPickTable TO WaitRobotGripHaveStatus_3   // T654
      := "KukaRobot3_CtrlDB".sROBtoPLC.User.Cycle.DO257_PickTableInside AND NOT "KukaRobot3_CtrlDB".sROBtoPLC.User.Cycle.DO258_PickTableFinish;
   END_TRANSITION
   STEP WaitRobotFinish_3:   // S353, max time T#10S, warning time T#7S
   END_STEP
   TRANSITION P11 FROM WaitRobotFinish_3 TO PickTableProcessFinish   // T658
      := "KukaRobot3_CtrlDB".sROBtoPLC.User.Cycle.DO258_PickTableFinish;
   END_TRANSITION
   STEP PickTableProcessFinish:   // S449, max time T#10S, warning time T#7S
              S    #ioPM_Inface.ProcessComplete
              R    #ioPM_Inface.ProcessStart
   END_STEP
   TRANSITION Trans660 FROM PickTableProcessFinish TO ProcessStart   // T449, jump
      := TRUE;
   END_TRANSITION
   STEP WaitRobotGripHaveStatus_3:   // S354, max time T#10S, warning time T#7S
   END_STEP
   TRANSITION Trans661 FROM WaitRobotGripHaveStatus_3 TO Grip2PartStatus   // T659
      := "KukaRobot3_CtrlDB".sROBtoPLC.User.Public.GO6_RobGrip2Status <> 0;
   END_TRANSITION
   STEP "Data Clear_2":   // S258, max time T#10S, warning time T#7S
          S1  N    "AutoProcessData".F_Robot3Grip2:="AutoProcessData".ClearData
   END_STEP
   TRANSITION Trans259 FROM "Data Clear_2" TO StartRobotPickTable   // T259
      := #"Data Clear_2".T > t#100MS;
   END_TRANSITION

   // sequencer 8: S450-S499 ScanRing
   STEP ScanRingProcess:   // S450, max time T#10S, warning time T#7S
   END_STEP
   TRANSITION Trans450 FROM ScanRingProcess TO StartRobotScanRing   // T450
      := TRUE;
   END_TRANSITION
   STEP CheckScanReady:   // S245, max time T#10S, warning time T#7S
   END_STEP
   TRANSITION Trans245 FROM CheckScanReady TO ScanStart   // T245
      := "KeyenceSR1000Ctrl_803A1DB".oReady;
   END_TRANSITION
   STEP StartRobotScanRing:   // S355, max time T#10S, warning time T#7S
              N    "KukaRobot3_CtrlDB".sPLCtoROB.User.Cycle.DI261_ScanRingReq
   END_STEP
   TRANSITION Trans619 FROM StartRobotScanRing TO WaitRobotReachScanPos   // T660
      := "KukaRobot3_CtrlDB".sROBtoPLC.User.Cycle.DO261_ScanRingtInside AND NOT "KukaRobot3_CtrlDB".sROBtoPLC.User.Cycle.DO262_ScanRingFinish;
   END_TRANSITION
   STEP WaitRobotFinish_4:   // S356, max time T#10S, warning time T#7S
              N    "KukaRobot3_CtrlDB".sPLCtoROB.User.Cycle.DI262_ScanRingComplete
   END_STEP
   TRANSITION P12 FROM WaitRobotFinish_4 TO ScanRingProcessFinish   // T661
      := "KukaRobot3_CtrlDB".sROBtoPLC.User.Cycle.DO262_ScanRingFinish;
   END_TRANSITION
   STEP ScanRingProcessFinish:   // S499, max time T#10S, warning time T#7S
              S    #ioPM_Inface.ProcessComplete
              R    #ioPM_Inface.ProcessStart
   END_STEP
   TRANSITION Trans662 FROM ScanRingProcessFinish TO ProcessStart   // T499, jump
      := TRUE;
   END_TRANSITION
   STEP WaitRobotReachScanPos:   // S357, max time T#10S, warning time T#7S
   END_STEP
   TRANSITION Trans663 FROM WaitRobotReachScanPos TO CheckScanReady   // T662
      := "KukaRobot3_CtrlDB".sROBtoPLC.User.Cycle.DO263_ScanReach;
   END_TRANSITION
   STEP ScanStart:   // S246, max time T#10S, warning time T#7S
          S1  S    "KeyenceSR1000Ctrl_803A1DB".ioAutoTrigger
   END_STEP
   TRANSITION Trans246 FROM ScanStart TO WaitScanCompletely   // T246
      := NOT "KeyenceSR1000Ctrl_803A1DB".sHMI.Status.Ready;
   END_TRANSITION
   STEP WaitScanCompletely:   // S247, max time T#10S, warning time T#7S
   END_STEP
   TRANSITION Trans247 FROM WaitScanCompletely TO CodeMove   // T247
      := "KeyenceSR1000Ctrl_803A1DB".sHMI.Status.Complete AND "KeyenceSR1000Ctrl_803A1DB".sHMI.Status.ReadOk;
   END_TRANSITION
   TRANSITION Trans248 FROM WaitScanCompletely TO PartNGStatus   // T248
      := "KeyenceSR1000Ctrl_803A1DB".sHMI.Status.Complete AND "KeyenceSR1000Ctrl_803A1DB".sHMI.Status.ReadNok;
   END_TRANSITION
   STEP CodeMove:   // S248, max time T#10S, warning time T#7S
              N    "AutoProcessData".F_Robot3Grip2.RingCode_2:="KeyenceSR1000Ctrl_803A1DB".sHMI.Status.CurrentCode
   END_STEP
   TRANSITION Trans249 FROM CodeMove TO PartOKStatus_1   // T249
      := TRUE;
   END_TRANSITION
   STEP PartOKStatus:   // S249, max time T#10S, warning time T#7S
              N    "AutoProcessData".F_Robot3Grip2.PartStatus:=199
   END_STEP
   TRANSITION Trans251 FROM PartOKStatus TO WaitRobotFinish_4   // T251
      := "AutoProcessData".F_Robot3Grip2.PartStatus = 199;
   END_TRANSITION
   STEP PartNGStatus:   // S251, max time T#10S, warning time T#7S
              N    "AutoProcessData".F_Robot3Grip2.PartStatus:=150
   END_STEP
   TRANSITION Trans252 FROM PartNGStatus TO WaitRobotFinish_4   // T252
      := "AutoProcessData".F_Robot3Grip2.PartStatus = 150;
   END_TRANSITION
   STEP "MES Online  offline?":   // S385, max time T#10S, warning time T#7S
   END_STEP
   TRANSITION Offline FROM "MES Online  offline?" TO PartOKStatus   // T702
      := "Station_Sys".Cmd.OnOffLine;
   END_TRANSITION
   TRANSITION Trans702 FROM "MES Online  offline?" TO WaitRobotFinish_4   // T704
      := NOT "Station_Sys".Cmd.OnOffLine;
   END_TRANSITION
   STEP PartOKStatus_1:   // S273, max time T#10S, warning time T#7S
              N    "AutoProcessData".F_Robot3Grip2.PartStatus:=110
   END_STEP
   TRANSITION Trans274 FROM PartOKStatus_1 TO "MES Online  offline?"   // T274
      := "AutoProcessData".F_Robot3Grip2.PartStatus = 110;
   END_TRANSITION

   // sequencer 9: S500-S549 PressShaftPut
   STEP PressShaftPutProcess:   // S500, max time T#10S, warning time T#7S
   END_STEP
   TRANSITION Trans500 FROM PressShaftPutProcess TO StartRobotPressShaftPut   // T500
      := TRUE;
   END_TRANSITION
   STEP DataMove_2:   // S257, max time T#10S, warning time T#7S
          S1  N    "AutoProcessData".B_Press2:="AutoProcessData".F_Robot3Grip1
          S1  N    "AutoProcessData".F_Robot3Grip1:="AutoProcessData".ClearData
   END_STEP
   TRANSITION Trans258 FROM DataMove_2 TO WaitRobotFinish_5   // T258
      := #DataMove_2.T > t#100MS;
   END_TRANSITION
   STEP StartRobotPressShaftPut:   // S358, max time T#10S, warning time T#7S
              N    "KukaRobot3_CtrlDB".sPLCtoROB.User.Cycle.DI273_PressPutPart1Req
   END_STEP
   TRANSITION Trans646 FROM StartRobotPressShaftPut TO WaitRobotGripStatus   // T663
      := "KukaRobot3_CtrlDB".sROBtoPLC.User.Cycle.DO273_PressPutPart1Inside AND NOT "KukaRobot3_CtrlDB".sROBtoPLC.User.Cycle.DO274_PressPutPart1Finish;
   END_TRANSITION
   STEP WaitRobotFinish_5:   // S359, max time T#10S, warning time T#7S
   END_STEP
   TRANSITION P13 FROM WaitRobotFinish_5 TO PressShaftPutProcessFinish   // T664
      := "KukaRobot3_CtrlDB".sROBtoPLC.User.Cycle.DO274_PressPutPart1Finish;
   END_TRANSITION
   STEP PressShaftPutProcessFinish:   // S549, max time T#10S, warning time T#7S
              S    #ioPM_Inface.ProcessComplete
              R    #ioPM_Inface.ProcessStart
   END_STEP
   TRANSITION Trans664 FROM PressShaftPutProcessFinish TO ProcessStart   // T549, jump
      := TRUE;
   END_TRANSITION
   STEP WaitRobotGripStatus:   // S360, max time T#10S, warning time T#7S
   END_STEP
   TRANSITION Trans665 FROM WaitRobotGripStatus TO DataMove_2   // T665
      := "KukaRobot3_CtrlDB".sROBtoPLC.User.Public.GO5_RobGrip1Status = 0;
   END_TRANSITION

